// TIA Portal V17 export
// export: Created 2025-05-22T12:27:02.8614335Z, ExportSetting WithDefaults, DisplayName Totally Integrated Automation Portal, DisplayVersion V17 Update 8, DisplayName TIA Portal Openness, DisplayVersion V17 Update 8, DisplayName TIA Portal Version Control Interface, DisplayVersion V17, DisplayName SINAMICS Startdrive Advanced, DisplayVersion V17 SP2, DisplayName SINAMICS Startdrive G110M, G120, G120C, G120D, G120P, G115D, DisplayVersion V17 SP2, DisplayName SINAMICS Startdrive G130, G150, S120, S150, SINAMICS MV, S210, DisplayVersion V17 SP2, DisplayName STEP 7 Professional, DisplayVersion V17 Update 8, DisplayName SINUMERIK ONE STEP 7 Toolbox, DisplayVersion V17 Update 12, DisplayName SINUMERIK ONE PLC Basic Program Plus, DisplayVersion V17 Update 12, DisplayName SINUMERIK 840D sl STEP 7 Toolbox, DisplayVersion V17 Update 12, DisplayName STEP 7 Safety, DisplayVersion V17 Update 6, DisplayName WinCC Advanced, DisplayVersion V17 Update 8
FUNCTION "FC16701_OPC_UA_MASTER_MACHINE_DATA_UPDATE" : Void   // FC16701, LAD
{ S7_Optimized_Access := 'FALSE' }
VERSION : 0.1
// stored: AutoNumber false, IsIECCheckEnabled false, SetENOAutomatically false, UDAEnableTagReadback false
   VAR_TEMP
      RETVAL : Word;
      ZERO : Byte;   // ZERO
      STATUS_FILL : Int;   // STATUS FILL
      U01_ASPIRATION_FINAL_VALUE_AUX : Real;
      U02_ASPIRATION_FINAL_VALUE_AUX : Real;
   END_VAR
   VAR_TEMP   // added for the SCL form of the ladder/FBD networks
      _w1 : Bool;
      _w2 : Bool;
      _w3 : Bool;
      _w4 : Bool;
      _w5 : Bool;
   END_VAR
BEGIN

REGION Network 1: <<<<<<<<<<<<<<<<<<<< OPC UA MASTER MACHINE >>>>>>>>>>>>>>>>>>>>
END_REGION

REGION Network 2: GENERAL INFO - ID
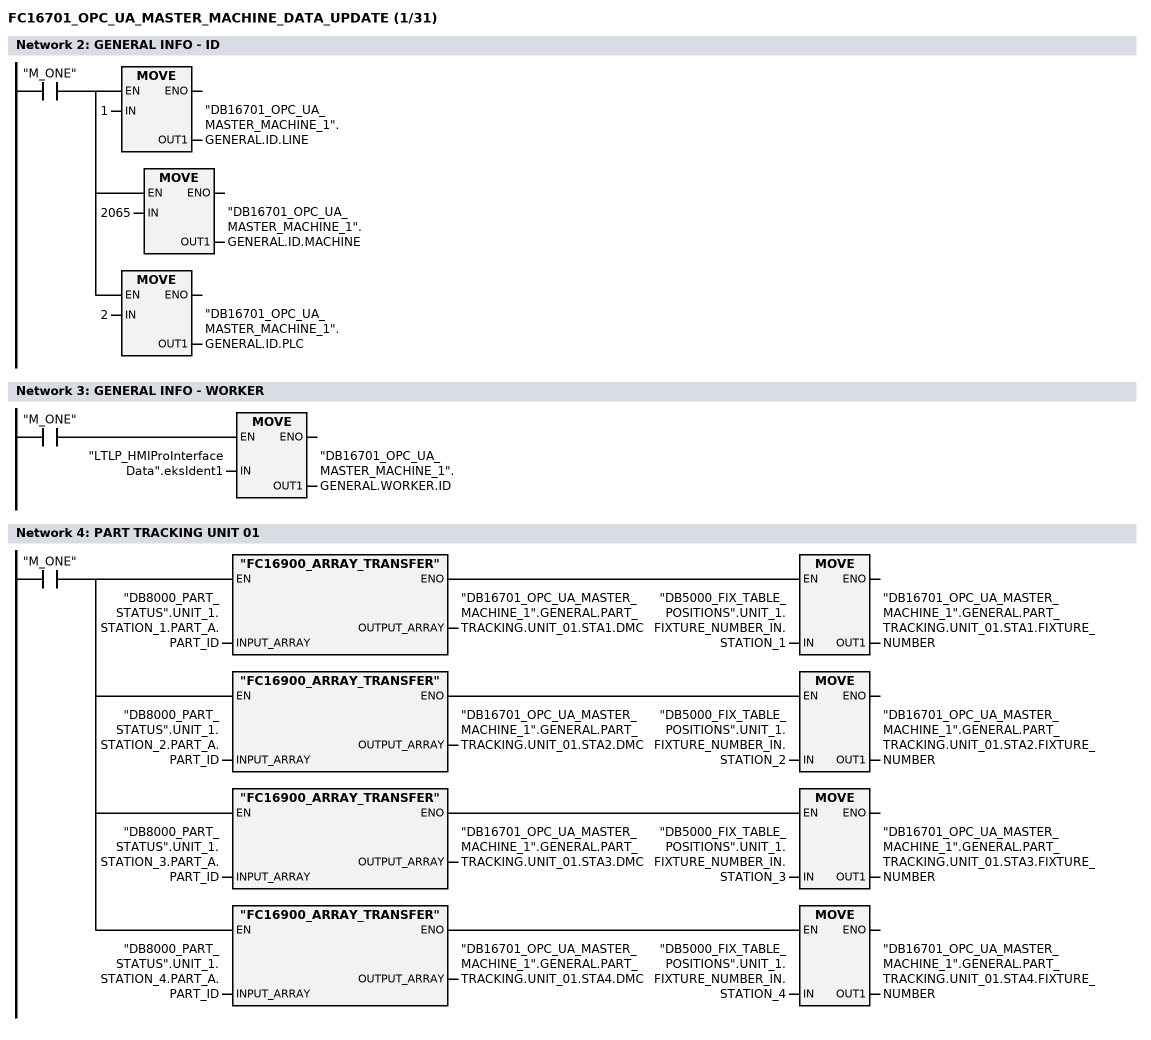
   RUNG wire#powerrail
      Contact( "M_ONE" )
      wire#w1
      Move(in := 1, out1 => "DB16701_OPC_UA_MASTER_MACHINE_1".GENERAL.ID.LINE)
   END_RUNG
   RUNG wire#w1
      Move(in := 2065, out1 => "DB16701_OPC_UA_MASTER_MACHINE_1".GENERAL.ID.MACHINE)
   END_RUNG
   RUNG wire#w1
      Move(in := 2, out1 => "DB16701_OPC_UA_MASTER_MACHINE_1".GENERAL.ID.PLC)
   END_RUNG
   // the same network as SCL:
   IF "M_ONE" THEN
       "DB16701_OPC_UA_MASTER_MACHINE_1".GENERAL.ID.LINE := 1;
       "DB16701_OPC_UA_MASTER_MACHINE_1".GENERAL.ID.MACHINE := 2065;
       "DB16701_OPC_UA_MASTER_MACHINE_1".GENERAL.ID.PLC := 2;
   END_IF;
END_REGION

REGION Network 3: GENERAL INFO - WORKER
   RUNG wire#powerrail
      Contact( "M_ONE" )
      Move(in := "LTLP_HMIProInterfaceData".eksIdent1, out1 => "DB16701_OPC_UA_MASTER_MACHINE_1".GENERAL.WORKER.ID)
   END_RUNG
   // the same network as SCL:
   IF "M_ONE" THEN
       "DB16701_OPC_UA_MASTER_MACHINE_1".GENERAL.WORKER.ID := "LTLP_HMIProInterfaceData".eksIdent1;
   END_IF;
END_REGION

REGION Network 4: PART TRACKING UNIT 01
   RUNG wire#powerrail
      Contact( "M_ONE" )
      wire#w1
      "FC16900_ARRAY_TRANSFER"(INPUT_ARRAY := "DB8000_PART_STATUS".UNIT_1.STATION_1.PART_A.PART_ID, OUTPUT_ARRAY => "DB16701_OPC_UA_MASTER_MACHINE_1".GENERAL.PART_TRACKING.UNIT_01.STA1.DMC)
      Move(in := "DB5000_FIX_TABLE_POSITIONS".UNIT_1.FIXTURE_NUMBER_IN.STATION_1, out1 => "DB16701_OPC_UA_MASTER_MACHINE_1".GENERAL.PART_TRACKING.UNIT_01.STA1.FIXTURE_NUMBER)
   END_RUNG
   RUNG wire#w1
      "FC16900_ARRAY_TRANSFER"(INPUT_ARRAY := "DB8000_PART_STATUS".UNIT_1.STATION_2.PART_A.PART_ID, OUTPUT_ARRAY => "DB16701_OPC_UA_MASTER_MACHINE_1".GENERAL.PART_TRACKING.UNIT_01.STA2.DMC)
      Move(in := "DB5000_FIX_TABLE_POSITIONS".UNIT_1.FIXTURE_NUMBER_IN.STATION_2, out1 => "DB16701_OPC_UA_MASTER_MACHINE_1".GENERAL.PART_TRACKING.UNIT_01.STA2.FIXTURE_NUMBER)
   END_RUNG
   RUNG wire#w1
      "FC16900_ARRAY_TRANSFER"(INPUT_ARRAY := "DB8000_PART_STATUS".UNIT_1.STATION_3.PART_A.PART_ID, OUTPUT_ARRAY => "DB16701_OPC_UA_MASTER_MACHINE_1".GENERAL.PART_TRACKING.UNIT_01.STA3.DMC)
      Move(in := "DB5000_FIX_TABLE_POSITIONS".UNIT_1.FIXTURE_NUMBER_IN.STATION_3, out1 => "DB16701_OPC_UA_MASTER_MACHINE_1".GENERAL.PART_TRACKING.UNIT_01.STA3.FIXTURE_NUMBER)
   END_RUNG
   RUNG wire#w1
      "FC16900_ARRAY_TRANSFER"(INPUT_ARRAY := "DB8000_PART_STATUS".UNIT_1.STATION_4.PART_A.PART_ID, OUTPUT_ARRAY => "DB16701_OPC_UA_MASTER_MACHINE_1".GENERAL.PART_TRACKING.UNIT_01.STA4.DMC)
      Move(in := "DB5000_FIX_TABLE_POSITIONS".UNIT_1.FIXTURE_NUMBER_IN.STATION_4, out1 => "DB16701_OPC_UA_MASTER_MACHINE_1".GENERAL.PART_TRACKING.UNIT_01.STA4.FIXTURE_NUMBER)
   END_RUNG
   // the same network as SCL:
   #_w2 := "M_ONE";
   "FC16900_ARRAY_TRANSFER"(EN := "M_ONE",
                           INPUT_ARRAY := "DB8000_PART_STATUS".UNIT_1.STATION_1.PART_A.PART_ID,
                           OUTPUT_ARRAY => "DB16701_OPC_UA_MASTER_MACHINE_1".GENERAL.PART_TRACKING.UNIT_01.STA1.DMC,
                           ENO => #_w1);
   IF #_w1 THEN
       "DB16701_OPC_UA_MASTER_MACHINE_1".GENERAL.PART_TRACKING.UNIT_01.STA1.FIXTURE_NUMBER := "DB5000_FIX_TABLE_POSITIONS".UNIT_1.FIXTURE_NUMBER_IN.STATION_1;
   END_IF;
   "FC16900_ARRAY_TRANSFER"(EN := #_w2,
                           INPUT_ARRAY := "DB8000_PART_STATUS".UNIT_1.STATION_2.PART_A.PART_ID,
                           OUTPUT_ARRAY => "DB16701_OPC_UA_MASTER_MACHINE_1".GENERAL.PART_TRACKING.UNIT_01.STA2.DMC,
                           ENO => #_w3);
   IF #_w3 THEN
       "DB16701_OPC_UA_MASTER_MACHINE_1".GENERAL.PART_TRACKING.UNIT_01.STA2.FIXTURE_NUMBER := "DB5000_FIX_TABLE_POSITIONS".UNIT_1.FIXTURE_NUMBER_IN.STATION_2;
   END_IF;
   "FC16900_ARRAY_TRANSFER"(EN := #_w2,
                           INPUT_ARRAY := "DB8000_PART_STATUS".UNIT_1.STATION_3.PART_A.PART_ID,
                           OUTPUT_ARRAY => "DB16701_OPC_UA_MASTER_MACHINE_1".GENERAL.PART_TRACKING.UNIT_01.STA3.DMC,
                           ENO => #_w4);
   IF #_w4 THEN
       "DB16701_OPC_UA_MASTER_MACHINE_1".GENERAL.PART_TRACKING.UNIT_01.STA3.FIXTURE_NUMBER := "DB5000_FIX_TABLE_POSITIONS".UNIT_1.FIXTURE_NUMBER_IN.STATION_3;
   END_IF;
   "FC16900_ARRAY_TRANSFER"(EN := #_w2,
                           INPUT_ARRAY := "DB8000_PART_STATUS".UNIT_1.STATION_4.PART_A.PART_ID,
                           OUTPUT_ARRAY => "DB16701_OPC_UA_MASTER_MACHINE_1".GENERAL.PART_TRACKING.UNIT_01.STA4.DMC,
                           ENO => #_w5);
   IF #_w5 THEN
       "DB16701_OPC_UA_MASTER_MACHINE_1".GENERAL.PART_TRACKING.UNIT_01.STA4.FIXTURE_NUMBER := "DB5000_FIX_TABLE_POSITIONS".UNIT_1.FIXTURE_NUMBER_IN.STATION_4;
   END_IF;
END_REGION

REGION Network 5: PART TRACKING UNIT 02
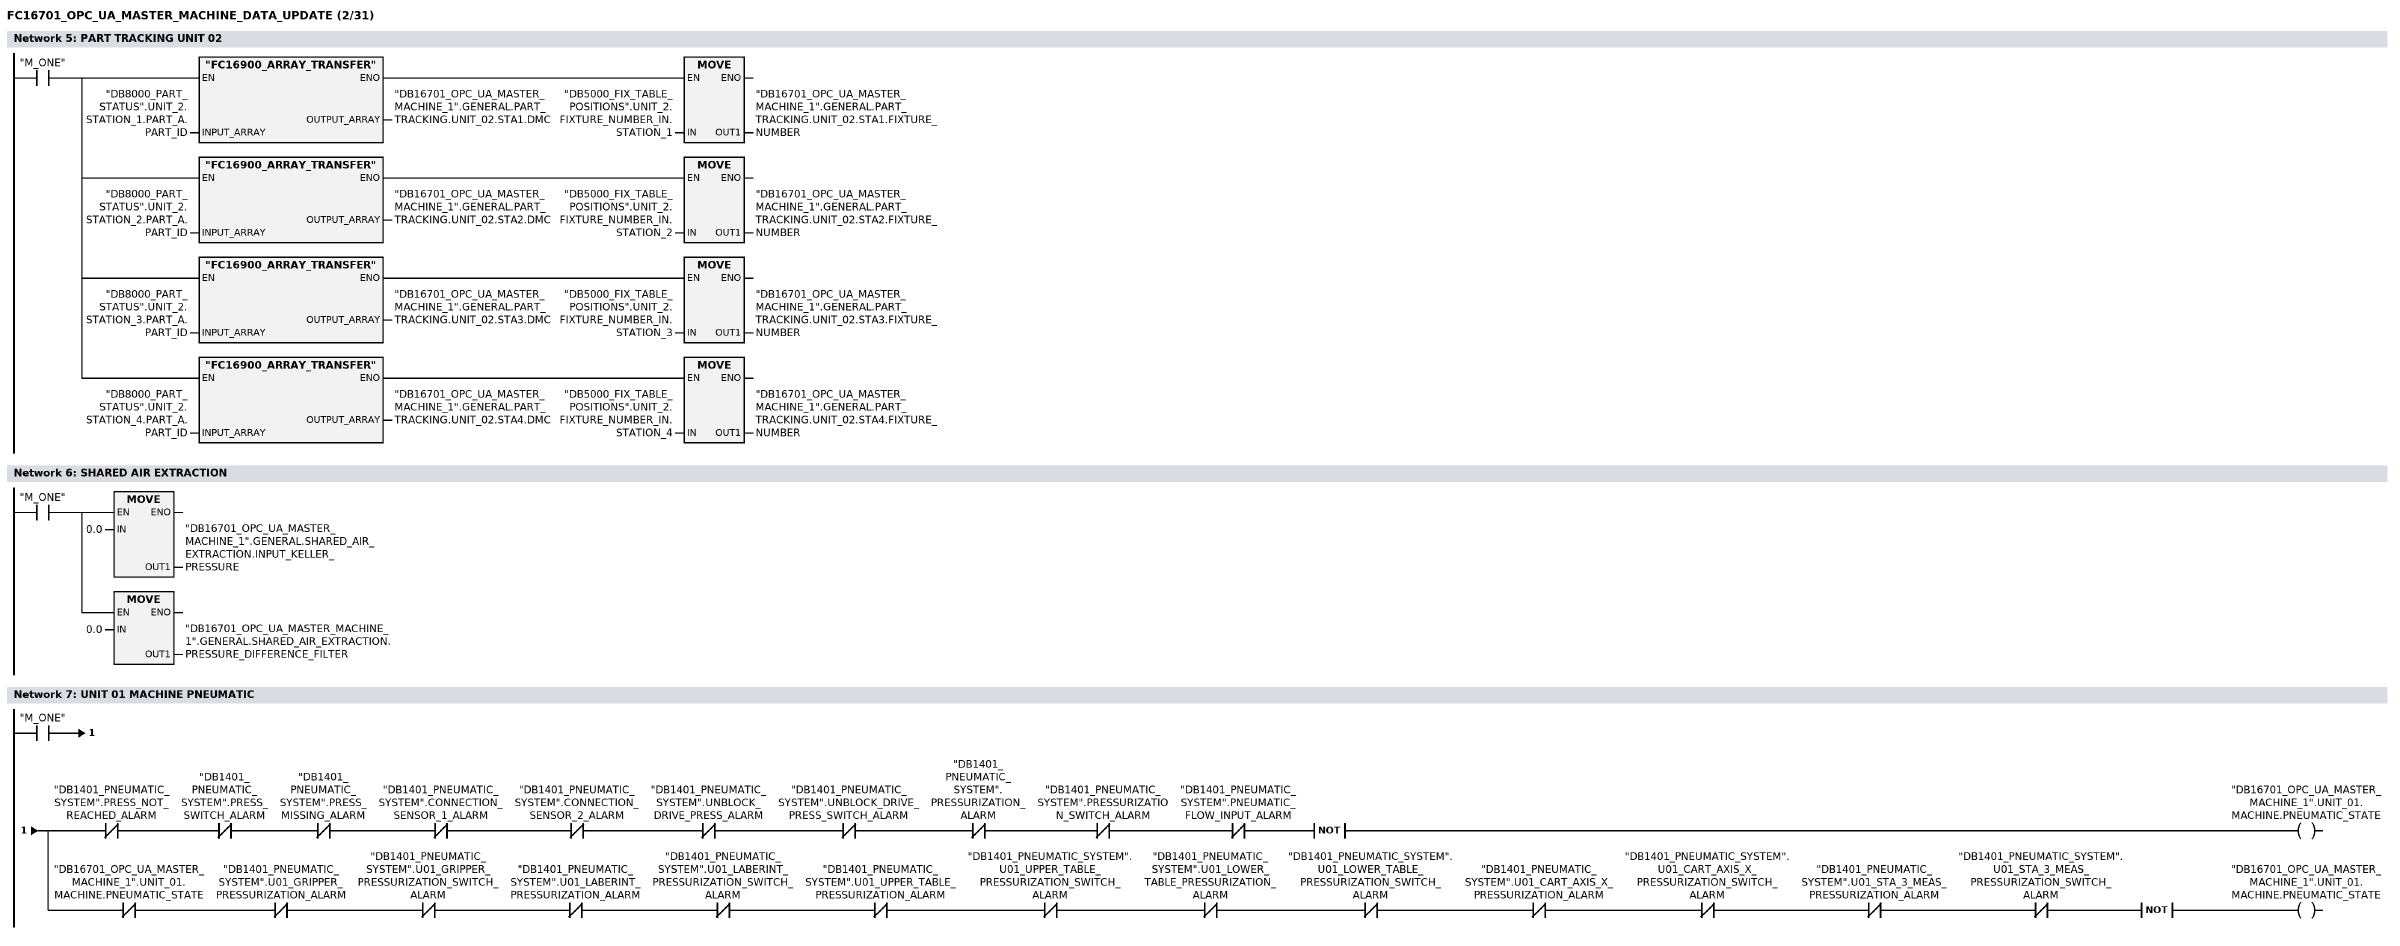
   RUNG wire#powerrail
      Contact( "M_ONE" )
      wire#w1
      "FC16900_ARRAY_TRANSFER"(INPUT_ARRAY := "DB8000_PART_STATUS".UNIT_2.STATION_1.PART_A.PART_ID, OUTPUT_ARRAY => "DB16701_OPC_UA_MASTER_MACHINE_1".GENERAL.PART_TRACKING.UNIT_02.STA1.DMC)
      Move(in := "DB5000_FIX_TABLE_POSITIONS".UNIT_2.FIXTURE_NUMBER_IN.STATION_1, out1 => "DB16701_OPC_UA_MASTER_MACHINE_1".GENERAL.PART_TRACKING.UNIT_02.STA1.FIXTURE_NUMBER)
   END_RUNG
   RUNG wire#w1
      "FC16900_ARRAY_TRANSFER"(INPUT_ARRAY := "DB8000_PART_STATUS".UNIT_2.STATION_2.PART_A.PART_ID, OUTPUT_ARRAY => "DB16701_OPC_UA_MASTER_MACHINE_1".GENERAL.PART_TRACKING.UNIT_02.STA2.DMC)
      Move(in := "DB5000_FIX_TABLE_POSITIONS".UNIT_2.FIXTURE_NUMBER_IN.STATION_2, out1 => "DB16701_OPC_UA_MASTER_MACHINE_1".GENERAL.PART_TRACKING.UNIT_02.STA2.FIXTURE_NUMBER)
   END_RUNG
   RUNG wire#w1
      "FC16900_ARRAY_TRANSFER"(INPUT_ARRAY := "DB8000_PART_STATUS".UNIT_2.STATION_3.PART_A.PART_ID, OUTPUT_ARRAY => "DB16701_OPC_UA_MASTER_MACHINE_1".GENERAL.PART_TRACKING.UNIT_02.STA3.DMC)
      Move(in := "DB5000_FIX_TABLE_POSITIONS".UNIT_2.FIXTURE_NUMBER_IN.STATION_3, out1 => "DB16701_OPC_UA_MASTER_MACHINE_1".GENERAL.PART_TRACKING.UNIT_02.STA3.FIXTURE_NUMBER)
   END_RUNG
   RUNG wire#w1
      "FC16900_ARRAY_TRANSFER"(INPUT_ARRAY := "DB8000_PART_STATUS".UNIT_2.STATION_4.PART_A.PART_ID, OUTPUT_ARRAY => "DB16701_OPC_UA_MASTER_MACHINE_1".GENERAL.PART_TRACKING.UNIT_02.STA4.DMC)
      Move(in := "DB5000_FIX_TABLE_POSITIONS".UNIT_2.FIXTURE_NUMBER_IN.STATION_4, out1 => "DB16701_OPC_UA_MASTER_MACHINE_1".GENERAL.PART_TRACKING.UNIT_02.STA4.FIXTURE_NUMBER)
   END_RUNG
   // the same network as SCL:
   #_w2 := "M_ONE";
   "FC16900_ARRAY_TRANSFER"(EN := "M_ONE",
                           INPUT_ARRAY := "DB8000_PART_STATUS".UNIT_2.STATION_1.PART_A.PART_ID,
                           OUTPUT_ARRAY => "DB16701_OPC_UA_MASTER_MACHINE_1".GENERAL.PART_TRACKING.UNIT_02.STA1.DMC,
                           ENO => #_w1);
   IF #_w1 THEN
       "DB16701_OPC_UA_MASTER_MACHINE_1".GENERAL.PART_TRACKING.UNIT_02.STA1.FIXTURE_NUMBER := "DB5000_FIX_TABLE_POSITIONS".UNIT_2.FIXTURE_NUMBER_IN.STATION_1;
   END_IF;
   "FC16900_ARRAY_TRANSFER"(EN := #_w2,
                           INPUT_ARRAY := "DB8000_PART_STATUS".UNIT_2.STATION_2.PART_A.PART_ID,
                           OUTPUT_ARRAY => "DB16701_OPC_UA_MASTER_MACHINE_1".GENERAL.PART_TRACKING.UNIT_02.STA2.DMC,
                           ENO => #_w3);
   IF #_w3 THEN
       "DB16701_OPC_UA_MASTER_MACHINE_1".GENERAL.PART_TRACKING.UNIT_02.STA2.FIXTURE_NUMBER := "DB5000_FIX_TABLE_POSITIONS".UNIT_2.FIXTURE_NUMBER_IN.STATION_2;
   END_IF;
   "FC16900_ARRAY_TRANSFER"(EN := #_w2,
                           INPUT_ARRAY := "DB8000_PART_STATUS".UNIT_2.STATION_3.PART_A.PART_ID,
                           OUTPUT_ARRAY => "DB16701_OPC_UA_MASTER_MACHINE_1".GENERAL.PART_TRACKING.UNIT_02.STA3.DMC,
                           ENO => #_w4);
   IF #_w4 THEN
       "DB16701_OPC_UA_MASTER_MACHINE_1".GENERAL.PART_TRACKING.UNIT_02.STA3.FIXTURE_NUMBER := "DB5000_FIX_TABLE_POSITIONS".UNIT_2.FIXTURE_NUMBER_IN.STATION_3;
   END_IF;
   "FC16900_ARRAY_TRANSFER"(EN := #_w2,
                           INPUT_ARRAY := "DB8000_PART_STATUS".UNIT_2.STATION_4.PART_A.PART_ID,
                           OUTPUT_ARRAY => "DB16701_OPC_UA_MASTER_MACHINE_1".GENERAL.PART_TRACKING.UNIT_02.STA4.DMC,
                           ENO => #_w5);
   IF #_w5 THEN
       "DB16701_OPC_UA_MASTER_MACHINE_1".GENERAL.PART_TRACKING.UNIT_02.STA4.FIXTURE_NUMBER := "DB5000_FIX_TABLE_POSITIONS".UNIT_2.FIXTURE_NUMBER_IN.STATION_4;
   END_IF;
END_REGION

REGION Network 6: SHARED AIR EXTRACTION
   RUNG wire#powerrail
      Contact( "M_ONE" )
      wire#w1
      Move(in := 0.0, out1 => "DB16701_OPC_UA_MASTER_MACHINE_1".GENERAL.SHARED_AIR_EXTRACTION.INPUT_KELLER_PRESSURE)
   END_RUNG
   RUNG wire#w1
      Move(in := 0.0, out1 => "DB16701_OPC_UA_MASTER_MACHINE_1".GENERAL.SHARED_AIR_EXTRACTION.PRESSURE_DIFFERENCE_FILTER)
   END_RUNG
   // the same network as SCL:
   IF "M_ONE" THEN
       "DB16701_OPC_UA_MASTER_MACHINE_1".GENERAL.SHARED_AIR_EXTRACTION.INPUT_KELLER_PRESSURE := 0.0;
       "DB16701_OPC_UA_MASTER_MACHINE_1".GENERAL.SHARED_AIR_EXTRACTION.PRESSURE_DIFFERENCE_FILTER := 0.0;
   END_IF;
END_REGION

REGION Network 7: UNIT 01 MACHINE PNEUMATIC
   RUNG wire#powerrail
      Contact( "M_ONE" )
      wire#w1
      I_Contact( "DB1401_PNEUMATIC_SYSTEM".PRESS_NOT_REACHED_ALARM )
      I_Contact( "DB1401_PNEUMATIC_SYSTEM".PRESS_SWITCH_ALARM )
      I_Contact( "DB1401_PNEUMATIC_SYSTEM".PRESS_MISSING_ALARM )
      I_Contact( "DB1401_PNEUMATIC_SYSTEM".CONNECTION_SENSOR_1_ALARM )
      I_Contact( "DB1401_PNEUMATIC_SYSTEM".CONNECTION_SENSOR_2_ALARM )
      I_Contact( "DB1401_PNEUMATIC_SYSTEM".UNBLOCK_DRIVE_PRESS_ALARM )
      I_Contact( "DB1401_PNEUMATIC_SYSTEM".UNBLOCK_DRIVE_PRESS_SWITCH_ALARM )
      I_Contact( "DB1401_PNEUMATIC_SYSTEM".PRESSURIZATION_ALARM )
      I_Contact( "DB1401_PNEUMATIC_SYSTEM".PRESSURIZATION_SWITCH_ALARM )
      I_Contact( "DB1401_PNEUMATIC_SYSTEM".PNEUMATIC_FLOW_INPUT_ALARM )
      Not()
      Coil( "DB16701_OPC_UA_MASTER_MACHINE_1".UNIT_01.MACHINE.PNEUMATIC_STATE )
   END_RUNG
   RUNG wire#w1
      I_Contact( "DB16701_OPC_UA_MASTER_MACHINE_1".UNIT_01.MACHINE.PNEUMATIC_STATE )
      I_Contact( "DB1401_PNEUMATIC_SYSTEM".U01_GRIPPER_PRESSURIZATION_ALARM )
      I_Contact( "DB1401_PNEUMATIC_SYSTEM".U01_GRIPPER_PRESSURIZATION_SWITCH_ALARM )
      I_Contact( "DB1401_PNEUMATIC_SYSTEM".U01_LABERINT_PRESSURIZATION_ALARM )
      I_Contact( "DB1401_PNEUMATIC_SYSTEM".U01_LABERINT_PRESSURIZATION_SWITCH_ALARM )
      I_Contact( "DB1401_PNEUMATIC_SYSTEM".U01_UPPER_TABLE_PRESSURIZATION_ALARM )
      I_Contact( "DB1401_PNEUMATIC_SYSTEM".U01_UPPER_TABLE_PRESSURIZATION_SWITCH_ALARM )
      I_Contact( "DB1401_PNEUMATIC_SYSTEM".U01_LOWER_TABLE_PRESSURIZATION_ALARM )
      I_Contact( "DB1401_PNEUMATIC_SYSTEM".U01_LOWER_TABLE_PRESSURIZATION_SWITCH_ALARM )
      I_Contact( "DB1401_PNEUMATIC_SYSTEM".U01_CART_AXIS_X_PRESSURIZATION_ALARM )
      I_Contact( "DB1401_PNEUMATIC_SYSTEM".U01_CART_AXIS_X_PRESSURIZATION_SWITCH_ALARM )
      I_Contact( "DB1401_PNEUMATIC_SYSTEM".U01_STA_3_MEAS_PRESSURIZATION_ALARM )
      I_Contact( "DB1401_PNEUMATIC_SYSTEM".U01_STA_3_MEAS_PRESSURIZATION_SWITCH_ALARM )
      Not()
      Coil( "DB16701_OPC_UA_MASTER_MACHINE_1".UNIT_01.MACHINE.PNEUMATIC_STATE )
   END_RUNG
   // the same network as SCL:
   "DB16701_OPC_UA_MASTER_MACHINE_1".UNIT_01.MACHINE.PNEUMATIC_STATE := NOT ("M_ONE" AND NOT "DB1401_PNEUMATIC_SYSTEM".PRESS_NOT_REACHED_ALARM AND NOT "DB1401_PNEUMATIC_SYSTEM".PRESS_SWITCH_ALARM AND NOT "DB1401_PNEUMATIC_SYSTEM".PRESS_MISSING_ALARM AND NOT "DB1401_PNEUMATIC_SYSTEM".CONNECTION_SENSOR_1_ALARM AND NOT "DB1401_PNEUMATIC_SYSTEM".CONNECTION_SENSOR_2_ALARM AND NOT "DB1401_PNEUMATIC_SYSTEM".UNBLOCK_DRIVE_PRESS_ALARM AND NOT "DB1401_PNEUMATIC_SYSTEM".UNBLOCK_DRIVE_PRESS_SWITCH_ALARM AND NOT "DB1401_PNEUMATIC_SYSTEM".PRESSURIZATION_ALARM AND NOT "DB1401_PNEUMATIC_SYSTEM".PRESSURIZATION_SWITCH_ALARM AND NOT "DB1401_PNEUMATIC_SYSTEM".PNEUMATIC_FLOW_INPUT_ALARM);
   "DB16701_OPC_UA_MASTER_MACHINE_1".UNIT_01.MACHINE.PNEUMATIC_STATE := NOT ("M_ONE" AND NOT "DB16701_OPC_UA_MASTER_MACHINE_1".UNIT_01.MACHINE.PNEUMATIC_STATE AND NOT "DB1401_PNEUMATIC_SYSTEM".U01_GRIPPER_PRESSURIZATION_ALARM AND NOT "DB1401_PNEUMATIC_SYSTEM".U01_GRIPPER_PRESSURIZATION_SWITCH_ALARM AND NOT "DB1401_PNEUMATIC_SYSTEM".U01_LABERINT_PRESSURIZATION_ALARM AND NOT "DB1401_PNEUMATIC_SYSTEM".U01_LABERINT_PRESSURIZATION_SWITCH_ALARM AND NOT "DB1401_PNEUMATIC_SYSTEM".U01_UPPER_TABLE_PRESSURIZATION_ALARM AND NOT "DB1401_PNEUMATIC_SYSTEM".U01_UPPER_TABLE_PRESSURIZATION_SWITCH_ALARM AND NOT "DB1401_PNEUMATIC_SYSTEM".U01_LOWER_TABLE_PRESSURIZATION_ALARM AND NOT "DB1401_PNEUMATIC_SYSTEM".U01_LOWER_TABLE_PRESSURIZATION_SWITCH_ALARM AND NOT "DB1401_PNEUMATIC_SYSTEM".U01_CART_AXIS_X_PRESSURIZATION_ALARM AND NOT "DB1401_PNEUMATIC_SYSTEM".U01_CART_AXIS_X_PRESSURIZATION_SWITCH_ALARM AND NOT "DB1401_PNEUMATIC_SYSTEM".U01_STA_3_MEAS_PRESSURIZATION_ALARM AND NOT "DB1401_PNEUMATIC_SYSTEM".U01_STA_3_MEAS_PRESSURIZATION_SWITCH_ALARM);
END_REGION

REGION Network 8: UNIT 01 MACHINE TEMPERATURE
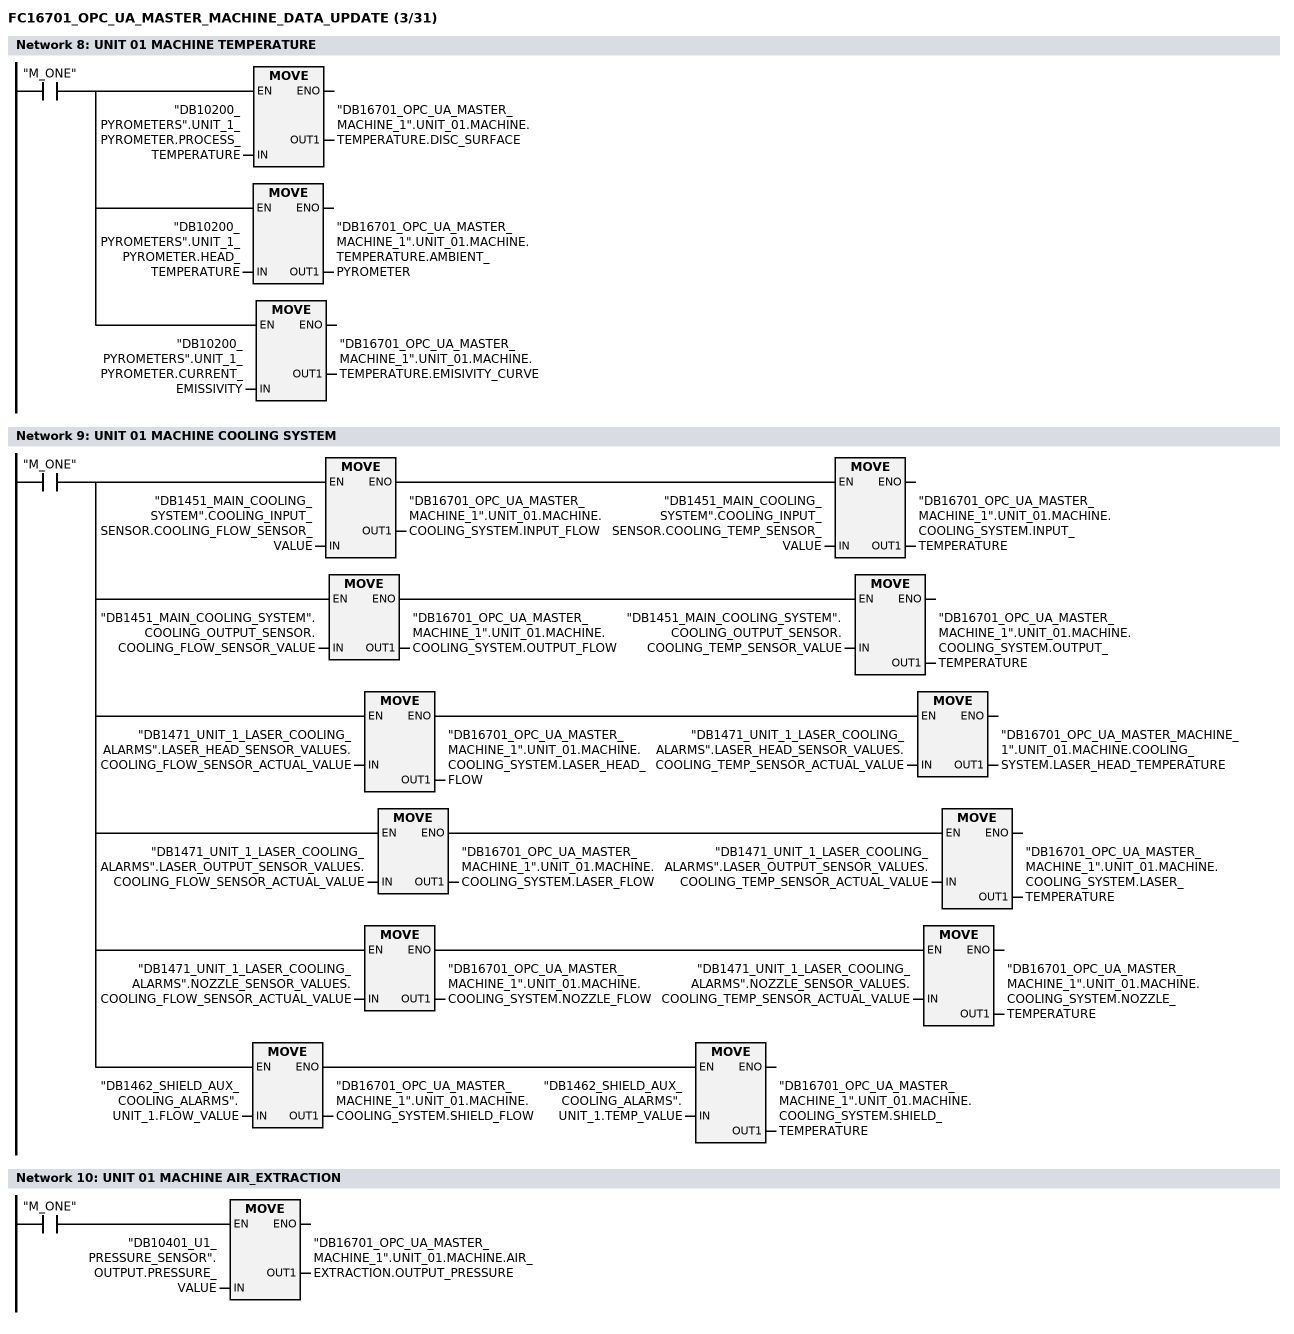
   RUNG wire#powerrail
      Contact( "M_ONE" )
      wire#w1
      Move(in := "DB10200_PYROMETERS".UNIT_1_PYROMETER.PROCESS_TEMPERATURE, out1 => "DB16701_OPC_UA_MASTER_MACHINE_1".UNIT_01.MACHINE.TEMPERATURE.DISC_SURFACE)
   END_RUNG
   RUNG wire#w1
      Move(in := "DB10200_PYROMETERS".UNIT_1_PYROMETER.HEAD_TEMPERATURE, out1 => "DB16701_OPC_UA_MASTER_MACHINE_1".UNIT_01.MACHINE.TEMPERATURE.AMBIENT_PYROMETER)
   END_RUNG
   RUNG wire#w1
      Move(in := "DB10200_PYROMETERS".UNIT_1_PYROMETER.CURRENT_EMISSIVITY, out1 => "DB16701_OPC_UA_MASTER_MACHINE_1".UNIT_01.MACHINE.TEMPERATURE.EMISIVITY_CURVE)
   END_RUNG
   // the same network as SCL:
   IF "M_ONE" THEN
       "DB16701_OPC_UA_MASTER_MACHINE_1".UNIT_01.MACHINE.TEMPERATURE.DISC_SURFACE := "DB10200_PYROMETERS".UNIT_1_PYROMETER.PROCESS_TEMPERATURE;
       "DB16701_OPC_UA_MASTER_MACHINE_1".UNIT_01.MACHINE.TEMPERATURE.AMBIENT_PYROMETER := "DB10200_PYROMETERS".UNIT_1_PYROMETER.HEAD_TEMPERATURE;
       "DB16701_OPC_UA_MASTER_MACHINE_1".UNIT_01.MACHINE.TEMPERATURE.EMISIVITY_CURVE := "DB10200_PYROMETERS".UNIT_1_PYROMETER.CURRENT_EMISSIVITY;
   END_IF;
END_REGION

REGION Network 9: UNIT 01 MACHINE COOLING SYSTEM
   RUNG wire#powerrail
      Contact( "M_ONE" )
      wire#w1
      Move(in := "DB1451_MAIN_COOLING_SYSTEM".COOLING_INPUT_SENSOR.COOLING_FLOW_SENSOR_VALUE, out1 => "DB16701_OPC_UA_MASTER_MACHINE_1".UNIT_01.MACHINE.COOLING_SYSTEM.INPUT_FLOW)
      Move(in := "DB1451_MAIN_COOLING_SYSTEM".COOLING_INPUT_SENSOR.COOLING_TEMP_SENSOR_VALUE, out1 => "DB16701_OPC_UA_MASTER_MACHINE_1".UNIT_01.MACHINE.COOLING_SYSTEM.INPUT_TEMPERATURE)
   END_RUNG
   RUNG wire#w1
      Move(in := "DB1451_MAIN_COOLING_SYSTEM".COOLING_OUTPUT_SENSOR.COOLING_FLOW_SENSOR_VALUE, out1 => "DB16701_OPC_UA_MASTER_MACHINE_1".UNIT_01.MACHINE.COOLING_SYSTEM.OUTPUT_FLOW)
      Move(in := "DB1451_MAIN_COOLING_SYSTEM".COOLING_OUTPUT_SENSOR.COOLING_TEMP_SENSOR_VALUE, out1 => "DB16701_OPC_UA_MASTER_MACHINE_1".UNIT_01.MACHINE.COOLING_SYSTEM.OUTPUT_TEMPERATURE)
   END_RUNG
   RUNG wire#w1
      Move(in := "DB1471_UNIT_1_LASER_COOLING_ALARMS".LASER_HEAD_SENSOR_VALUES.COOLING_FLOW_SENSOR_ACTUAL_VALUE, out1 => "DB16701_OPC_UA_MASTER_MACHINE_1".UNIT_01.MACHINE.COOLING_SYSTEM.LASER_HEAD_FLOW)
      Move(in := "DB1471_UNIT_1_LASER_COOLING_ALARMS".LASER_HEAD_SENSOR_VALUES.COOLING_TEMP_SENSOR_ACTUAL_VALUE, out1 => "DB16701_OPC_UA_MASTER_MACHINE_1".UNIT_01.MACHINE.COOLING_SYSTEM.LASER_HEAD_TEMPERATURE)
   END_RUNG
   RUNG wire#w1
      Move(in := "DB1471_UNIT_1_LASER_COOLING_ALARMS".LASER_OUTPUT_SENSOR_VALUES.COOLING_FLOW_SENSOR_ACTUAL_VALUE, out1 => "DB16701_OPC_UA_MASTER_MACHINE_1".UNIT_01.MACHINE.COOLING_SYSTEM.LASER_FLOW)
      Move(in := "DB1471_UNIT_1_LASER_COOLING_ALARMS".LASER_OUTPUT_SENSOR_VALUES.COOLING_TEMP_SENSOR_ACTUAL_VALUE, out1 => "DB16701_OPC_UA_MASTER_MACHINE_1".UNIT_01.MACHINE.COOLING_SYSTEM.LASER_TEMPERATURE)
   END_RUNG
   RUNG wire#w1
      Move(in := "DB1471_UNIT_1_LASER_COOLING_ALARMS".NOZZLE_SENSOR_VALUES.COOLING_FLOW_SENSOR_ACTUAL_VALUE, out1 => "DB16701_OPC_UA_MASTER_MACHINE_1".UNIT_01.MACHINE.COOLING_SYSTEM.NOZZLE_FLOW)
      Move(in := "DB1471_UNIT_1_LASER_COOLING_ALARMS".NOZZLE_SENSOR_VALUES.COOLING_TEMP_SENSOR_ACTUAL_VALUE, out1 => "DB16701_OPC_UA_MASTER_MACHINE_1".UNIT_01.MACHINE.COOLING_SYSTEM.NOZZLE_TEMPERATURE)
   END_RUNG
   RUNG wire#w1
      Move(in := "DB1462_SHIELD_AUX_COOLING_ALARMS".UNIT_1.FLOW_VALUE, out1 => "DB16701_OPC_UA_MASTER_MACHINE_1".UNIT_01.MACHINE.COOLING_SYSTEM.SHIELD_FLOW)
      Move(in := "DB1462_SHIELD_AUX_COOLING_ALARMS".UNIT_1.TEMP_VALUE, out1 => "DB16701_OPC_UA_MASTER_MACHINE_1".UNIT_01.MACHINE.COOLING_SYSTEM.SHIELD_TEMPERATURE)
   END_RUNG
   // the same network as SCL:
   IF "M_ONE" THEN
       "DB16701_OPC_UA_MASTER_MACHINE_1".UNIT_01.MACHINE.COOLING_SYSTEM.INPUT_FLOW := "DB1451_MAIN_COOLING_SYSTEM".COOLING_INPUT_SENSOR.COOLING_FLOW_SENSOR_VALUE;
       "DB16701_OPC_UA_MASTER_MACHINE_1".UNIT_01.MACHINE.COOLING_SYSTEM.INPUT_TEMPERATURE := "DB1451_MAIN_COOLING_SYSTEM".COOLING_INPUT_SENSOR.COOLING_TEMP_SENSOR_VALUE;
       "DB16701_OPC_UA_MASTER_MACHINE_1".UNIT_01.MACHINE.COOLING_SYSTEM.OUTPUT_FLOW := "DB1451_MAIN_COOLING_SYSTEM".COOLING_OUTPUT_SENSOR.COOLING_FLOW_SENSOR_VALUE;
       "DB16701_OPC_UA_MASTER_MACHINE_1".UNIT_01.MACHINE.COOLING_SYSTEM.OUTPUT_TEMPERATURE := "DB1451_MAIN_COOLING_SYSTEM".COOLING_OUTPUT_SENSOR.COOLING_TEMP_SENSOR_VALUE;
       "DB16701_OPC_UA_MASTER_MACHINE_1".UNIT_01.MACHINE.COOLING_SYSTEM.LASER_HEAD_FLOW := "DB1471_UNIT_1_LASER_COOLING_ALARMS".LASER_HEAD_SENSOR_VALUES.COOLING_FLOW_SENSOR_ACTUAL_VALUE;
       "DB16701_OPC_UA_MASTER_MACHINE_1".UNIT_01.MACHINE.COOLING_SYSTEM.LASER_HEAD_TEMPERATURE := "DB1471_UNIT_1_LASER_COOLING_ALARMS".LASER_HEAD_SENSOR_VALUES.COOLING_TEMP_SENSOR_ACTUAL_VALUE;
       "DB16701_OPC_UA_MASTER_MACHINE_1".UNIT_01.MACHINE.COOLING_SYSTEM.LASER_FLOW := "DB1471_UNIT_1_LASER_COOLING_ALARMS".LASER_OUTPUT_SENSOR_VALUES.COOLING_FLOW_SENSOR_ACTUAL_VALUE;
       "DB16701_OPC_UA_MASTER_MACHINE_1".UNIT_01.MACHINE.COOLING_SYSTEM.LASER_TEMPERATURE := "DB1471_UNIT_1_LASER_COOLING_ALARMS".LASER_OUTPUT_SENSOR_VALUES.COOLING_TEMP_SENSOR_ACTUAL_VALUE;
       "DB16701_OPC_UA_MASTER_MACHINE_1".UNIT_01.MACHINE.COOLING_SYSTEM.NOZZLE_FLOW := "DB1471_UNIT_1_LASER_COOLING_ALARMS".NOZZLE_SENSOR_VALUES.COOLING_FLOW_SENSOR_ACTUAL_VALUE;
       "DB16701_OPC_UA_MASTER_MACHINE_1".UNIT_01.MACHINE.COOLING_SYSTEM.NOZZLE_TEMPERATURE := "DB1471_UNIT_1_LASER_COOLING_ALARMS".NOZZLE_SENSOR_VALUES.COOLING_TEMP_SENSOR_ACTUAL_VALUE;
       "DB16701_OPC_UA_MASTER_MACHINE_1".UNIT_01.MACHINE.COOLING_SYSTEM.SHIELD_FLOW := "DB1462_SHIELD_AUX_COOLING_ALARMS".UNIT_1.FLOW_VALUE;
       "DB16701_OPC_UA_MASTER_MACHINE_1".UNIT_01.MACHINE.COOLING_SYSTEM.SHIELD_TEMPERATURE := "DB1462_SHIELD_AUX_COOLING_ALARMS".UNIT_1.TEMP_VALUE;
   END_IF;
END_REGION

REGION Network 10: UNIT 01 MACHINE AIR_EXTRACTION
   RUNG wire#powerrail
      Contact( "M_ONE" )
      Move(in := "DB10401_U1_PRESSURE_SENSOR".OUTPUT.PRESSURE_VALUE, out1 => "DB16701_OPC_UA_MASTER_MACHINE_1".UNIT_01.MACHINE.AIR_EXTRACTION.OUTPUT_PRESSURE)
   END_RUNG
   // the same network as SCL:
   IF "M_ONE" THEN
       "DB16701_OPC_UA_MASTER_MACHINE_1".UNIT_01.MACHINE.AIR_EXTRACTION.OUTPUT_PRESSURE := "DB10401_U1_PRESSURE_SENSOR".OUTPUT.PRESSURE_VALUE;
   END_IF;
END_REGION

REGION Network 11: UNIT 01 MACHINE ST3 PRESSURE CONTROL
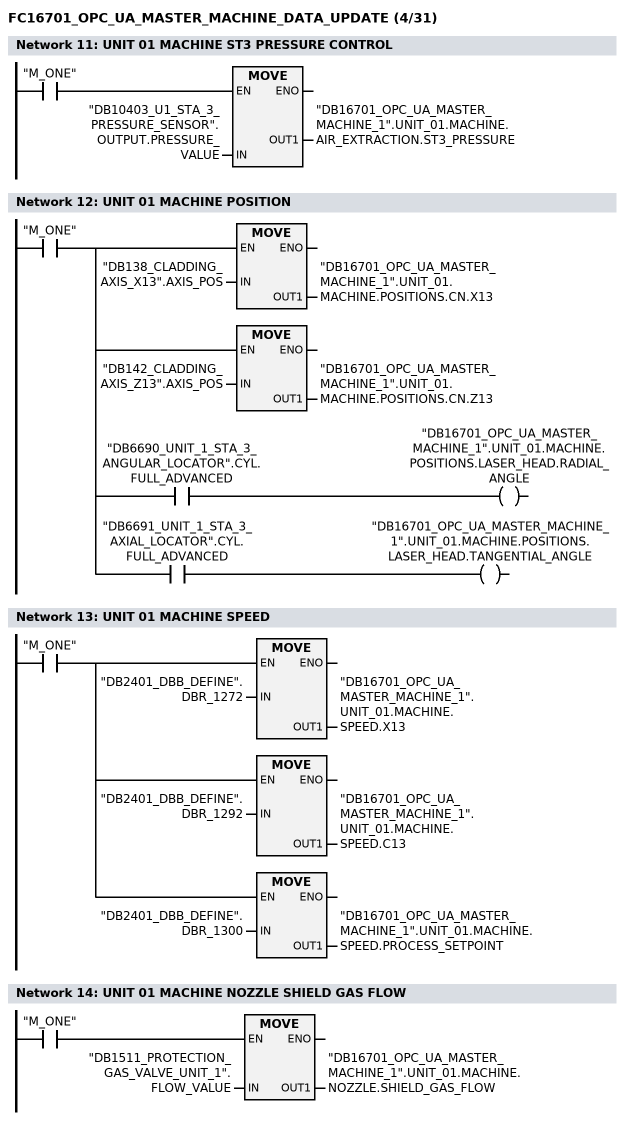
   RUNG wire#powerrail
      Contact( "M_ONE" )
      Move(in := "DB10403_U1_STA_3_PRESSURE_SENSOR".OUTPUT.PRESSURE_VALUE, out1 => "DB16701_OPC_UA_MASTER_MACHINE_1".UNIT_01.MACHINE.AIR_EXTRACTION.ST3_PRESSURE)
   END_RUNG
   // the same network as SCL:
   IF "M_ONE" THEN
       "DB16701_OPC_UA_MASTER_MACHINE_1".UNIT_01.MACHINE.AIR_EXTRACTION.ST3_PRESSURE := "DB10403_U1_STA_3_PRESSURE_SENSOR".OUTPUT.PRESSURE_VALUE;
   END_IF;
END_REGION

REGION Network 12: UNIT 01 MACHINE POSITION
   RUNG wire#powerrail
      Contact( "M_ONE" )
      wire#w1
      Move(in := "DB138_CLADDING_AXIS_X13".AXIS_POS, out1 => "DB16701_OPC_UA_MASTER_MACHINE_1".UNIT_01.MACHINE.POSITIONS.CN.X13)
   END_RUNG
   RUNG wire#w1
      Move(in := "DB142_CLADDING_AXIS_Z13".AXIS_POS, out1 => "DB16701_OPC_UA_MASTER_MACHINE_1".UNIT_01.MACHINE.POSITIONS.CN.Z13)
   END_RUNG
   RUNG wire#w1
      Contact( "DB6690_UNIT_1_STA_3_ANGULAR_LOCATOR".CYL.FULL_ADVANCED )
      Coil( "DB16701_OPC_UA_MASTER_MACHINE_1".UNIT_01.MACHINE.POSITIONS.LASER_HEAD.RADIAL_ANGLE )
   END_RUNG
   RUNG wire#w1
      Contact( "DB6691_UNIT_1_STA_3_AXIAL_LOCATOR".CYL.FULL_ADVANCED )
      Coil( "DB16701_OPC_UA_MASTER_MACHINE_1".UNIT_01.MACHINE.POSITIONS.LASER_HEAD.TANGENTIAL_ANGLE )
   END_RUNG
   // the same network as SCL:
   IF "M_ONE" THEN
       "DB16701_OPC_UA_MASTER_MACHINE_1".UNIT_01.MACHINE.POSITIONS.CN.X13 := "DB138_CLADDING_AXIS_X13".AXIS_POS;
       "DB16701_OPC_UA_MASTER_MACHINE_1".UNIT_01.MACHINE.POSITIONS.CN.Z13 := "DB142_CLADDING_AXIS_Z13".AXIS_POS;
   END_IF;
   "DB16701_OPC_UA_MASTER_MACHINE_1".UNIT_01.MACHINE.POSITIONS.LASER_HEAD.RADIAL_ANGLE := "M_ONE" AND "DB6690_UNIT_1_STA_3_ANGULAR_LOCATOR".CYL.FULL_ADVANCED;
   "DB16701_OPC_UA_MASTER_MACHINE_1".UNIT_01.MACHINE.POSITIONS.LASER_HEAD.TANGENTIAL_ANGLE := "M_ONE" AND "DB6691_UNIT_1_STA_3_AXIAL_LOCATOR".CYL.FULL_ADVANCED;
END_REGION

REGION Network 13: UNIT 01 MACHINE SPEED
   RUNG wire#powerrail
      Contact( "M_ONE" )
      wire#w1
      Move(in := "DB2401_DBB_DEFINE".DBR_1272, out1 => "DB16701_OPC_UA_MASTER_MACHINE_1".UNIT_01.MACHINE.SPEED.X13)
   END_RUNG
   RUNG wire#w1
      Move(in := "DB2401_DBB_DEFINE".DBR_1292, out1 => "DB16701_OPC_UA_MASTER_MACHINE_1".UNIT_01.MACHINE.SPEED.C13)
   END_RUNG
   RUNG wire#w1
      Move(in := "DB2401_DBB_DEFINE".DBR_1300, out1 => "DB16701_OPC_UA_MASTER_MACHINE_1".UNIT_01.MACHINE.SPEED.PROCESS_SETPOINT)
   END_RUNG
   // the same network as SCL:
   IF "M_ONE" THEN
       "DB16701_OPC_UA_MASTER_MACHINE_1".UNIT_01.MACHINE.SPEED.X13 := "DB2401_DBB_DEFINE".DBR_1272;
       "DB16701_OPC_UA_MASTER_MACHINE_1".UNIT_01.MACHINE.SPEED.C13 := "DB2401_DBB_DEFINE".DBR_1292;
       "DB16701_OPC_UA_MASTER_MACHINE_1".UNIT_01.MACHINE.SPEED.PROCESS_SETPOINT := "DB2401_DBB_DEFINE".DBR_1300;
   END_IF;
END_REGION

REGION Network 14: UNIT 01 MACHINE NOZZLE SHIELD GAS FLOW
   RUNG wire#powerrail
      Contact( "M_ONE" )
      Move(in := "DB1511_PROTECTION_GAS_VALVE_UNIT_1".FLOW_VALUE, out1 => "DB16701_OPC_UA_MASTER_MACHINE_1".UNIT_01.MACHINE.NOZZLE.SHIELD_GAS_FLOW)
   END_RUNG
   // the same network as SCL:
   IF "M_ONE" THEN
       "DB16701_OPC_UA_MASTER_MACHINE_1".UNIT_01.MACHINE.NOZZLE.SHIELD_GAS_FLOW := "DB1511_PROTECTION_GAS_VALVE_UNIT_1".FLOW_VALUE;
   END_IF;
END_REGION

REGION Network 15: UNIT 01 PROCCESS
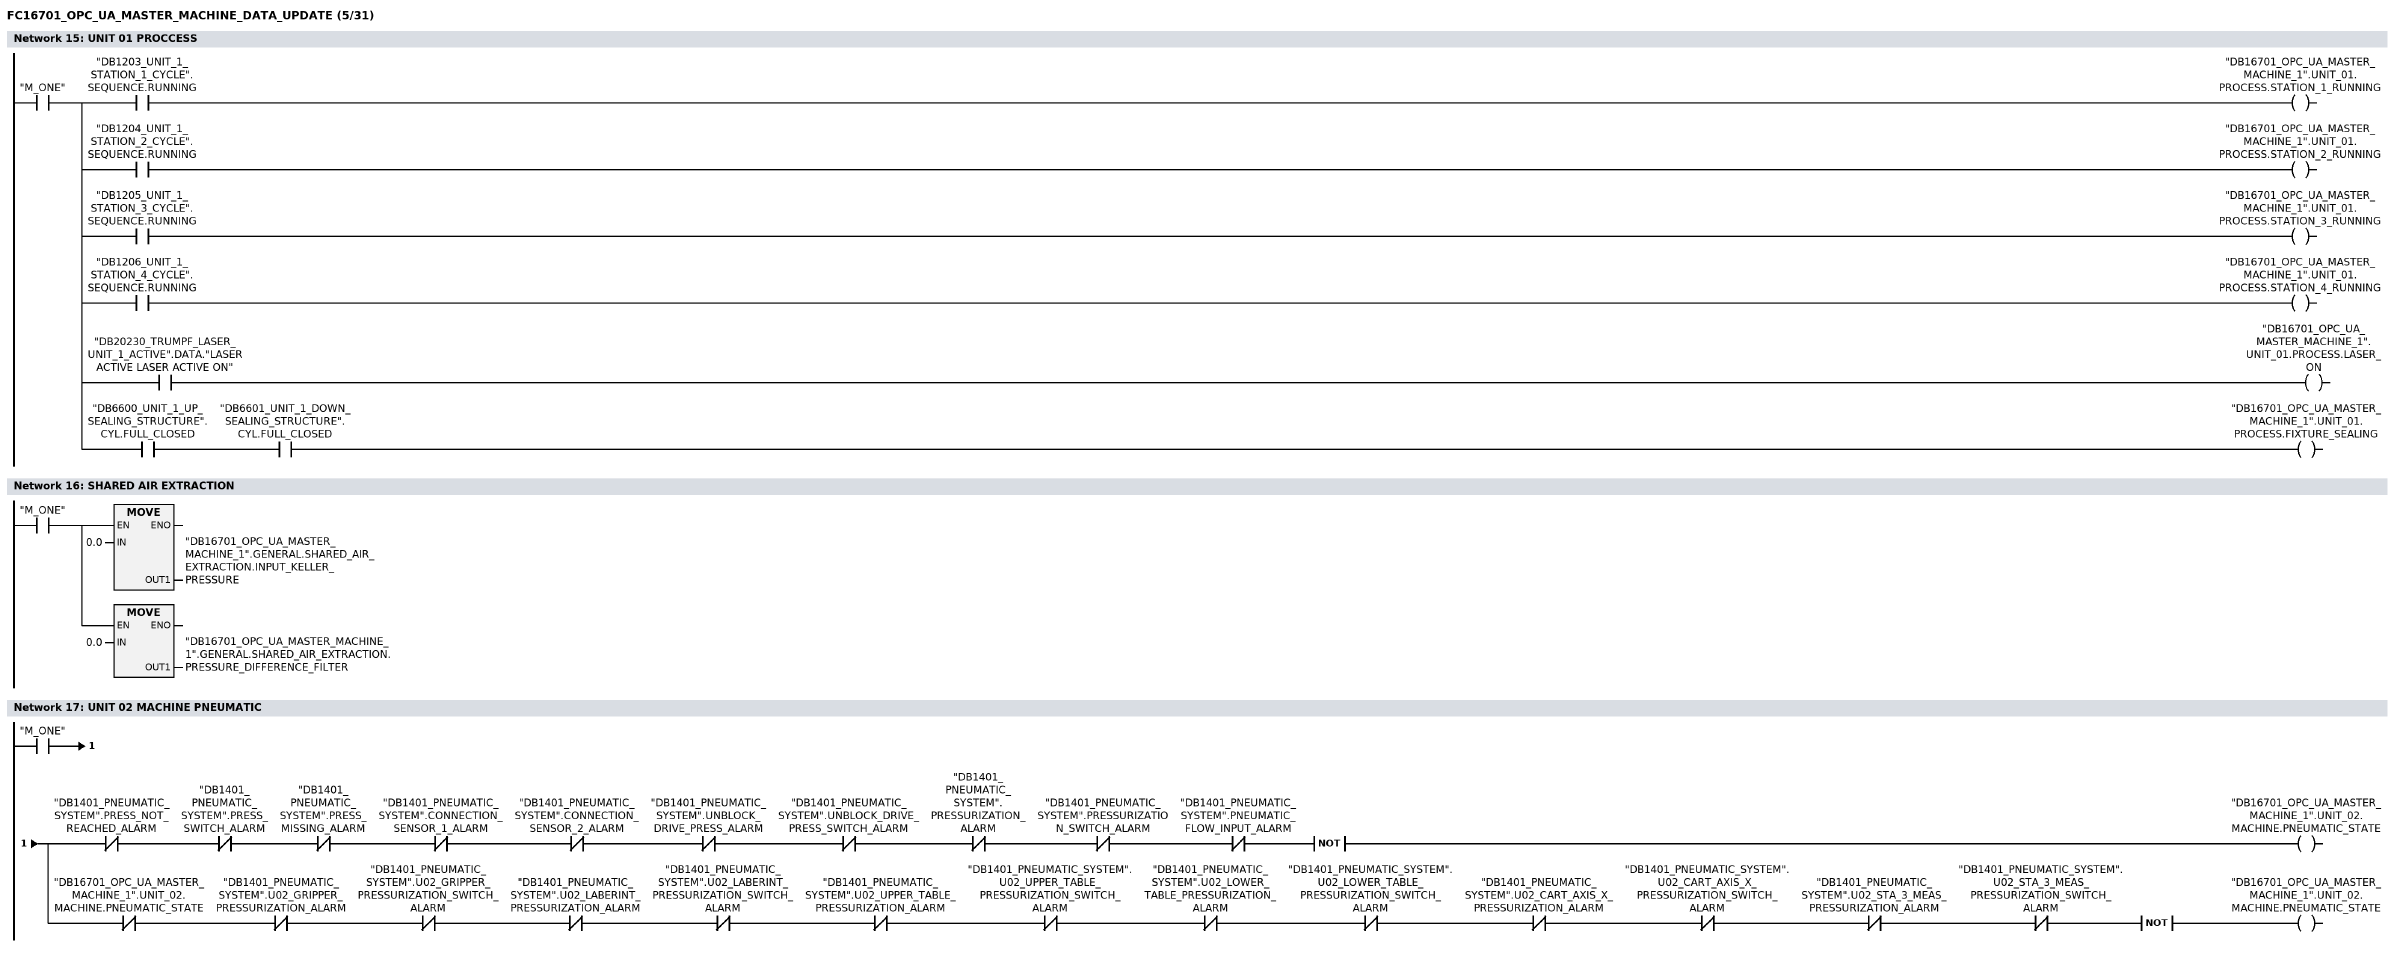
   RUNG wire#powerrail
      Contact( "M_ONE" )
      wire#w1
      Contact( "DB1203_UNIT_1_STATION_1_CYCLE".SEQUENCE.RUNNING )
      Coil( "DB16701_OPC_UA_MASTER_MACHINE_1".UNIT_01.PROCESS.STATION_1_RUNNING )
   END_RUNG
   RUNG wire#w1
      Contact( "DB1204_UNIT_1_STATION_2_CYCLE".SEQUENCE.RUNNING )
      Coil( "DB16701_OPC_UA_MASTER_MACHINE_1".UNIT_01.PROCESS.STATION_2_RUNNING )
   END_RUNG
   RUNG wire#w1
      Contact( "DB1205_UNIT_1_STATION_3_CYCLE".SEQUENCE.RUNNING )
      Coil( "DB16701_OPC_UA_MASTER_MACHINE_1".UNIT_01.PROCESS.STATION_3_RUNNING )
   END_RUNG
   RUNG wire#w1
      Contact( "DB1206_UNIT_1_STATION_4_CYCLE".SEQUENCE.RUNNING )
      Coil( "DB16701_OPC_UA_MASTER_MACHINE_1".UNIT_01.PROCESS.STATION_4_RUNNING )
   END_RUNG
   RUNG wire#w1
      Contact( "DB20230_TRUMPF_LASER_UNIT_1_ACTIVE".DATA."LASER ACTIVE LASER ACTIVE ON" )
      Coil( "DB16701_OPC_UA_MASTER_MACHINE_1".UNIT_01.PROCESS.LASER_ON )
   END_RUNG
   RUNG wire#w1
      Contact( "DB6600_UNIT_1_UP_SEALING_STRUCTURE".CYL.FULL_CLOSED )
      Contact( "DB6601_UNIT_1_DOWN_SEALING_STRUCTURE".CYL.FULL_CLOSED )
      Coil( "DB16701_OPC_UA_MASTER_MACHINE_1".UNIT_01.PROCESS.FIXTURE_SEALING )
   END_RUNG
   // the same network as SCL:
   "DB16701_OPC_UA_MASTER_MACHINE_1".UNIT_01.PROCESS.STATION_1_RUNNING := "M_ONE" AND "DB1203_UNIT_1_STATION_1_CYCLE".SEQUENCE.RUNNING;
   "DB16701_OPC_UA_MASTER_MACHINE_1".UNIT_01.PROCESS.STATION_2_RUNNING := "M_ONE" AND "DB1204_UNIT_1_STATION_2_CYCLE".SEQUENCE.RUNNING;
   "DB16701_OPC_UA_MASTER_MACHINE_1".UNIT_01.PROCESS.STATION_3_RUNNING := "M_ONE" AND "DB1205_UNIT_1_STATION_3_CYCLE".SEQUENCE.RUNNING;
   "DB16701_OPC_UA_MASTER_MACHINE_1".UNIT_01.PROCESS.STATION_4_RUNNING := "M_ONE" AND "DB1206_UNIT_1_STATION_4_CYCLE".SEQUENCE.RUNNING;
   "DB16701_OPC_UA_MASTER_MACHINE_1".UNIT_01.PROCESS.LASER_ON := "M_ONE" AND "DB20230_TRUMPF_LASER_UNIT_1_ACTIVE".DATA."LASER ACTIVE LASER ACTIVE ON";
   "DB16701_OPC_UA_MASTER_MACHINE_1".UNIT_01.PROCESS.FIXTURE_SEALING := "M_ONE" AND "DB6600_UNIT_1_UP_SEALING_STRUCTURE".CYL.FULL_CLOSED AND "DB6601_UNIT_1_DOWN_SEALING_STRUCTURE".CYL.FULL_CLOSED;
END_REGION

REGION Network 16: SHARED AIR EXTRACTION
   RUNG wire#powerrail
      Contact( "M_ONE" )
      wire#w1
      Move(in := 0.0, out1 => "DB16701_OPC_UA_MASTER_MACHINE_1".GENERAL.SHARED_AIR_EXTRACTION.INPUT_KELLER_PRESSURE)
   END_RUNG
   RUNG wire#w1
      Move(in := 0.0, out1 => "DB16701_OPC_UA_MASTER_MACHINE_1".GENERAL.SHARED_AIR_EXTRACTION.PRESSURE_DIFFERENCE_FILTER)
   END_RUNG
   // the same network as SCL:
   IF "M_ONE" THEN
       "DB16701_OPC_UA_MASTER_MACHINE_1".GENERAL.SHARED_AIR_EXTRACTION.INPUT_KELLER_PRESSURE := 0.0;
       "DB16701_OPC_UA_MASTER_MACHINE_1".GENERAL.SHARED_AIR_EXTRACTION.PRESSURE_DIFFERENCE_FILTER := 0.0;
   END_IF;
END_REGION

REGION Network 17: UNIT 02 MACHINE PNEUMATIC
   RUNG wire#powerrail
      Contact( "M_ONE" )
      wire#w1
      I_Contact( "DB1401_PNEUMATIC_SYSTEM".PRESS_NOT_REACHED_ALARM )
      I_Contact( "DB1401_PNEUMATIC_SYSTEM".PRESS_SWITCH_ALARM )
      I_Contact( "DB1401_PNEUMATIC_SYSTEM".PRESS_MISSING_ALARM )
      I_Contact( "DB1401_PNEUMATIC_SYSTEM".CONNECTION_SENSOR_1_ALARM )
      I_Contact( "DB1401_PNEUMATIC_SYSTEM".CONNECTION_SENSOR_2_ALARM )
      I_Contact( "DB1401_PNEUMATIC_SYSTEM".UNBLOCK_DRIVE_PRESS_ALARM )
      I_Contact( "DB1401_PNEUMATIC_SYSTEM".UNBLOCK_DRIVE_PRESS_SWITCH_ALARM )
      I_Contact( "DB1401_PNEUMATIC_SYSTEM".PRESSURIZATION_ALARM )
      I_Contact( "DB1401_PNEUMATIC_SYSTEM".PRESSURIZATION_SWITCH_ALARM )
      I_Contact( "DB1401_PNEUMATIC_SYSTEM".PNEUMATIC_FLOW_INPUT_ALARM )
      Not()
      Coil( "DB16701_OPC_UA_MASTER_MACHINE_1".UNIT_02.MACHINE.PNEUMATIC_STATE )
   END_RUNG
   RUNG wire#w1
      I_Contact( "DB16701_OPC_UA_MASTER_MACHINE_1".UNIT_02.MACHINE.PNEUMATIC_STATE )
      I_Contact( "DB1401_PNEUMATIC_SYSTEM".U02_GRIPPER_PRESSURIZATION_ALARM )
      I_Contact( "DB1401_PNEUMATIC_SYSTEM".U02_GRIPPER_PRESSURIZATION_SWITCH_ALARM )
      I_Contact( "DB1401_PNEUMATIC_SYSTEM".U02_LABERINT_PRESSURIZATION_ALARM )
      I_Contact( "DB1401_PNEUMATIC_SYSTEM".U02_LABERINT_PRESSURIZATION_SWITCH_ALARM )
      I_Contact( "DB1401_PNEUMATIC_SYSTEM".U02_UPPER_TABLE_PRESSURIZATION_ALARM )
      I_Contact( "DB1401_PNEUMATIC_SYSTEM".U02_UPPER_TABLE_PRESSURIZATION_SWITCH_ALARM )
      I_Contact( "DB1401_PNEUMATIC_SYSTEM".U02_LOWER_TABLE_PRESSURIZATION_ALARM )
      I_Contact( "DB1401_PNEUMATIC_SYSTEM".U02_LOWER_TABLE_PRESSURIZATION_SWITCH_ALARM )
      I_Contact( "DB1401_PNEUMATIC_SYSTEM".U02_CART_AXIS_X_PRESSURIZATION_ALARM )
      I_Contact( "DB1401_PNEUMATIC_SYSTEM".U02_CART_AXIS_X_PRESSURIZATION_SWITCH_ALARM )
      I_Contact( "DB1401_PNEUMATIC_SYSTEM".U02_STA_3_MEAS_PRESSURIZATION_ALARM )
      I_Contact( "DB1401_PNEUMATIC_SYSTEM".U02_STA_3_MEAS_PRESSURIZATION_SWITCH_ALARM )
      Not()
      Coil( "DB16701_OPC_UA_MASTER_MACHINE_1".UNIT_02.MACHINE.PNEUMATIC_STATE )
   END_RUNG
   // the same network as SCL:
   "DB16701_OPC_UA_MASTER_MACHINE_1".UNIT_02.MACHINE.PNEUMATIC_STATE := NOT ("M_ONE" AND NOT "DB1401_PNEUMATIC_SYSTEM".PRESS_NOT_REACHED_ALARM AND NOT "DB1401_PNEUMATIC_SYSTEM".PRESS_SWITCH_ALARM AND NOT "DB1401_PNEUMATIC_SYSTEM".PRESS_MISSING_ALARM AND NOT "DB1401_PNEUMATIC_SYSTEM".CONNECTION_SENSOR_1_ALARM AND NOT "DB1401_PNEUMATIC_SYSTEM".CONNECTION_SENSOR_2_ALARM AND NOT "DB1401_PNEUMATIC_SYSTEM".UNBLOCK_DRIVE_PRESS_ALARM AND NOT "DB1401_PNEUMATIC_SYSTEM".UNBLOCK_DRIVE_PRESS_SWITCH_ALARM AND NOT "DB1401_PNEUMATIC_SYSTEM".PRESSURIZATION_ALARM AND NOT "DB1401_PNEUMATIC_SYSTEM".PRESSURIZATION_SWITCH_ALARM AND NOT "DB1401_PNEUMATIC_SYSTEM".PNEUMATIC_FLOW_INPUT_ALARM);
   "DB16701_OPC_UA_MASTER_MACHINE_1".UNIT_02.MACHINE.PNEUMATIC_STATE := NOT ("M_ONE" AND NOT "DB16701_OPC_UA_MASTER_MACHINE_1".UNIT_02.MACHINE.PNEUMATIC_STATE AND NOT "DB1401_PNEUMATIC_SYSTEM".U02_GRIPPER_PRESSURIZATION_ALARM AND NOT "DB1401_PNEUMATIC_SYSTEM".U02_GRIPPER_PRESSURIZATION_SWITCH_ALARM AND NOT "DB1401_PNEUMATIC_SYSTEM".U02_LABERINT_PRESSURIZATION_ALARM AND NOT "DB1401_PNEUMATIC_SYSTEM".U02_LABERINT_PRESSURIZATION_SWITCH_ALARM AND NOT "DB1401_PNEUMATIC_SYSTEM".U02_UPPER_TABLE_PRESSURIZATION_ALARM AND NOT "DB1401_PNEUMATIC_SYSTEM".U02_UPPER_TABLE_PRESSURIZATION_SWITCH_ALARM AND NOT "DB1401_PNEUMATIC_SYSTEM".U02_LOWER_TABLE_PRESSURIZATION_ALARM AND NOT "DB1401_PNEUMATIC_SYSTEM".U02_LOWER_TABLE_PRESSURIZATION_SWITCH_ALARM AND NOT "DB1401_PNEUMATIC_SYSTEM".U02_CART_AXIS_X_PRESSURIZATION_ALARM AND NOT "DB1401_PNEUMATIC_SYSTEM".U02_CART_AXIS_X_PRESSURIZATION_SWITCH_ALARM AND NOT "DB1401_PNEUMATIC_SYSTEM".U02_STA_3_MEAS_PRESSURIZATION_ALARM AND NOT "DB1401_PNEUMATIC_SYSTEM".U02_STA_3_MEAS_PRESSURIZATION_SWITCH_ALARM);
END_REGION

REGION Network 18: UNIT 02 MACHINE TEMPERATURE
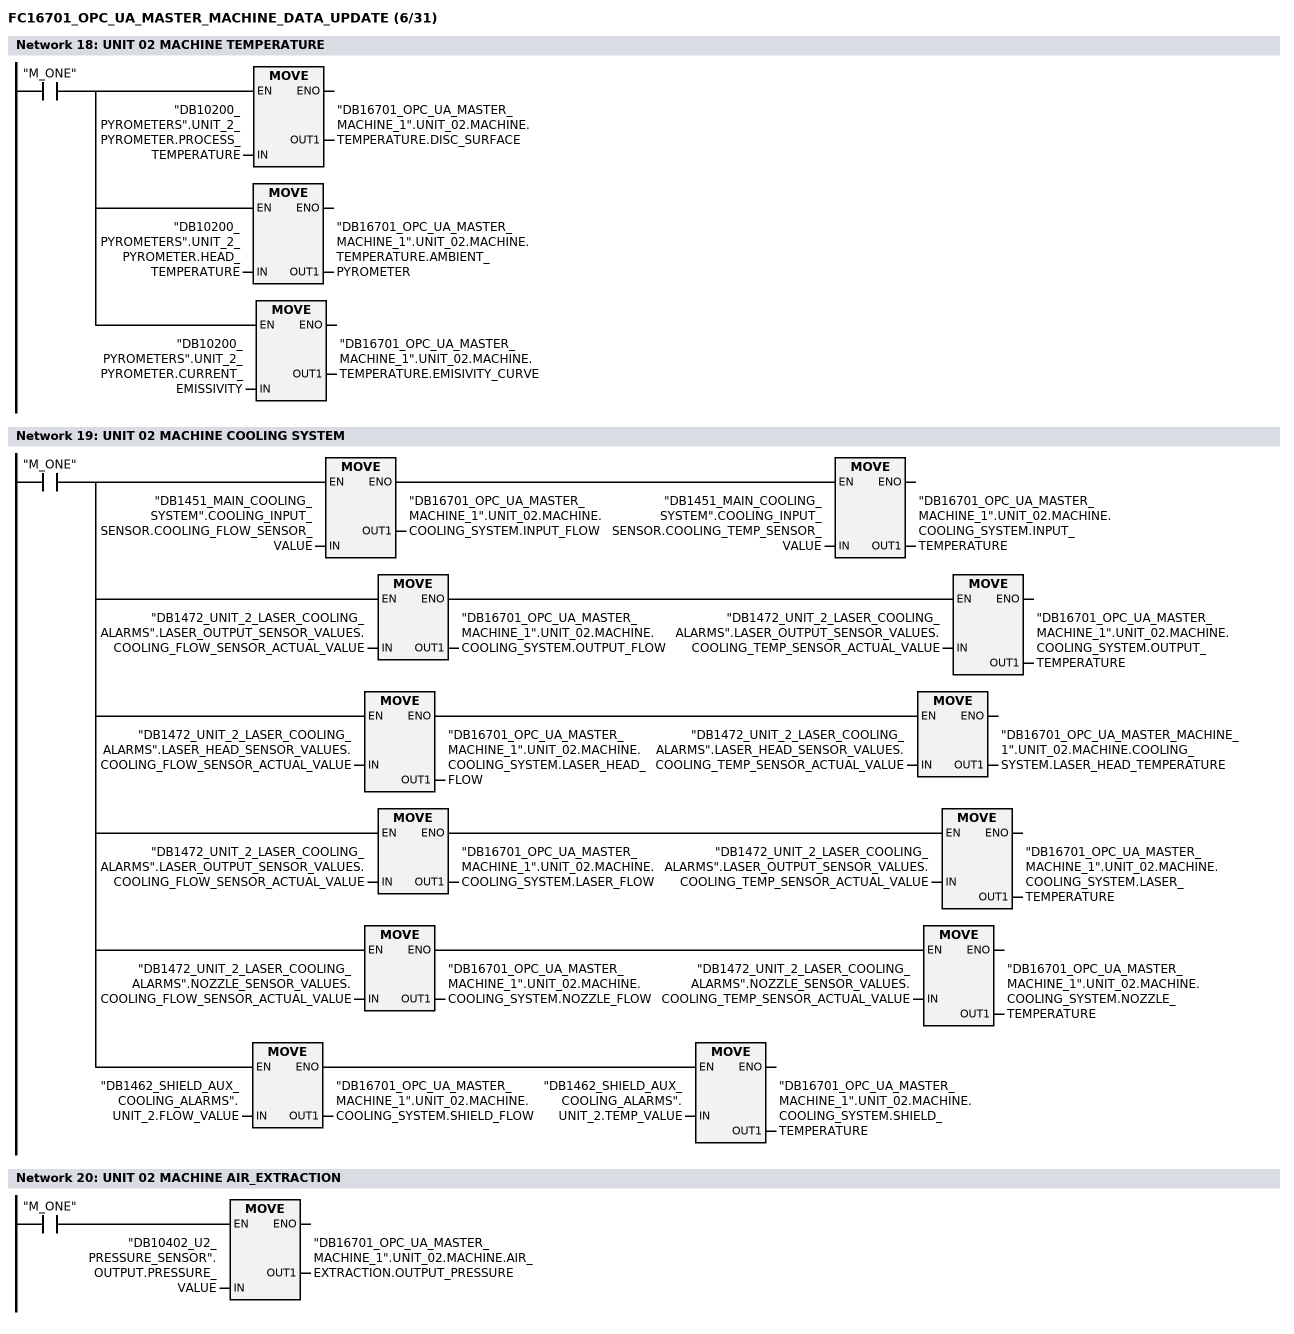
   RUNG wire#powerrail
      Contact( "M_ONE" )
      wire#w1
      Move(in := "DB10200_PYROMETERS".UNIT_2_PYROMETER.PROCESS_TEMPERATURE, out1 => "DB16701_OPC_UA_MASTER_MACHINE_1".UNIT_02.MACHINE.TEMPERATURE.DISC_SURFACE)
   END_RUNG
   RUNG wire#w1
      Move(in := "DB10200_PYROMETERS".UNIT_2_PYROMETER.HEAD_TEMPERATURE, out1 => "DB16701_OPC_UA_MASTER_MACHINE_1".UNIT_02.MACHINE.TEMPERATURE.AMBIENT_PYROMETER)
   END_RUNG
   RUNG wire#w1
      Move(in := "DB10200_PYROMETERS".UNIT_2_PYROMETER.CURRENT_EMISSIVITY, out1 => "DB16701_OPC_UA_MASTER_MACHINE_1".UNIT_02.MACHINE.TEMPERATURE.EMISIVITY_CURVE)
   END_RUNG
   // the same network as SCL:
   IF "M_ONE" THEN
       "DB16701_OPC_UA_MASTER_MACHINE_1".UNIT_02.MACHINE.TEMPERATURE.DISC_SURFACE := "DB10200_PYROMETERS".UNIT_2_PYROMETER.PROCESS_TEMPERATURE;
       "DB16701_OPC_UA_MASTER_MACHINE_1".UNIT_02.MACHINE.TEMPERATURE.AMBIENT_PYROMETER := "DB10200_PYROMETERS".UNIT_2_PYROMETER.HEAD_TEMPERATURE;
       "DB16701_OPC_UA_MASTER_MACHINE_1".UNIT_02.MACHINE.TEMPERATURE.EMISIVITY_CURVE := "DB10200_PYROMETERS".UNIT_2_PYROMETER.CURRENT_EMISSIVITY;
   END_IF;
END_REGION

REGION Network 19: UNIT 02 MACHINE COOLING SYSTEM
   RUNG wire#powerrail
      Contact( "M_ONE" )
      wire#w1
      Move(in := "DB1451_MAIN_COOLING_SYSTEM".COOLING_INPUT_SENSOR.COOLING_FLOW_SENSOR_VALUE, out1 => "DB16701_OPC_UA_MASTER_MACHINE_1".UNIT_02.MACHINE.COOLING_SYSTEM.INPUT_FLOW)
      Move(in := "DB1451_MAIN_COOLING_SYSTEM".COOLING_INPUT_SENSOR.COOLING_TEMP_SENSOR_VALUE, out1 => "DB16701_OPC_UA_MASTER_MACHINE_1".UNIT_02.MACHINE.COOLING_SYSTEM.INPUT_TEMPERATURE)
   END_RUNG
   RUNG wire#w1
      Move(in := "DB1472_UNIT_2_LASER_COOLING_ALARMS".LASER_OUTPUT_SENSOR_VALUES.COOLING_FLOW_SENSOR_ACTUAL_VALUE, out1 => "DB16701_OPC_UA_MASTER_MACHINE_1".UNIT_02.MACHINE.COOLING_SYSTEM.OUTPUT_FLOW)
      Move(in := "DB1472_UNIT_2_LASER_COOLING_ALARMS".LASER_OUTPUT_SENSOR_VALUES.COOLING_TEMP_SENSOR_ACTUAL_VALUE, out1 => "DB16701_OPC_UA_MASTER_MACHINE_1".UNIT_02.MACHINE.COOLING_SYSTEM.OUTPUT_TEMPERATURE)
   END_RUNG
   RUNG wire#w1
      Move(in := "DB1472_UNIT_2_LASER_COOLING_ALARMS".LASER_HEAD_SENSOR_VALUES.COOLING_FLOW_SENSOR_ACTUAL_VALUE, out1 => "DB16701_OPC_UA_MASTER_MACHINE_1".UNIT_02.MACHINE.COOLING_SYSTEM.LASER_HEAD_FLOW)
      Move(in := "DB1472_UNIT_2_LASER_COOLING_ALARMS".LASER_HEAD_SENSOR_VALUES.COOLING_TEMP_SENSOR_ACTUAL_VALUE, out1 => "DB16701_OPC_UA_MASTER_MACHINE_1".UNIT_02.MACHINE.COOLING_SYSTEM.LASER_HEAD_TEMPERATURE)
   END_RUNG
   RUNG wire#w1
      Move(in := "DB1472_UNIT_2_LASER_COOLING_ALARMS".LASER_OUTPUT_SENSOR_VALUES.COOLING_FLOW_SENSOR_ACTUAL_VALUE, out1 => "DB16701_OPC_UA_MASTER_MACHINE_1".UNIT_02.MACHINE.COOLING_SYSTEM.LASER_FLOW)
      Move(in := "DB1472_UNIT_2_LASER_COOLING_ALARMS".LASER_OUTPUT_SENSOR_VALUES.COOLING_TEMP_SENSOR_ACTUAL_VALUE, out1 => "DB16701_OPC_UA_MASTER_MACHINE_1".UNIT_02.MACHINE.COOLING_SYSTEM.LASER_TEMPERATURE)
   END_RUNG
   RUNG wire#w1
      Move(in := "DB1472_UNIT_2_LASER_COOLING_ALARMS".NOZZLE_SENSOR_VALUES.COOLING_FLOW_SENSOR_ACTUAL_VALUE, out1 => "DB16701_OPC_UA_MASTER_MACHINE_1".UNIT_02.MACHINE.COOLING_SYSTEM.NOZZLE_FLOW)
      Move(in := "DB1472_UNIT_2_LASER_COOLING_ALARMS".NOZZLE_SENSOR_VALUES.COOLING_TEMP_SENSOR_ACTUAL_VALUE, out1 => "DB16701_OPC_UA_MASTER_MACHINE_1".UNIT_02.MACHINE.COOLING_SYSTEM.NOZZLE_TEMPERATURE)
   END_RUNG
   RUNG wire#w1
      Move(in := "DB1462_SHIELD_AUX_COOLING_ALARMS".UNIT_2.FLOW_VALUE, out1 => "DB16701_OPC_UA_MASTER_MACHINE_1".UNIT_02.MACHINE.COOLING_SYSTEM.SHIELD_FLOW)
      Move(in := "DB1462_SHIELD_AUX_COOLING_ALARMS".UNIT_2.TEMP_VALUE, out1 => "DB16701_OPC_UA_MASTER_MACHINE_1".UNIT_02.MACHINE.COOLING_SYSTEM.SHIELD_TEMPERATURE)
   END_RUNG
   // the same network as SCL:
   IF "M_ONE" THEN
       "DB16701_OPC_UA_MASTER_MACHINE_1".UNIT_02.MACHINE.COOLING_SYSTEM.INPUT_FLOW := "DB1451_MAIN_COOLING_SYSTEM".COOLING_INPUT_SENSOR.COOLING_FLOW_SENSOR_VALUE;
       "DB16701_OPC_UA_MASTER_MACHINE_1".UNIT_02.MACHINE.COOLING_SYSTEM.INPUT_TEMPERATURE := "DB1451_MAIN_COOLING_SYSTEM".COOLING_INPUT_SENSOR.COOLING_TEMP_SENSOR_VALUE;
       "DB16701_OPC_UA_MASTER_MACHINE_1".UNIT_02.MACHINE.COOLING_SYSTEM.OUTPUT_FLOW := "DB1472_UNIT_2_LASER_COOLING_ALARMS".LASER_OUTPUT_SENSOR_VALUES.COOLING_FLOW_SENSOR_ACTUAL_VALUE;
       "DB16701_OPC_UA_MASTER_MACHINE_1".UNIT_02.MACHINE.COOLING_SYSTEM.OUTPUT_TEMPERATURE := "DB1472_UNIT_2_LASER_COOLING_ALARMS".LASER_OUTPUT_SENSOR_VALUES.COOLING_TEMP_SENSOR_ACTUAL_VALUE;
       "DB16701_OPC_UA_MASTER_MACHINE_1".UNIT_02.MACHINE.COOLING_SYSTEM.LASER_HEAD_FLOW := "DB1472_UNIT_2_LASER_COOLING_ALARMS".LASER_HEAD_SENSOR_VALUES.COOLING_FLOW_SENSOR_ACTUAL_VALUE;
       "DB16701_OPC_UA_MASTER_MACHINE_1".UNIT_02.MACHINE.COOLING_SYSTEM.LASER_HEAD_TEMPERATURE := "DB1472_UNIT_2_LASER_COOLING_ALARMS".LASER_HEAD_SENSOR_VALUES.COOLING_TEMP_SENSOR_ACTUAL_VALUE;
       "DB16701_OPC_UA_MASTER_MACHINE_1".UNIT_02.MACHINE.COOLING_SYSTEM.LASER_FLOW := "DB1472_UNIT_2_LASER_COOLING_ALARMS".LASER_OUTPUT_SENSOR_VALUES.COOLING_FLOW_SENSOR_ACTUAL_VALUE;
       "DB16701_OPC_UA_MASTER_MACHINE_1".UNIT_02.MACHINE.COOLING_SYSTEM.LASER_TEMPERATURE := "DB1472_UNIT_2_LASER_COOLING_ALARMS".LASER_OUTPUT_SENSOR_VALUES.COOLING_TEMP_SENSOR_ACTUAL_VALUE;
       "DB16701_OPC_UA_MASTER_MACHINE_1".UNIT_02.MACHINE.COOLING_SYSTEM.NOZZLE_FLOW := "DB1472_UNIT_2_LASER_COOLING_ALARMS".NOZZLE_SENSOR_VALUES.COOLING_FLOW_SENSOR_ACTUAL_VALUE;
       "DB16701_OPC_UA_MASTER_MACHINE_1".UNIT_02.MACHINE.COOLING_SYSTEM.NOZZLE_TEMPERATURE := "DB1472_UNIT_2_LASER_COOLING_ALARMS".NOZZLE_SENSOR_VALUES.COOLING_TEMP_SENSOR_ACTUAL_VALUE;
       "DB16701_OPC_UA_MASTER_MACHINE_1".UNIT_02.MACHINE.COOLING_SYSTEM.SHIELD_FLOW := "DB1462_SHIELD_AUX_COOLING_ALARMS".UNIT_2.FLOW_VALUE;
       "DB16701_OPC_UA_MASTER_MACHINE_1".UNIT_02.MACHINE.COOLING_SYSTEM.SHIELD_TEMPERATURE := "DB1462_SHIELD_AUX_COOLING_ALARMS".UNIT_2.TEMP_VALUE;
   END_IF;
END_REGION

REGION Network 20: UNIT 02 MACHINE AIR_EXTRACTION
   RUNG wire#powerrail
      Contact( "M_ONE" )
      Move(in := "DB10402_U2_PRESSURE_SENSOR".OUTPUT.PRESSURE_VALUE, out1 => "DB16701_OPC_UA_MASTER_MACHINE_1".UNIT_02.MACHINE.AIR_EXTRACTION.OUTPUT_PRESSURE)
   END_RUNG
   // the same network as SCL:
   IF "M_ONE" THEN
       "DB16701_OPC_UA_MASTER_MACHINE_1".UNIT_02.MACHINE.AIR_EXTRACTION.OUTPUT_PRESSURE := "DB10402_U2_PRESSURE_SENSOR".OUTPUT.PRESSURE_VALUE;
   END_IF;
END_REGION

REGION Network 21: UNIT 02 MACHINE ST3 PRESSURE CONTROL
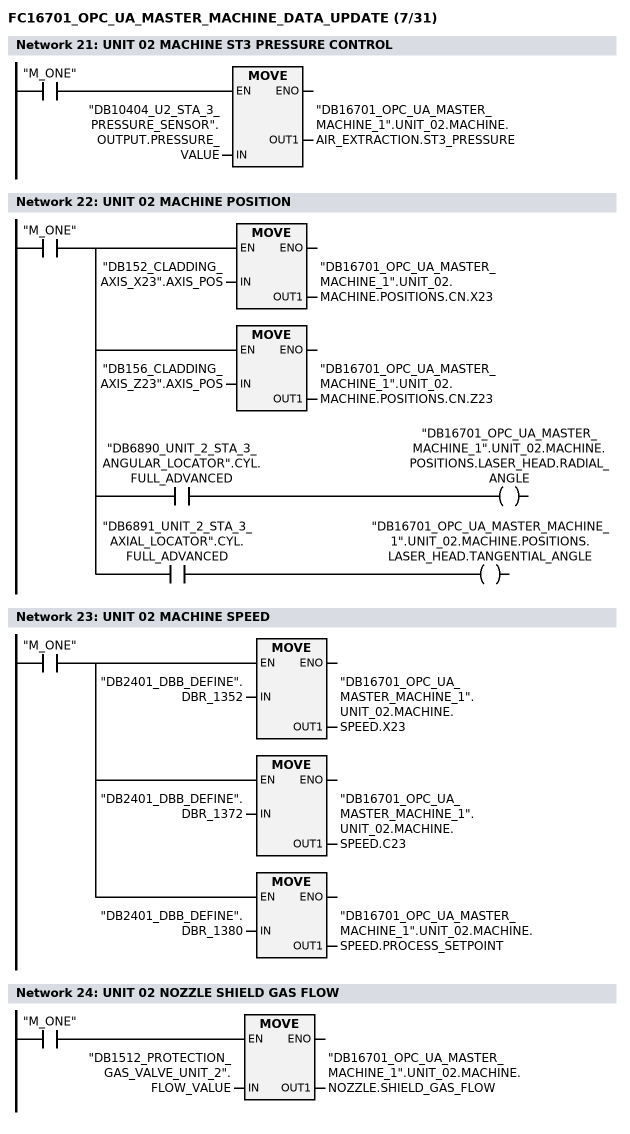
   RUNG wire#powerrail
      Contact( "M_ONE" )
      Move(in := "DB10404_U2_STA_3_PRESSURE_SENSOR".OUTPUT.PRESSURE_VALUE, out1 => "DB16701_OPC_UA_MASTER_MACHINE_1".UNIT_02.MACHINE.AIR_EXTRACTION.ST3_PRESSURE)
   END_RUNG
   // the same network as SCL:
   IF "M_ONE" THEN
       "DB16701_OPC_UA_MASTER_MACHINE_1".UNIT_02.MACHINE.AIR_EXTRACTION.ST3_PRESSURE := "DB10404_U2_STA_3_PRESSURE_SENSOR".OUTPUT.PRESSURE_VALUE;
   END_IF;
END_REGION

REGION Network 22: UNIT 02 MACHINE POSITION
   RUNG wire#powerrail
      Contact( "M_ONE" )
      wire#w1
      Move(in := "DB152_CLADDING_AXIS_X23".AXIS_POS, out1 => "DB16701_OPC_UA_MASTER_MACHINE_1".UNIT_02.MACHINE.POSITIONS.CN.X23)
   END_RUNG
   RUNG wire#w1
      Move(in := "DB156_CLADDING_AXIS_Z23".AXIS_POS, out1 => "DB16701_OPC_UA_MASTER_MACHINE_1".UNIT_02.MACHINE.POSITIONS.CN.Z23)
   END_RUNG
   RUNG wire#w1
      Contact( "DB6890_UNIT_2_STA_3_ANGULAR_LOCATOR".CYL.FULL_ADVANCED )
      Coil( "DB16701_OPC_UA_MASTER_MACHINE_1".UNIT_02.MACHINE.POSITIONS.LASER_HEAD.RADIAL_ANGLE )
   END_RUNG
   RUNG wire#w1
      Contact( "DB6891_UNIT_2_STA_3_AXIAL_LOCATOR".CYL.FULL_ADVANCED )
      Coil( "DB16701_OPC_UA_MASTER_MACHINE_1".UNIT_02.MACHINE.POSITIONS.LASER_HEAD.TANGENTIAL_ANGLE )
   END_RUNG
   // the same network as SCL:
   IF "M_ONE" THEN
       "DB16701_OPC_UA_MASTER_MACHINE_1".UNIT_02.MACHINE.POSITIONS.CN.X23 := "DB152_CLADDING_AXIS_X23".AXIS_POS;
       "DB16701_OPC_UA_MASTER_MACHINE_1".UNIT_02.MACHINE.POSITIONS.CN.Z23 := "DB156_CLADDING_AXIS_Z23".AXIS_POS;
   END_IF;
   "DB16701_OPC_UA_MASTER_MACHINE_1".UNIT_02.MACHINE.POSITIONS.LASER_HEAD.RADIAL_ANGLE := "M_ONE" AND "DB6890_UNIT_2_STA_3_ANGULAR_LOCATOR".CYL.FULL_ADVANCED;
   "DB16701_OPC_UA_MASTER_MACHINE_1".UNIT_02.MACHINE.POSITIONS.LASER_HEAD.TANGENTIAL_ANGLE := "M_ONE" AND "DB6891_UNIT_2_STA_3_AXIAL_LOCATOR".CYL.FULL_ADVANCED;
END_REGION

REGION Network 23: UNIT 02 MACHINE SPEED
   RUNG wire#powerrail
      Contact( "M_ONE" )
      wire#w1
      Move(in := "DB2401_DBB_DEFINE".DBR_1352, out1 => "DB16701_OPC_UA_MASTER_MACHINE_1".UNIT_02.MACHINE.SPEED.X23)
   END_RUNG
   RUNG wire#w1
      Move(in := "DB2401_DBB_DEFINE".DBR_1372, out1 => "DB16701_OPC_UA_MASTER_MACHINE_1".UNIT_02.MACHINE.SPEED.C23)
   END_RUNG
   RUNG wire#w1
      Move(in := "DB2401_DBB_DEFINE".DBR_1380, out1 => "DB16701_OPC_UA_MASTER_MACHINE_1".UNIT_02.MACHINE.SPEED.PROCESS_SETPOINT)
   END_RUNG
   // the same network as SCL:
   IF "M_ONE" THEN
       "DB16701_OPC_UA_MASTER_MACHINE_1".UNIT_02.MACHINE.SPEED.X23 := "DB2401_DBB_DEFINE".DBR_1352;
       "DB16701_OPC_UA_MASTER_MACHINE_1".UNIT_02.MACHINE.SPEED.C23 := "DB2401_DBB_DEFINE".DBR_1372;
       "DB16701_OPC_UA_MASTER_MACHINE_1".UNIT_02.MACHINE.SPEED.PROCESS_SETPOINT := "DB2401_DBB_DEFINE".DBR_1380;
   END_IF;
END_REGION

REGION Network 24: UNIT 02 NOZZLE SHIELD GAS FLOW
   RUNG wire#powerrail
      Contact( "M_ONE" )
      Move(in := "DB1512_PROTECTION_GAS_VALVE_UNIT_2".FLOW_VALUE, out1 => "DB16701_OPC_UA_MASTER_MACHINE_1".UNIT_02.MACHINE.NOZZLE.SHIELD_GAS_FLOW)
   END_RUNG
   // the same network as SCL:
   IF "M_ONE" THEN
       "DB16701_OPC_UA_MASTER_MACHINE_1".UNIT_02.MACHINE.NOZZLE.SHIELD_GAS_FLOW := "DB1512_PROTECTION_GAS_VALVE_UNIT_2".FLOW_VALUE;
   END_IF;
END_REGION

REGION Network 25: UNIT 02 PROCCESS
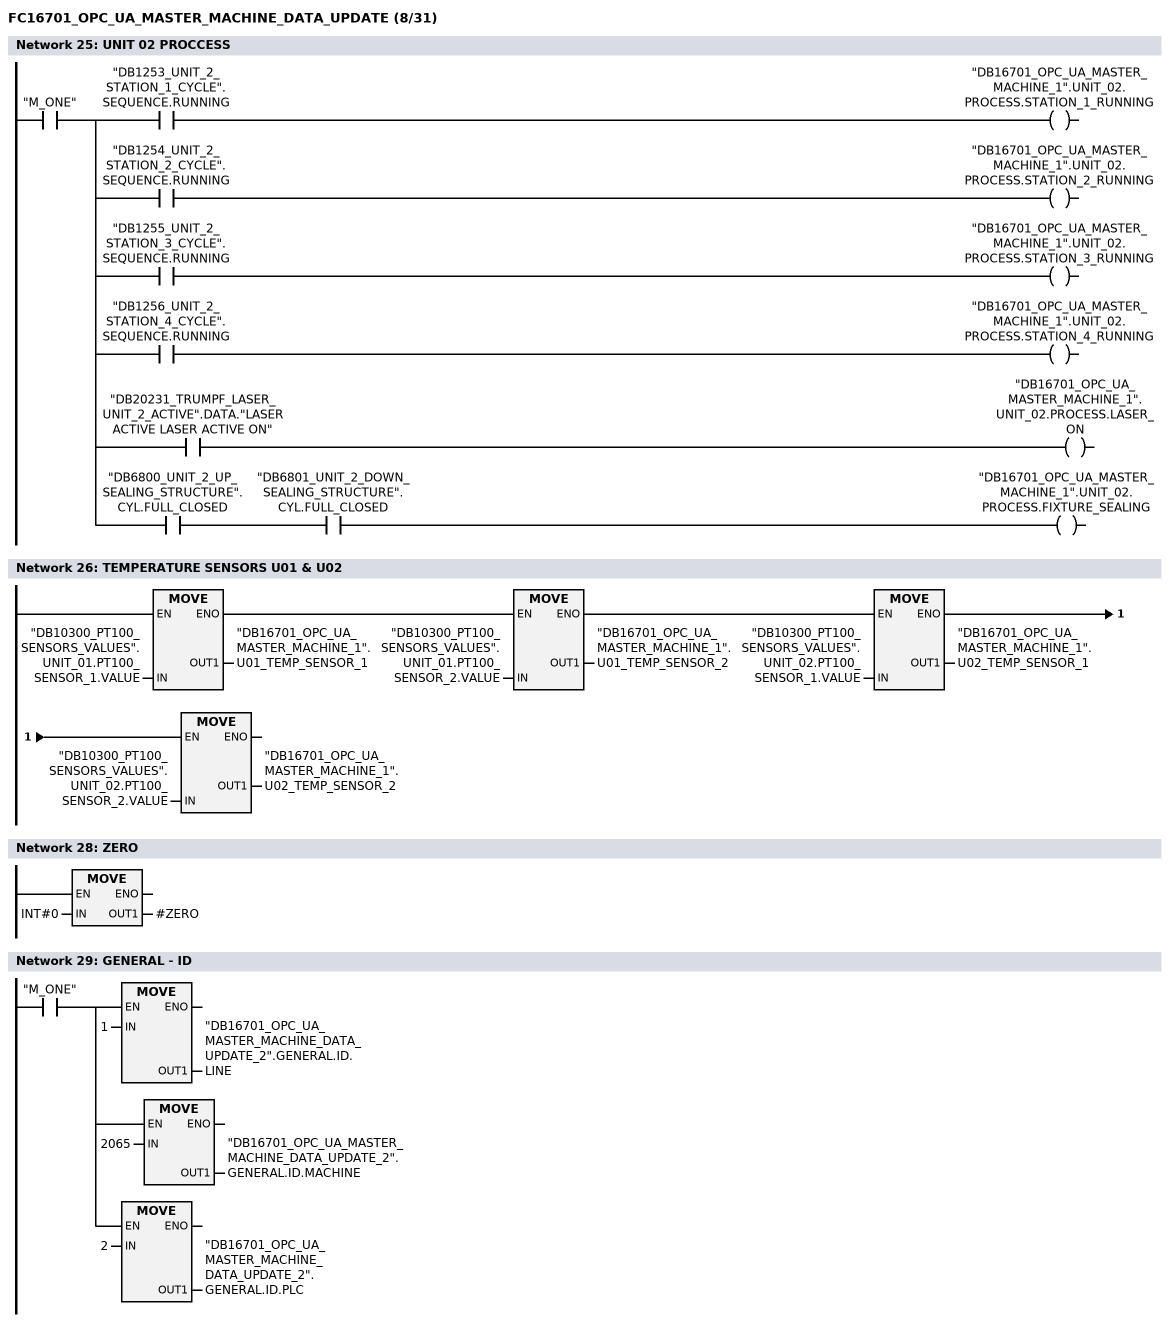
   RUNG wire#powerrail
      Contact( "M_ONE" )
      wire#w1
      Contact( "DB1253_UNIT_2_STATION_1_CYCLE".SEQUENCE.RUNNING )
      Coil( "DB16701_OPC_UA_MASTER_MACHINE_1".UNIT_02.PROCESS.STATION_1_RUNNING )
   END_RUNG
   RUNG wire#w1
      Contact( "DB1254_UNIT_2_STATION_2_CYCLE".SEQUENCE.RUNNING )
      Coil( "DB16701_OPC_UA_MASTER_MACHINE_1".UNIT_02.PROCESS.STATION_2_RUNNING )
   END_RUNG
   RUNG wire#w1
      Contact( "DB1255_UNIT_2_STATION_3_CYCLE".SEQUENCE.RUNNING )
      Coil( "DB16701_OPC_UA_MASTER_MACHINE_1".UNIT_02.PROCESS.STATION_3_RUNNING )
   END_RUNG
   RUNG wire#w1
      Contact( "DB1256_UNIT_2_STATION_4_CYCLE".SEQUENCE.RUNNING )
      Coil( "DB16701_OPC_UA_MASTER_MACHINE_1".UNIT_02.PROCESS.STATION_4_RUNNING )
   END_RUNG
   RUNG wire#w1
      Contact( "DB20231_TRUMPF_LASER_UNIT_2_ACTIVE".DATA."LASER ACTIVE LASER ACTIVE ON" )
      Coil( "DB16701_OPC_UA_MASTER_MACHINE_1".UNIT_02.PROCESS.LASER_ON )
   END_RUNG
   RUNG wire#w1
      Contact( "DB6800_UNIT_2_UP_SEALING_STRUCTURE".CYL.FULL_CLOSED )
      Contact( "DB6801_UNIT_2_DOWN_SEALING_STRUCTURE".CYL.FULL_CLOSED )
      Coil( "DB16701_OPC_UA_MASTER_MACHINE_1".UNIT_02.PROCESS.FIXTURE_SEALING )
   END_RUNG
   // the same network as SCL:
   "DB16701_OPC_UA_MASTER_MACHINE_1".UNIT_02.PROCESS.STATION_1_RUNNING := "M_ONE" AND "DB1253_UNIT_2_STATION_1_CYCLE".SEQUENCE.RUNNING;
   "DB16701_OPC_UA_MASTER_MACHINE_1".UNIT_02.PROCESS.STATION_2_RUNNING := "M_ONE" AND "DB1254_UNIT_2_STATION_2_CYCLE".SEQUENCE.RUNNING;
   "DB16701_OPC_UA_MASTER_MACHINE_1".UNIT_02.PROCESS.STATION_3_RUNNING := "M_ONE" AND "DB1255_UNIT_2_STATION_3_CYCLE".SEQUENCE.RUNNING;
   "DB16701_OPC_UA_MASTER_MACHINE_1".UNIT_02.PROCESS.STATION_4_RUNNING := "M_ONE" AND "DB1256_UNIT_2_STATION_4_CYCLE".SEQUENCE.RUNNING;
   "DB16701_OPC_UA_MASTER_MACHINE_1".UNIT_02.PROCESS.LASER_ON := "M_ONE" AND "DB20231_TRUMPF_LASER_UNIT_2_ACTIVE".DATA."LASER ACTIVE LASER ACTIVE ON";
   "DB16701_OPC_UA_MASTER_MACHINE_1".UNIT_02.PROCESS.FIXTURE_SEALING := "M_ONE" AND "DB6800_UNIT_2_UP_SEALING_STRUCTURE".CYL.FULL_CLOSED AND "DB6801_UNIT_2_DOWN_SEALING_STRUCTURE".CYL.FULL_CLOSED;
END_REGION

REGION Network 26: TEMPERATURE SENSORS U01 & U02
   RUNG wire#powerrail
      Move(in := "DB10300_PT100_SENSORS_VALUES".UNIT_01.PT100_SENSOR_1.VALUE, out1 => "DB16701_OPC_UA_MASTER_MACHINE_1".U01_TEMP_SENSOR_1)
      Move(in := "DB10300_PT100_SENSORS_VALUES".UNIT_01.PT100_SENSOR_2.VALUE, out1 => "DB16701_OPC_UA_MASTER_MACHINE_1".U01_TEMP_SENSOR_2)
      Move(in := "DB10300_PT100_SENSORS_VALUES".UNIT_02.PT100_SENSOR_1.VALUE, out1 => "DB16701_OPC_UA_MASTER_MACHINE_1".U02_TEMP_SENSOR_1)
      Move(in := "DB10300_PT100_SENSORS_VALUES".UNIT_02.PT100_SENSOR_2.VALUE, out1 => "DB16701_OPC_UA_MASTER_MACHINE_1".U02_TEMP_SENSOR_2)
   END_RUNG
   // the same network as SCL:
   "DB16701_OPC_UA_MASTER_MACHINE_1".U01_TEMP_SENSOR_1 := "DB10300_PT100_SENSORS_VALUES".UNIT_01.PT100_SENSOR_1.VALUE;
   "DB16701_OPC_UA_MASTER_MACHINE_1".U01_TEMP_SENSOR_2 := "DB10300_PT100_SENSORS_VALUES".UNIT_01.PT100_SENSOR_2.VALUE;
   "DB16701_OPC_UA_MASTER_MACHINE_1".U02_TEMP_SENSOR_1 := "DB10300_PT100_SENSORS_VALUES".UNIT_02.PT100_SENSOR_1.VALUE;
   "DB16701_OPC_UA_MASTER_MACHINE_1".U02_TEMP_SENSOR_2 := "DB10300_PT100_SENSORS_VALUES".UNIT_02.PT100_SENSOR_2.VALUE;
END_REGION

REGION Network 27: <<<<<<<<<<<<<<<<<<<< OPC UA MASTER MACHINE NEW DB >>>>>>>>>>>>>>>>>>>>
END_REGION

REGION Network 28: ZERO
   RUNG wire#powerrail
      { S7_GenerateENO := "TRUE" } Move(in := INT#0, out1 => #ZERO)
   END_RUNG
   // the same network as SCL:
   #ZERO := INT#0;
END_REGION

REGION Network 29: GENERAL - ID
   RUNG wire#powerrail
      Contact( "M_ONE" )
      wire#w1
      Move(in := 1, out1 => "DB16701_OPC_UA_MASTER_MACHINE_DATA_UPDATE_2".GENERAL.ID.LINE)
   END_RUNG
   RUNG wire#w1
      Move(in := 2065, out1 => "DB16701_OPC_UA_MASTER_MACHINE_DATA_UPDATE_2".GENERAL.ID.MACHINE)
   END_RUNG
   RUNG wire#w1
      Move(in := 2, out1 => "DB16701_OPC_UA_MASTER_MACHINE_DATA_UPDATE_2".GENERAL.ID.PLC)
   END_RUNG
   // the same network as SCL:
   IF "M_ONE" THEN
       "DB16701_OPC_UA_MASTER_MACHINE_DATA_UPDATE_2".GENERAL.ID.LINE := 1;
       "DB16701_OPC_UA_MASTER_MACHINE_DATA_UPDATE_2".GENERAL.ID.MACHINE := 2065;
       "DB16701_OPC_UA_MASTER_MACHINE_DATA_UPDATE_2".GENERAL.ID.PLC := 2;
   END_IF;
END_REGION

REGION Network 30: PARAMETERS - PART TYPE
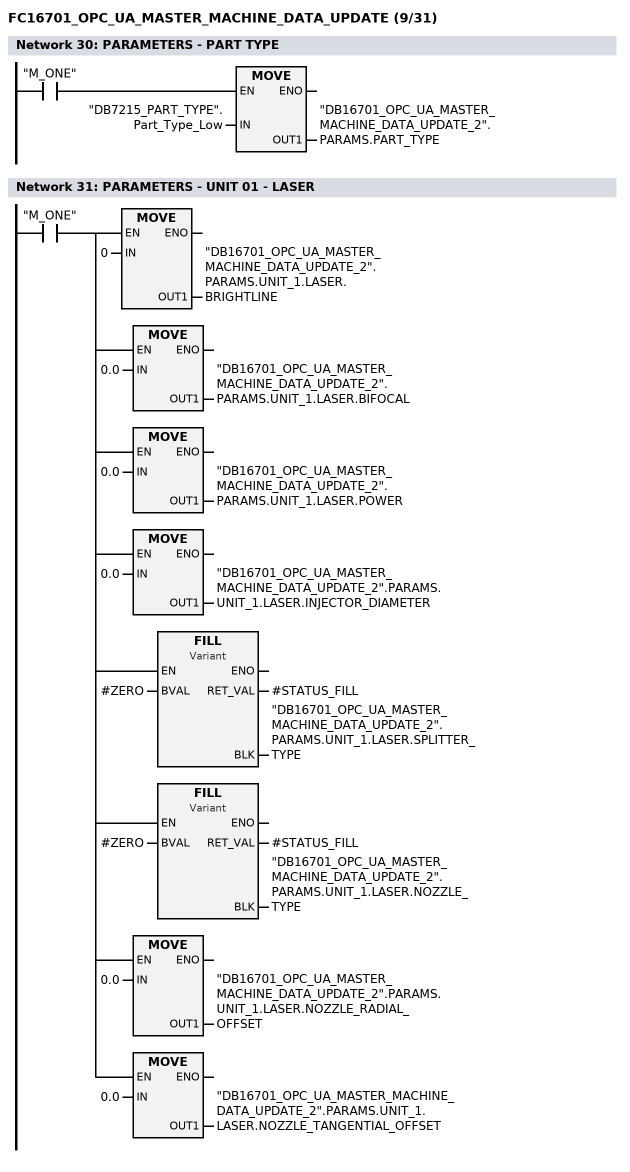
   RUNG wire#powerrail
      Contact( "M_ONE" )
      Move(in := "DB7215_PART_TYPE".Part_Type_Low, out1 => "DB16701_OPC_UA_MASTER_MACHINE_DATA_UPDATE_2".PARAMS.PART_TYPE)
   END_RUNG
   // the same network as SCL:
   IF "M_ONE" THEN
       "DB16701_OPC_UA_MASTER_MACHINE_DATA_UPDATE_2".PARAMS.PART_TYPE := "DB7215_PART_TYPE".Part_Type_Low;
   END_IF;
END_REGION

REGION Network 31: PARAMETERS - UNIT 01 - LASER
   RUNG wire#powerrail
      Contact( "M_ONE" )
      wire#w1
      Move(in := 0, out1 => "DB16701_OPC_UA_MASTER_MACHINE_DATA_UPDATE_2".PARAMS.UNIT_1.LASER.BRIGHTLINE)
   END_RUNG
   RUNG wire#w1
      Move(in := 0.0, out1 => "DB16701_OPC_UA_MASTER_MACHINE_DATA_UPDATE_2".PARAMS.UNIT_1.LASER.BIFOCAL)
   END_RUNG
   RUNG wire#w1
      Move(in := 0.0, out1 => "DB16701_OPC_UA_MASTER_MACHINE_DATA_UPDATE_2".PARAMS.UNIT_1.LASER.POWER)
   END_RUNG
   RUNG wire#w1
      Move(in := 0.0, out1 => "DB16701_OPC_UA_MASTER_MACHINE_DATA_UPDATE_2".PARAMS.UNIT_1.LASER.INJECTOR_DIAMETER)
   END_RUNG
   RUNG wire#w1
      { S7_Templates := "ptr_type := Variant" } FILL(BVAL := #ZERO, RET_VAL => #STATUS_FILL, BLK => "DB16701_OPC_UA_MASTER_MACHINE_DATA_UPDATE_2".PARAMS.UNIT_1.LASER.SPLITTER_TYPE)
   END_RUNG
   RUNG wire#w1
      { S7_Templates := "ptr_type := Variant" } FILL(BVAL := #ZERO, RET_VAL => #STATUS_FILL, BLK => "DB16701_OPC_UA_MASTER_MACHINE_DATA_UPDATE_2".PARAMS.UNIT_1.LASER.NOZZLE_TYPE)
   END_RUNG
   RUNG wire#w1
      Move(in := 0.0, out1 => "DB16701_OPC_UA_MASTER_MACHINE_DATA_UPDATE_2".PARAMS.UNIT_1.LASER.NOZZLE_RADIAL_OFFSET)
   END_RUNG
   RUNG wire#w1
      Move(in := 0.0, out1 => "DB16701_OPC_UA_MASTER_MACHINE_DATA_UPDATE_2".PARAMS.UNIT_1.LASER.NOZZLE_TANGENTIAL_OFFSET)
   END_RUNG
   // the same network as SCL:
   IF "M_ONE" THEN
       "DB16701_OPC_UA_MASTER_MACHINE_DATA_UPDATE_2".PARAMS.UNIT_1.LASER.BRIGHTLINE := 0;
       "DB16701_OPC_UA_MASTER_MACHINE_DATA_UPDATE_2".PARAMS.UNIT_1.LASER.BIFOCAL := 0.0;
       "DB16701_OPC_UA_MASTER_MACHINE_DATA_UPDATE_2".PARAMS.UNIT_1.LASER.POWER := 0.0;
       "DB16701_OPC_UA_MASTER_MACHINE_DATA_UPDATE_2".PARAMS.UNIT_1.LASER.INJECTOR_DIAMETER := 0.0;
   END_IF;
   #_w1 := "M_ONE";
   IF #_w1 THEN
       #STATUS_FILL := FILL(BVAL := #ZERO,
                            BLK => "DB16701_OPC_UA_MASTER_MACHINE_DATA_UPDATE_2".PARAMS.UNIT_1.LASER.SPLITTER_TYPE);
       #STATUS_FILL := FILL(BVAL := #ZERO,
                            BLK => "DB16701_OPC_UA_MASTER_MACHINE_DATA_UPDATE_2".PARAMS.UNIT_1.LASER.NOZZLE_TYPE);
       "DB16701_OPC_UA_MASTER_MACHINE_DATA_UPDATE_2".PARAMS.UNIT_1.LASER.NOZZLE_RADIAL_OFFSET := 0.0;
       "DB16701_OPC_UA_MASTER_MACHINE_DATA_UPDATE_2".PARAMS.UNIT_1.LASER.NOZZLE_TANGENTIAL_OFFSET := 0.0;
   END_IF;
END_REGION

REGION Network 32: PARAMETERS - UNIT 01 - MACHINE
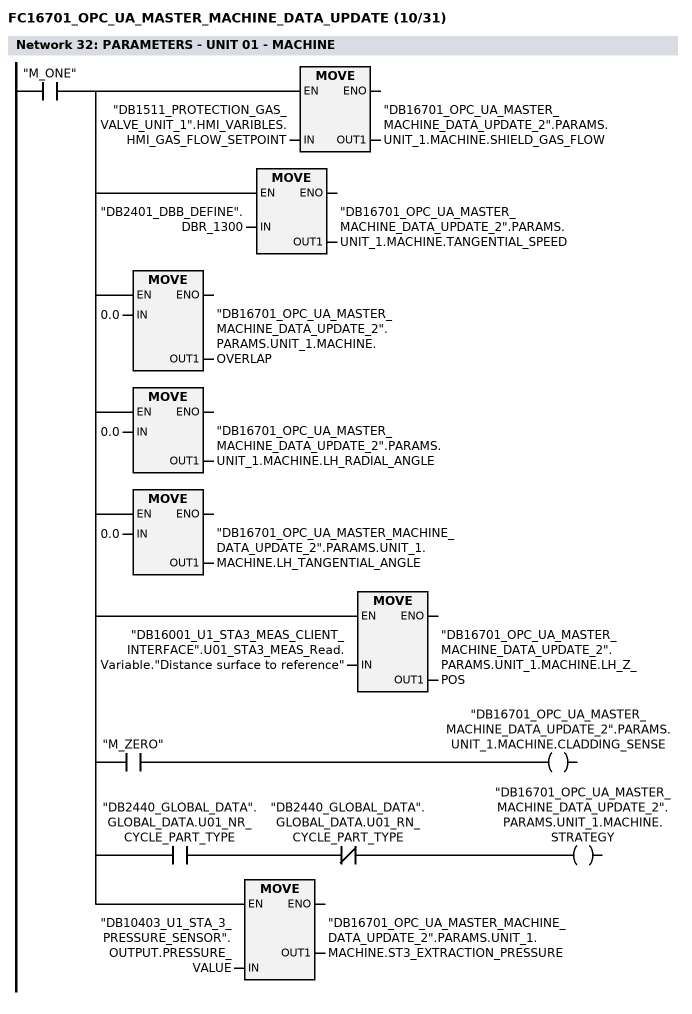
   RUNG wire#powerrail
      Contact( "M_ONE" )
      wire#w1
      Move(in := "DB1511_PROTECTION_GAS_VALVE_UNIT_1".HMI_VARIBLES.HMI_GAS_FLOW_SETPOINT, out1 => "DB16701_OPC_UA_MASTER_MACHINE_DATA_UPDATE_2".PARAMS.UNIT_1.MACHINE.SHIELD_GAS_FLOW)
   END_RUNG
   RUNG wire#w1
      Move(in := "DB2401_DBB_DEFINE".DBR_1300, out1 => "DB16701_OPC_UA_MASTER_MACHINE_DATA_UPDATE_2".PARAMS.UNIT_1.MACHINE.TANGENTIAL_SPEED)
   END_RUNG
   RUNG wire#w1
      Move(in := 0.0, out1 => "DB16701_OPC_UA_MASTER_MACHINE_DATA_UPDATE_2".PARAMS.UNIT_1.MACHINE.OVERLAP)
   END_RUNG
   RUNG wire#w1
      Move(in := 0.0, out1 => "DB16701_OPC_UA_MASTER_MACHINE_DATA_UPDATE_2".PARAMS.UNIT_1.MACHINE.LH_RADIAL_ANGLE)
   END_RUNG
   RUNG wire#w1
      Move(in := 0.0, out1 => "DB16701_OPC_UA_MASTER_MACHINE_DATA_UPDATE_2".PARAMS.UNIT_1.MACHINE.LH_TANGENTIAL_ANGLE)
   END_RUNG
   RUNG wire#w1
      Move(in := "DB16001_U1_STA3_MEAS_CLIENT_INTERFACE".U01_STA3_MEAS_Read.Variable."Distance surface to reference", out1 => "DB16701_OPC_UA_MASTER_MACHINE_DATA_UPDATE_2".PARAMS.UNIT_1.MACHINE.LH_Z_POS)
   END_RUNG
   RUNG wire#w1
      Contact( "M_ZERO" )
      Coil( "DB16701_OPC_UA_MASTER_MACHINE_DATA_UPDATE_2".PARAMS.UNIT_1.MACHINE.CLADDING_SENSE )
   END_RUNG
   RUNG wire#w1
      Contact( "DB2440_GLOBAL_DATA".GLOBAL_DATA.U01_NR_CYCLE_PART_TYPE )
      I_Contact( "DB2440_GLOBAL_DATA".GLOBAL_DATA.U01_RN_CYCLE_PART_TYPE )
      Coil( "DB16701_OPC_UA_MASTER_MACHINE_DATA_UPDATE_2".PARAMS.UNIT_1.MACHINE.STRATEGY )
   END_RUNG
   RUNG wire#w1
      Move(in := "DB10403_U1_STA_3_PRESSURE_SENSOR".OUTPUT.PRESSURE_VALUE, out1 => "DB16701_OPC_UA_MASTER_MACHINE_DATA_UPDATE_2".PARAMS.UNIT_1.MACHINE.ST3_EXTRACTION_PRESSURE)
   END_RUNG
   // the same network as SCL:
   IF "M_ONE" THEN
       "DB16701_OPC_UA_MASTER_MACHINE_DATA_UPDATE_2".PARAMS.UNIT_1.MACHINE.SHIELD_GAS_FLOW := "DB1511_PROTECTION_GAS_VALVE_UNIT_1".HMI_VARIBLES.HMI_GAS_FLOW_SETPOINT;
       "DB16701_OPC_UA_MASTER_MACHINE_DATA_UPDATE_2".PARAMS.UNIT_1.MACHINE.TANGENTIAL_SPEED := "DB2401_DBB_DEFINE".DBR_1300;
       "DB16701_OPC_UA_MASTER_MACHINE_DATA_UPDATE_2".PARAMS.UNIT_1.MACHINE.OVERLAP := 0.0;
       "DB16701_OPC_UA_MASTER_MACHINE_DATA_UPDATE_2".PARAMS.UNIT_1.MACHINE.LH_RADIAL_ANGLE := 0.0;
       "DB16701_OPC_UA_MASTER_MACHINE_DATA_UPDATE_2".PARAMS.UNIT_1.MACHINE.LH_TANGENTIAL_ANGLE := 0.0;
       "DB16701_OPC_UA_MASTER_MACHINE_DATA_UPDATE_2".PARAMS.UNIT_1.MACHINE.LH_Z_POS := "DB16001_U1_STA3_MEAS_CLIENT_INTERFACE".U01_STA3_MEAS_Read.Variable."Distance surface to reference";
   END_IF;
   "DB16701_OPC_UA_MASTER_MACHINE_DATA_UPDATE_2".PARAMS.UNIT_1.MACHINE.CLADDING_SENSE := "M_ONE" AND "M_ZERO";
   "DB16701_OPC_UA_MASTER_MACHINE_DATA_UPDATE_2".PARAMS.UNIT_1.MACHINE.STRATEGY := "M_ONE" AND "DB2440_GLOBAL_DATA".GLOBAL_DATA.U01_NR_CYCLE_PART_TYPE AND NOT "DB2440_GLOBAL_DATA".GLOBAL_DATA.U01_RN_CYCLE_PART_TYPE;
   IF "M_ONE" THEN
       "DB16701_OPC_UA_MASTER_MACHINE_DATA_UPDATE_2".PARAMS.UNIT_1.MACHINE.ST3_EXTRACTION_PRESSURE := "DB10403_U1_STA_3_PRESSURE_SENSOR".OUTPUT.PRESSURE_VALUE;
   END_IF;
END_REGION

REGION Network 33: PARAMETERS - UNIT 02 - LASER
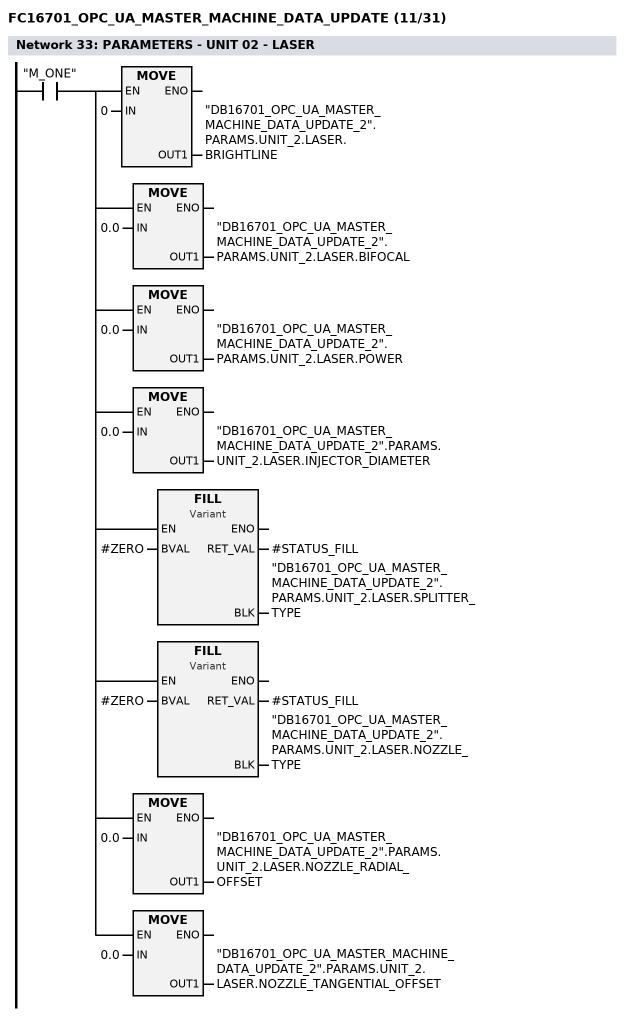
   RUNG wire#powerrail
      Contact( "M_ONE" )
      wire#w1
      Move(in := 0, out1 => "DB16701_OPC_UA_MASTER_MACHINE_DATA_UPDATE_2".PARAMS.UNIT_2.LASER.BRIGHTLINE)
   END_RUNG
   RUNG wire#w1
      Move(in := 0.0, out1 => "DB16701_OPC_UA_MASTER_MACHINE_DATA_UPDATE_2".PARAMS.UNIT_2.LASER.BIFOCAL)
   END_RUNG
   RUNG wire#w1
      Move(in := 0.0, out1 => "DB16701_OPC_UA_MASTER_MACHINE_DATA_UPDATE_2".PARAMS.UNIT_2.LASER.POWER)
   END_RUNG
   RUNG wire#w1
      Move(in := 0.0, out1 => "DB16701_OPC_UA_MASTER_MACHINE_DATA_UPDATE_2".PARAMS.UNIT_2.LASER.INJECTOR_DIAMETER)
   END_RUNG
   RUNG wire#w1
      { S7_Templates := "ptr_type := Variant" } FILL(BVAL := #ZERO, RET_VAL => #STATUS_FILL, BLK => "DB16701_OPC_UA_MASTER_MACHINE_DATA_UPDATE_2".PARAMS.UNIT_2.LASER.SPLITTER_TYPE)
   END_RUNG
   RUNG wire#w1
      { S7_Templates := "ptr_type := Variant" } FILL(BVAL := #ZERO, RET_VAL => #STATUS_FILL, BLK => "DB16701_OPC_UA_MASTER_MACHINE_DATA_UPDATE_2".PARAMS.UNIT_2.LASER.NOZZLE_TYPE)
   END_RUNG
   RUNG wire#w1
      Move(in := 0.0, out1 => "DB16701_OPC_UA_MASTER_MACHINE_DATA_UPDATE_2".PARAMS.UNIT_2.LASER.NOZZLE_RADIAL_OFFSET)
   END_RUNG
   RUNG wire#w1
      Move(in := 0.0, out1 => "DB16701_OPC_UA_MASTER_MACHINE_DATA_UPDATE_2".PARAMS.UNIT_2.LASER.NOZZLE_TANGENTIAL_OFFSET)
   END_RUNG
   // the same network as SCL:
   IF "M_ONE" THEN
       "DB16701_OPC_UA_MASTER_MACHINE_DATA_UPDATE_2".PARAMS.UNIT_2.LASER.BRIGHTLINE := 0;
       "DB16701_OPC_UA_MASTER_MACHINE_DATA_UPDATE_2".PARAMS.UNIT_2.LASER.BIFOCAL := 0.0;
       "DB16701_OPC_UA_MASTER_MACHINE_DATA_UPDATE_2".PARAMS.UNIT_2.LASER.POWER := 0.0;
       "DB16701_OPC_UA_MASTER_MACHINE_DATA_UPDATE_2".PARAMS.UNIT_2.LASER.INJECTOR_DIAMETER := 0.0;
   END_IF;
   #_w1 := "M_ONE";
   IF #_w1 THEN
       #STATUS_FILL := FILL(BVAL := #ZERO,
                            BLK => "DB16701_OPC_UA_MASTER_MACHINE_DATA_UPDATE_2".PARAMS.UNIT_2.LASER.SPLITTER_TYPE);
       #STATUS_FILL := FILL(BVAL := #ZERO,
                            BLK => "DB16701_OPC_UA_MASTER_MACHINE_DATA_UPDATE_2".PARAMS.UNIT_2.LASER.NOZZLE_TYPE);
       "DB16701_OPC_UA_MASTER_MACHINE_DATA_UPDATE_2".PARAMS.UNIT_2.LASER.NOZZLE_RADIAL_OFFSET := 0.0;
       "DB16701_OPC_UA_MASTER_MACHINE_DATA_UPDATE_2".PARAMS.UNIT_2.LASER.NOZZLE_TANGENTIAL_OFFSET := 0.0;
   END_IF;
END_REGION

REGION Network 34: PARAMETERS - UNIT 02 - MACHINE
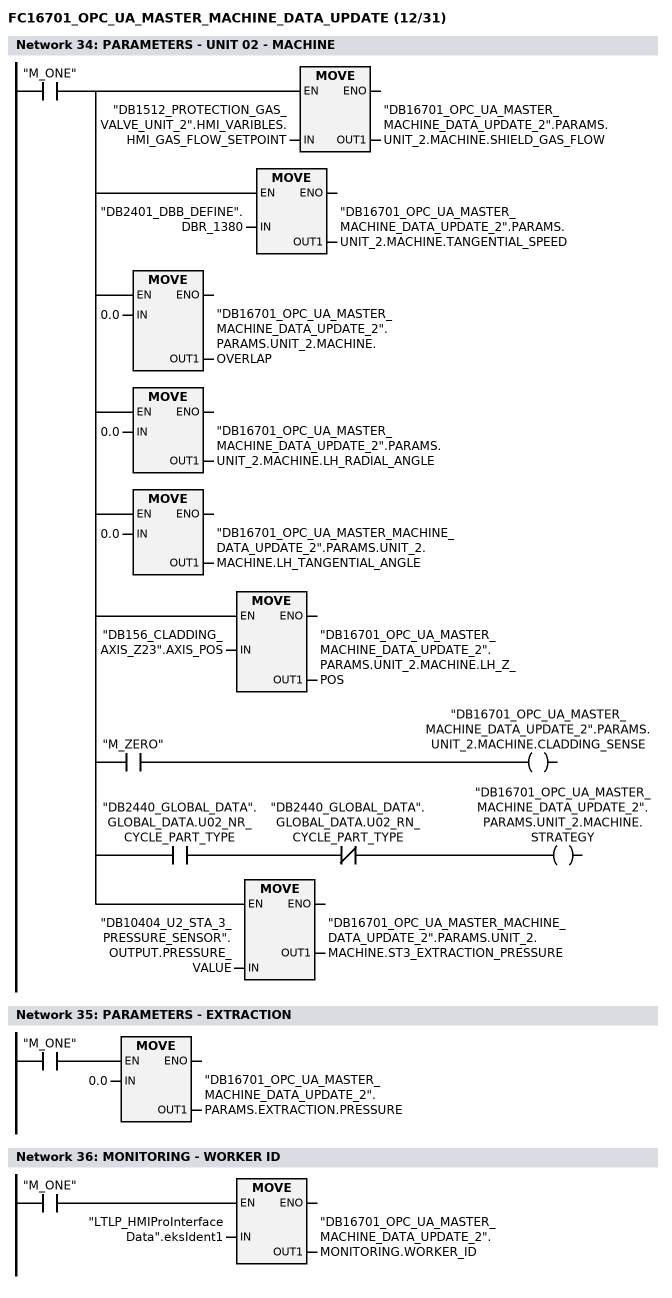
   RUNG wire#powerrail
      Contact( "M_ONE" )
      wire#w1
      Move(in := "DB1512_PROTECTION_GAS_VALVE_UNIT_2".HMI_VARIBLES.HMI_GAS_FLOW_SETPOINT, out1 => "DB16701_OPC_UA_MASTER_MACHINE_DATA_UPDATE_2".PARAMS.UNIT_2.MACHINE.SHIELD_GAS_FLOW)
   END_RUNG
   RUNG wire#w1
      Move(in := "DB2401_DBB_DEFINE".DBR_1380, out1 => "DB16701_OPC_UA_MASTER_MACHINE_DATA_UPDATE_2".PARAMS.UNIT_2.MACHINE.TANGENTIAL_SPEED)
   END_RUNG
   RUNG wire#w1
      Move(in := 0.0, out1 => "DB16701_OPC_UA_MASTER_MACHINE_DATA_UPDATE_2".PARAMS.UNIT_2.MACHINE.OVERLAP)
   END_RUNG
   RUNG wire#w1
      Move(in := 0.0, out1 => "DB16701_OPC_UA_MASTER_MACHINE_DATA_UPDATE_2".PARAMS.UNIT_2.MACHINE.LH_RADIAL_ANGLE)
   END_RUNG
   RUNG wire#w1
      Move(in := 0.0, out1 => "DB16701_OPC_UA_MASTER_MACHINE_DATA_UPDATE_2".PARAMS.UNIT_2.MACHINE.LH_TANGENTIAL_ANGLE)
   END_RUNG
   RUNG wire#w1
      Move(in := "DB156_CLADDING_AXIS_Z23".AXIS_POS, out1 => "DB16701_OPC_UA_MASTER_MACHINE_DATA_UPDATE_2".PARAMS.UNIT_2.MACHINE.LH_Z_POS)
   END_RUNG
   RUNG wire#w1
      Contact( "M_ZERO" )
      Coil( "DB16701_OPC_UA_MASTER_MACHINE_DATA_UPDATE_2".PARAMS.UNIT_2.MACHINE.CLADDING_SENSE )
   END_RUNG
   RUNG wire#w1
      Contact( "DB2440_GLOBAL_DATA".GLOBAL_DATA.U02_NR_CYCLE_PART_TYPE )
      I_Contact( "DB2440_GLOBAL_DATA".GLOBAL_DATA.U02_RN_CYCLE_PART_TYPE )
      Coil( "DB16701_OPC_UA_MASTER_MACHINE_DATA_UPDATE_2".PARAMS.UNIT_2.MACHINE.STRATEGY )
   END_RUNG
   RUNG wire#w1
      Move(in := "DB10404_U2_STA_3_PRESSURE_SENSOR".OUTPUT.PRESSURE_VALUE, out1 => "DB16701_OPC_UA_MASTER_MACHINE_DATA_UPDATE_2".PARAMS.UNIT_2.MACHINE.ST3_EXTRACTION_PRESSURE)
   END_RUNG
   // the same network as SCL:
   IF "M_ONE" THEN
       "DB16701_OPC_UA_MASTER_MACHINE_DATA_UPDATE_2".PARAMS.UNIT_2.MACHINE.SHIELD_GAS_FLOW := "DB1512_PROTECTION_GAS_VALVE_UNIT_2".HMI_VARIBLES.HMI_GAS_FLOW_SETPOINT;
       "DB16701_OPC_UA_MASTER_MACHINE_DATA_UPDATE_2".PARAMS.UNIT_2.MACHINE.TANGENTIAL_SPEED := "DB2401_DBB_DEFINE".DBR_1380;
       "DB16701_OPC_UA_MASTER_MACHINE_DATA_UPDATE_2".PARAMS.UNIT_2.MACHINE.OVERLAP := 0.0;
       "DB16701_OPC_UA_MASTER_MACHINE_DATA_UPDATE_2".PARAMS.UNIT_2.MACHINE.LH_RADIAL_ANGLE := 0.0;
       "DB16701_OPC_UA_MASTER_MACHINE_DATA_UPDATE_2".PARAMS.UNIT_2.MACHINE.LH_TANGENTIAL_ANGLE := 0.0;
       "DB16701_OPC_UA_MASTER_MACHINE_DATA_UPDATE_2".PARAMS.UNIT_2.MACHINE.LH_Z_POS := "DB156_CLADDING_AXIS_Z23".AXIS_POS;
   END_IF;
   "DB16701_OPC_UA_MASTER_MACHINE_DATA_UPDATE_2".PARAMS.UNIT_2.MACHINE.CLADDING_SENSE := "M_ONE" AND "M_ZERO";
   "DB16701_OPC_UA_MASTER_MACHINE_DATA_UPDATE_2".PARAMS.UNIT_2.MACHINE.STRATEGY := "M_ONE" AND "DB2440_GLOBAL_DATA".GLOBAL_DATA.U02_NR_CYCLE_PART_TYPE AND NOT "DB2440_GLOBAL_DATA".GLOBAL_DATA.U02_RN_CYCLE_PART_TYPE;
   IF "M_ONE" THEN
       "DB16701_OPC_UA_MASTER_MACHINE_DATA_UPDATE_2".PARAMS.UNIT_2.MACHINE.ST3_EXTRACTION_PRESSURE := "DB10404_U2_STA_3_PRESSURE_SENSOR".OUTPUT.PRESSURE_VALUE;
   END_IF;
END_REGION

REGION Network 35: PARAMETERS - EXTRACTION
   RUNG wire#powerrail
      Contact( "M_ONE" )
      Move(in := 0.0, out1 => "DB16701_OPC_UA_MASTER_MACHINE_DATA_UPDATE_2".PARAMS.EXTRACTION.PRESSURE)
   END_RUNG
   // the same network as SCL:
   IF "M_ONE" THEN "DB16701_OPC_UA_MASTER_MACHINE_DATA_UPDATE_2".PARAMS.EXTRACTION.PRESSURE := 0.0; END_IF;
END_REGION

REGION Network 36: MONITORING - WORKER ID
   RUNG wire#powerrail
      Contact( "M_ONE" )
      Move(in := "LTLP_HMIProInterfaceData".eksIdent1, out1 => "DB16701_OPC_UA_MASTER_MACHINE_DATA_UPDATE_2".MONITORING.WORKER_ID)
   END_RUNG
   // the same network as SCL:
   IF "M_ONE" THEN
       "DB16701_OPC_UA_MASTER_MACHINE_DATA_UPDATE_2".MONITORING.WORKER_ID := "LTLP_HMIProInterfaceData".eksIdent1;
   END_IF;
END_REGION

REGION Network 37: MONITORING - EXTRACTION
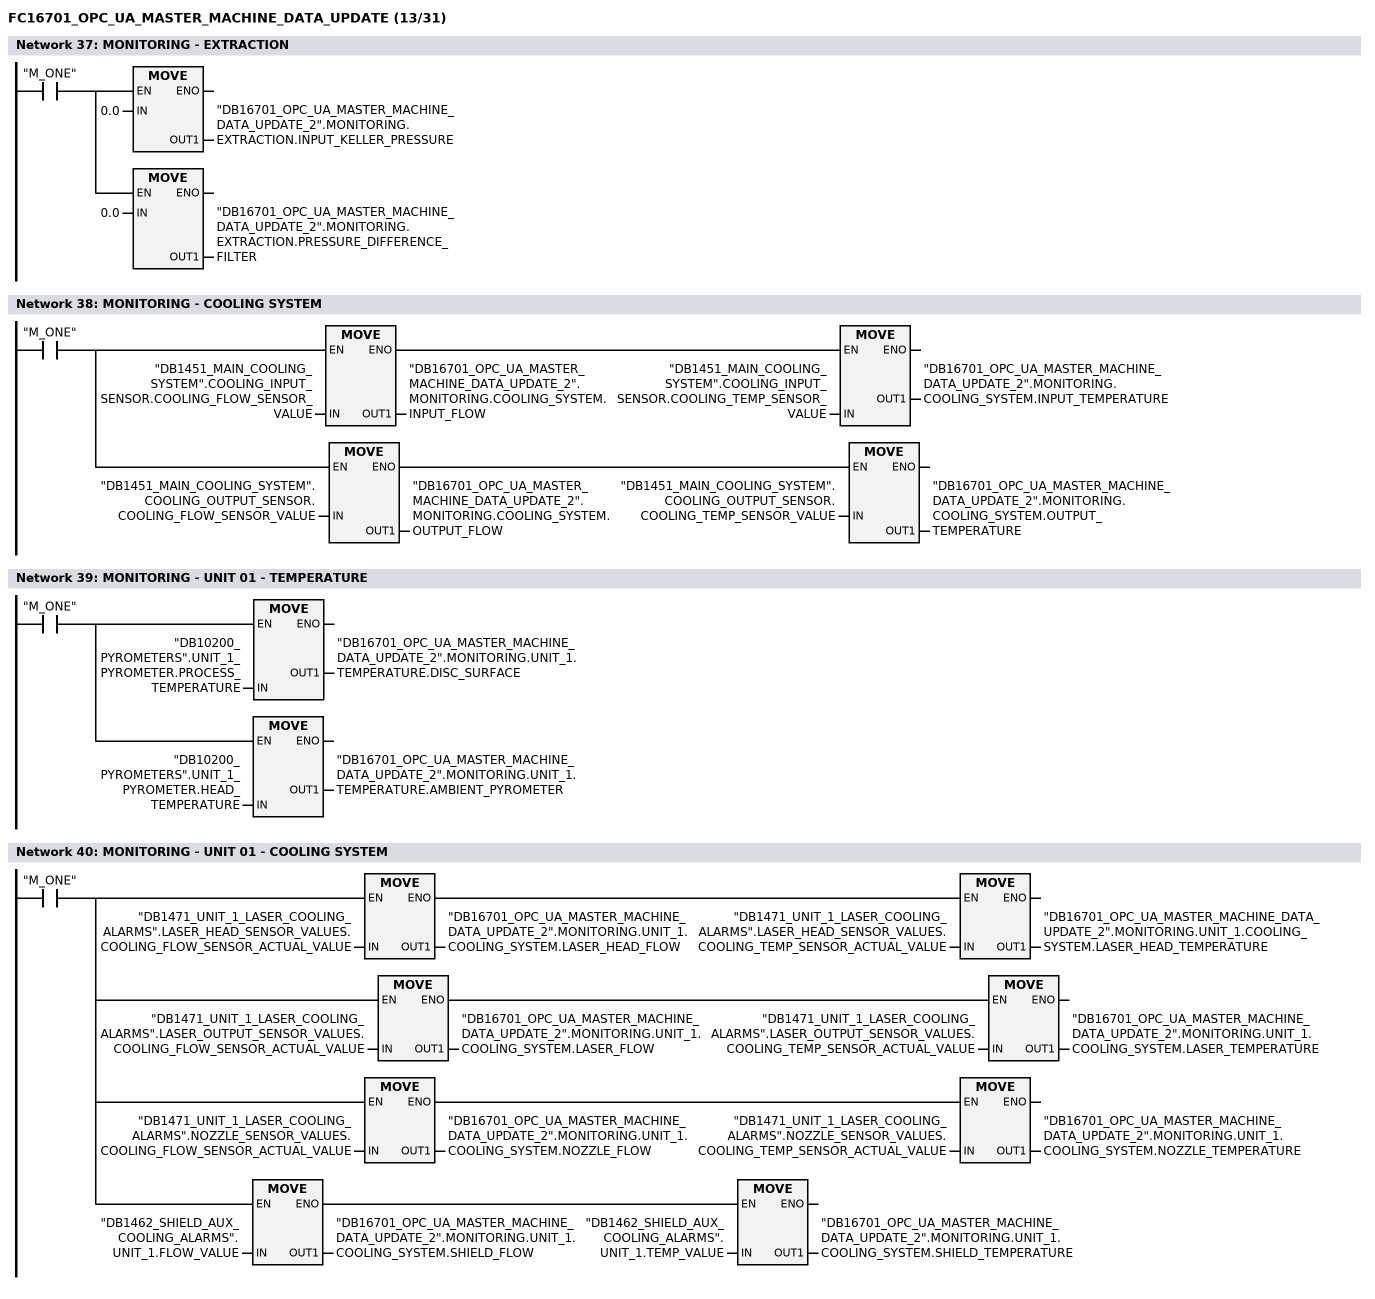
   RUNG wire#powerrail
      Contact( "M_ONE" )
      wire#w1
      Move(in := 0.0, out1 => "DB16701_OPC_UA_MASTER_MACHINE_DATA_UPDATE_2".MONITORING.EXTRACTION.INPUT_KELLER_PRESSURE)
   END_RUNG
   RUNG wire#w1
      Move(in := 0.0, out1 => "DB16701_OPC_UA_MASTER_MACHINE_DATA_UPDATE_2".MONITORING.EXTRACTION.PRESSURE_DIFFERENCE_FILTER)
   END_RUNG
   // the same network as SCL:
   IF "M_ONE" THEN
       "DB16701_OPC_UA_MASTER_MACHINE_DATA_UPDATE_2".MONITORING.EXTRACTION.INPUT_KELLER_PRESSURE := 0.0;
       "DB16701_OPC_UA_MASTER_MACHINE_DATA_UPDATE_2".MONITORING.EXTRACTION.PRESSURE_DIFFERENCE_FILTER := 0.0;
   END_IF;
END_REGION

REGION Network 38: MONITORING - COOLING SYSTEM
   RUNG wire#powerrail
      Contact( "M_ONE" )
      wire#w1
      Move(in := "DB1451_MAIN_COOLING_SYSTEM".COOLING_INPUT_SENSOR.COOLING_FLOW_SENSOR_VALUE, out1 => "DB16701_OPC_UA_MASTER_MACHINE_DATA_UPDATE_2".MONITORING.COOLING_SYSTEM.INPUT_FLOW)
      Move(in := "DB1451_MAIN_COOLING_SYSTEM".COOLING_INPUT_SENSOR.COOLING_TEMP_SENSOR_VALUE, out1 => "DB16701_OPC_UA_MASTER_MACHINE_DATA_UPDATE_2".MONITORING.COOLING_SYSTEM.INPUT_TEMPERATURE)
   END_RUNG
   RUNG wire#w1
      Move(in := "DB1451_MAIN_COOLING_SYSTEM".COOLING_OUTPUT_SENSOR.COOLING_FLOW_SENSOR_VALUE, out1 => "DB16701_OPC_UA_MASTER_MACHINE_DATA_UPDATE_2".MONITORING.COOLING_SYSTEM.OUTPUT_FLOW)
      Move(in := "DB1451_MAIN_COOLING_SYSTEM".COOLING_OUTPUT_SENSOR.COOLING_TEMP_SENSOR_VALUE, out1 => "DB16701_OPC_UA_MASTER_MACHINE_DATA_UPDATE_2".MONITORING.COOLING_SYSTEM.OUTPUT_TEMPERATURE)
   END_RUNG
   // the same network as SCL:
   IF "M_ONE" THEN
       "DB16701_OPC_UA_MASTER_MACHINE_DATA_UPDATE_2".MONITORING.COOLING_SYSTEM.INPUT_FLOW := "DB1451_MAIN_COOLING_SYSTEM".COOLING_INPUT_SENSOR.COOLING_FLOW_SENSOR_VALUE;
       "DB16701_OPC_UA_MASTER_MACHINE_DATA_UPDATE_2".MONITORING.COOLING_SYSTEM.INPUT_TEMPERATURE := "DB1451_MAIN_COOLING_SYSTEM".COOLING_INPUT_SENSOR.COOLING_TEMP_SENSOR_VALUE;
       "DB16701_OPC_UA_MASTER_MACHINE_DATA_UPDATE_2".MONITORING.COOLING_SYSTEM.OUTPUT_FLOW := "DB1451_MAIN_COOLING_SYSTEM".COOLING_OUTPUT_SENSOR.COOLING_FLOW_SENSOR_VALUE;
       "DB16701_OPC_UA_MASTER_MACHINE_DATA_UPDATE_2".MONITORING.COOLING_SYSTEM.OUTPUT_TEMPERATURE := "DB1451_MAIN_COOLING_SYSTEM".COOLING_OUTPUT_SENSOR.COOLING_TEMP_SENSOR_VALUE;
   END_IF;
END_REGION

REGION Network 39: MONITORING - UNIT 01 - TEMPERATURE
   RUNG wire#powerrail
      Contact( "M_ONE" )
      wire#w1
      Move(in := "DB10200_PYROMETERS".UNIT_1_PYROMETER.PROCESS_TEMPERATURE, out1 => "DB16701_OPC_UA_MASTER_MACHINE_DATA_UPDATE_2".MONITORING.UNIT_1.TEMPERATURE.DISC_SURFACE)
   END_RUNG
   RUNG wire#w1
      Move(in := "DB10200_PYROMETERS".UNIT_1_PYROMETER.HEAD_TEMPERATURE, out1 => "DB16701_OPC_UA_MASTER_MACHINE_DATA_UPDATE_2".MONITORING.UNIT_1.TEMPERATURE.AMBIENT_PYROMETER)
   END_RUNG
   // the same network as SCL:
   IF "M_ONE" THEN
       "DB16701_OPC_UA_MASTER_MACHINE_DATA_UPDATE_2".MONITORING.UNIT_1.TEMPERATURE.DISC_SURFACE := "DB10200_PYROMETERS".UNIT_1_PYROMETER.PROCESS_TEMPERATURE;
       "DB16701_OPC_UA_MASTER_MACHINE_DATA_UPDATE_2".MONITORING.UNIT_1.TEMPERATURE.AMBIENT_PYROMETER := "DB10200_PYROMETERS".UNIT_1_PYROMETER.HEAD_TEMPERATURE;
   END_IF;
END_REGION

REGION Network 40: MONITORING - UNIT 01 - COOLING SYSTEM
   RUNG wire#powerrail
      Contact( "M_ONE" )
      wire#w1
      Move(in := "DB1471_UNIT_1_LASER_COOLING_ALARMS".LASER_HEAD_SENSOR_VALUES.COOLING_FLOW_SENSOR_ACTUAL_VALUE, out1 => "DB16701_OPC_UA_MASTER_MACHINE_DATA_UPDATE_2".MONITORING.UNIT_1.COOLING_SYSTEM.LASER_HEAD_FLOW)
      Move(in := "DB1471_UNIT_1_LASER_COOLING_ALARMS".LASER_HEAD_SENSOR_VALUES.COOLING_TEMP_SENSOR_ACTUAL_VALUE, out1 => "DB16701_OPC_UA_MASTER_MACHINE_DATA_UPDATE_2".MONITORING.UNIT_1.COOLING_SYSTEM.LASER_HEAD_TEMPERATURE)
   END_RUNG
   RUNG wire#w1
      Move(in := "DB1471_UNIT_1_LASER_COOLING_ALARMS".LASER_OUTPUT_SENSOR_VALUES.COOLING_FLOW_SENSOR_ACTUAL_VALUE, out1 => "DB16701_OPC_UA_MASTER_MACHINE_DATA_UPDATE_2".MONITORING.UNIT_1.COOLING_SYSTEM.LASER_FLOW)
      Move(in := "DB1471_UNIT_1_LASER_COOLING_ALARMS".LASER_OUTPUT_SENSOR_VALUES.COOLING_TEMP_SENSOR_ACTUAL_VALUE, out1 => "DB16701_OPC_UA_MASTER_MACHINE_DATA_UPDATE_2".MONITORING.UNIT_1.COOLING_SYSTEM.LASER_TEMPERATURE)
   END_RUNG
   RUNG wire#w1
      Move(in := "DB1471_UNIT_1_LASER_COOLING_ALARMS".NOZZLE_SENSOR_VALUES.COOLING_FLOW_SENSOR_ACTUAL_VALUE, out1 => "DB16701_OPC_UA_MASTER_MACHINE_DATA_UPDATE_2".MONITORING.UNIT_1.COOLING_SYSTEM.NOZZLE_FLOW)
      Move(in := "DB1471_UNIT_1_LASER_COOLING_ALARMS".NOZZLE_SENSOR_VALUES.COOLING_TEMP_SENSOR_ACTUAL_VALUE, out1 => "DB16701_OPC_UA_MASTER_MACHINE_DATA_UPDATE_2".MONITORING.UNIT_1.COOLING_SYSTEM.NOZZLE_TEMPERATURE)
   END_RUNG
   RUNG wire#w1
      Move(in := "DB1462_SHIELD_AUX_COOLING_ALARMS".UNIT_1.FLOW_VALUE, out1 => "DB16701_OPC_UA_MASTER_MACHINE_DATA_UPDATE_2".MONITORING.UNIT_1.COOLING_SYSTEM.SHIELD_FLOW)
      Move(in := "DB1462_SHIELD_AUX_COOLING_ALARMS".UNIT_1.TEMP_VALUE, out1 => "DB16701_OPC_UA_MASTER_MACHINE_DATA_UPDATE_2".MONITORING.UNIT_1.COOLING_SYSTEM.SHIELD_TEMPERATURE)
   END_RUNG
   // the same network as SCL:
   IF "M_ONE" THEN
       "DB16701_OPC_UA_MASTER_MACHINE_DATA_UPDATE_2".MONITORING.UNIT_1.COOLING_SYSTEM.LASER_HEAD_FLOW := "DB1471_UNIT_1_LASER_COOLING_ALARMS".LASER_HEAD_SENSOR_VALUES.COOLING_FLOW_SENSOR_ACTUAL_VALUE;
       "DB16701_OPC_UA_MASTER_MACHINE_DATA_UPDATE_2".MONITORING.UNIT_1.COOLING_SYSTEM.LASER_HEAD_TEMPERATURE := "DB1471_UNIT_1_LASER_COOLING_ALARMS".LASER_HEAD_SENSOR_VALUES.COOLING_TEMP_SENSOR_ACTUAL_VALUE;
       "DB16701_OPC_UA_MASTER_MACHINE_DATA_UPDATE_2".MONITORING.UNIT_1.COOLING_SYSTEM.LASER_FLOW := "DB1471_UNIT_1_LASER_COOLING_ALARMS".LASER_OUTPUT_SENSOR_VALUES.COOLING_FLOW_SENSOR_ACTUAL_VALUE;
       "DB16701_OPC_UA_MASTER_MACHINE_DATA_UPDATE_2".MONITORING.UNIT_1.COOLING_SYSTEM.LASER_TEMPERATURE := "DB1471_UNIT_1_LASER_COOLING_ALARMS".LASER_OUTPUT_SENSOR_VALUES.COOLING_TEMP_SENSOR_ACTUAL_VALUE;
       "DB16701_OPC_UA_MASTER_MACHINE_DATA_UPDATE_2".MONITORING.UNIT_1.COOLING_SYSTEM.NOZZLE_FLOW := "DB1471_UNIT_1_LASER_COOLING_ALARMS".NOZZLE_SENSOR_VALUES.COOLING_FLOW_SENSOR_ACTUAL_VALUE;
       "DB16701_OPC_UA_MASTER_MACHINE_DATA_UPDATE_2".MONITORING.UNIT_1.COOLING_SYSTEM.NOZZLE_TEMPERATURE := "DB1471_UNIT_1_LASER_COOLING_ALARMS".NOZZLE_SENSOR_VALUES.COOLING_TEMP_SENSOR_ACTUAL_VALUE;
       "DB16701_OPC_UA_MASTER_MACHINE_DATA_UPDATE_2".MONITORING.UNIT_1.COOLING_SYSTEM.SHIELD_FLOW := "DB1462_SHIELD_AUX_COOLING_ALARMS".UNIT_1.FLOW_VALUE;
       "DB16701_OPC_UA_MASTER_MACHINE_DATA_UPDATE_2".MONITORING.UNIT_1.COOLING_SYSTEM.SHIELD_TEMPERATURE := "DB1462_SHIELD_AUX_COOLING_ALARMS".UNIT_1.TEMP_VALUE;
   END_IF;
END_REGION

REGION Network 41: MONITORING - UNIT 01 - AIR EXTRACTION
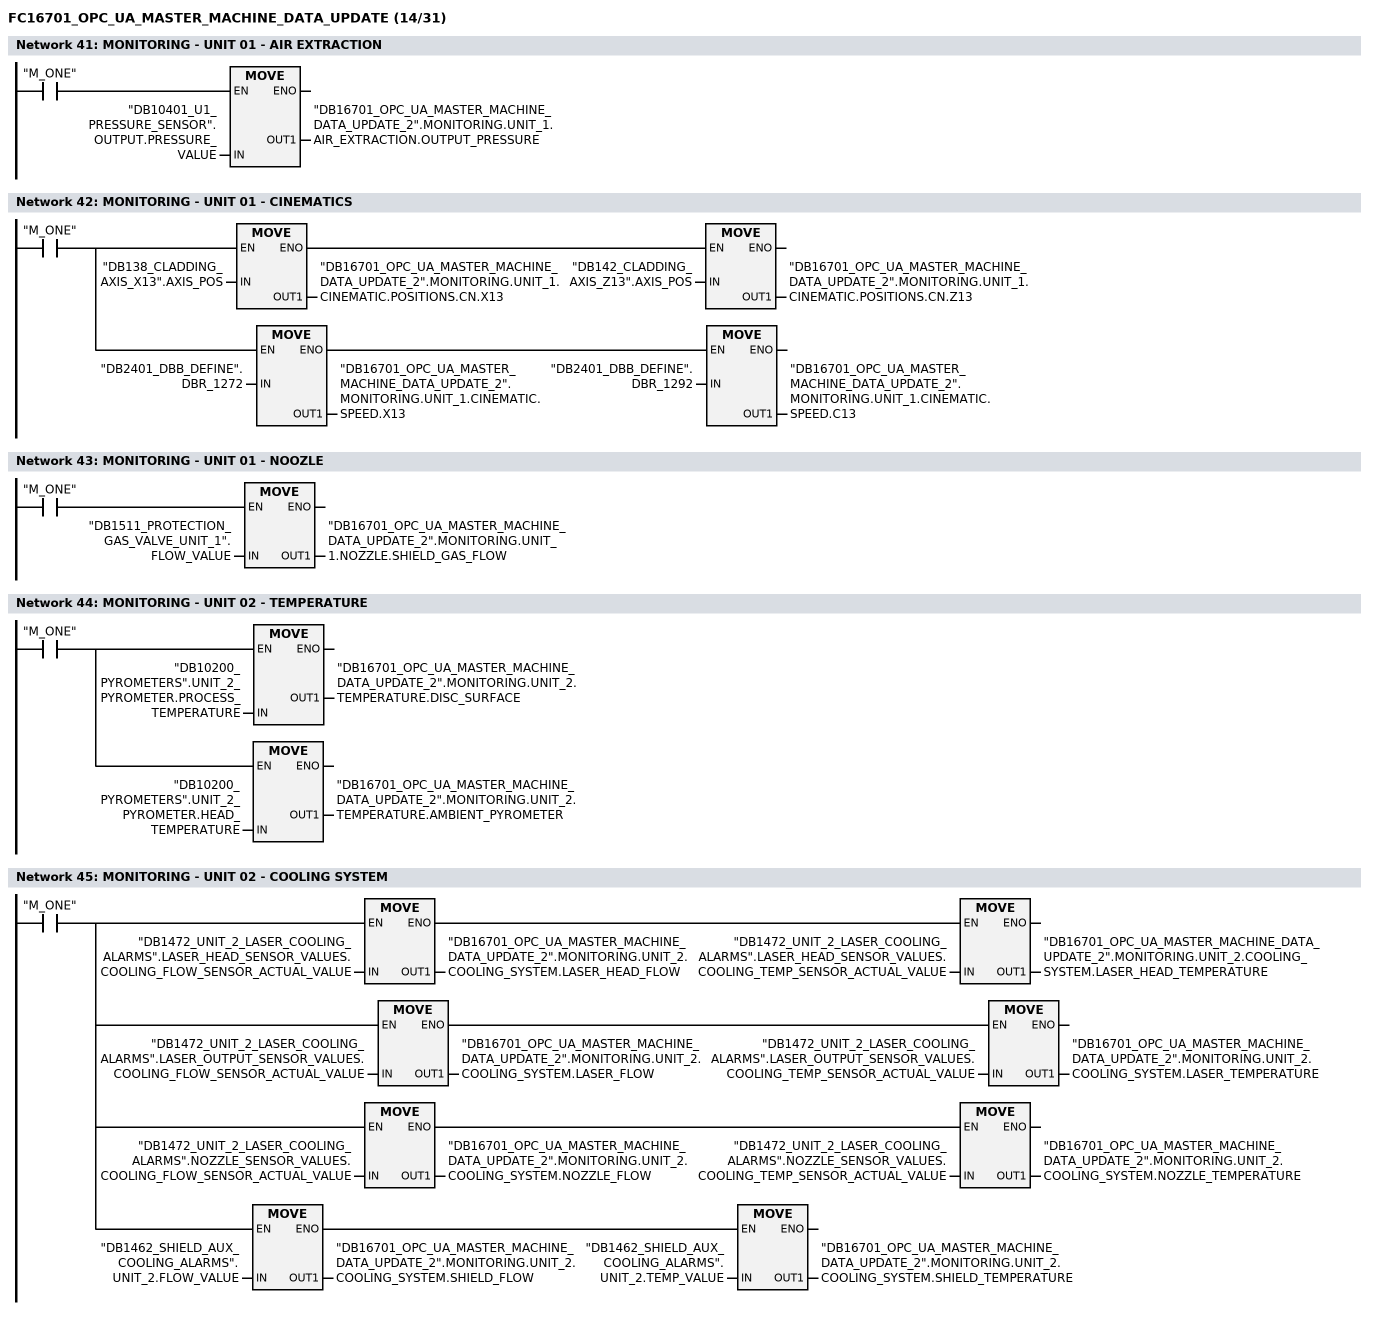
   RUNG wire#powerrail
      Contact( "M_ONE" )
      Move(in := "DB10401_U1_PRESSURE_SENSOR".OUTPUT.PRESSURE_VALUE, out1 => "DB16701_OPC_UA_MASTER_MACHINE_DATA_UPDATE_2".MONITORING.UNIT_1.AIR_EXTRACTION.OUTPUT_PRESSURE)
   END_RUNG
   // the same network as SCL:
   IF "M_ONE" THEN
       "DB16701_OPC_UA_MASTER_MACHINE_DATA_UPDATE_2".MONITORING.UNIT_1.AIR_EXTRACTION.OUTPUT_PRESSURE := "DB10401_U1_PRESSURE_SENSOR".OUTPUT.PRESSURE_VALUE;
   END_IF;
END_REGION

REGION Network 42: MONITORING - UNIT 01 - CINEMATICS
   RUNG wire#powerrail
      Contact( "M_ONE" )
      wire#w1
      Move(in := "DB138_CLADDING_AXIS_X13".AXIS_POS, out1 => "DB16701_OPC_UA_MASTER_MACHINE_DATA_UPDATE_2".MONITORING.UNIT_1.CINEMATIC.POSITIONS.CN.X13)
      Move(in := "DB142_CLADDING_AXIS_Z13".AXIS_POS, out1 => "DB16701_OPC_UA_MASTER_MACHINE_DATA_UPDATE_2".MONITORING.UNIT_1.CINEMATIC.POSITIONS.CN.Z13)
   END_RUNG
   RUNG wire#w1
      Move(in := "DB2401_DBB_DEFINE".DBR_1272, out1 => "DB16701_OPC_UA_MASTER_MACHINE_DATA_UPDATE_2".MONITORING.UNIT_1.CINEMATIC.SPEED.X13)
      Move(in := "DB2401_DBB_DEFINE".DBR_1292, out1 => "DB16701_OPC_UA_MASTER_MACHINE_DATA_UPDATE_2".MONITORING.UNIT_1.CINEMATIC.SPEED.C13)
   END_RUNG
   // the same network as SCL:
   IF "M_ONE" THEN
       "DB16701_OPC_UA_MASTER_MACHINE_DATA_UPDATE_2".MONITORING.UNIT_1.CINEMATIC.POSITIONS.CN.X13 := "DB138_CLADDING_AXIS_X13".AXIS_POS;
       "DB16701_OPC_UA_MASTER_MACHINE_DATA_UPDATE_2".MONITORING.UNIT_1.CINEMATIC.POSITIONS.CN.Z13 := "DB142_CLADDING_AXIS_Z13".AXIS_POS;
       "DB16701_OPC_UA_MASTER_MACHINE_DATA_UPDATE_2".MONITORING.UNIT_1.CINEMATIC.SPEED.X13 := "DB2401_DBB_DEFINE".DBR_1272;
       "DB16701_OPC_UA_MASTER_MACHINE_DATA_UPDATE_2".MONITORING.UNIT_1.CINEMATIC.SPEED.C13 := "DB2401_DBB_DEFINE".DBR_1292;
   END_IF;
END_REGION

REGION Network 43: MONITORING - UNIT 01 - NOOZLE
   RUNG wire#powerrail
      Contact( "M_ONE" )
      Move(in := "DB1511_PROTECTION_GAS_VALVE_UNIT_1".FLOW_VALUE, out1 => "DB16701_OPC_UA_MASTER_MACHINE_DATA_UPDATE_2".MONITORING.UNIT_1.NOZZLE.SHIELD_GAS_FLOW)
   END_RUNG
   // the same network as SCL:
   IF "M_ONE" THEN
       "DB16701_OPC_UA_MASTER_MACHINE_DATA_UPDATE_2".MONITORING.UNIT_1.NOZZLE.SHIELD_GAS_FLOW := "DB1511_PROTECTION_GAS_VALVE_UNIT_1".FLOW_VALUE;
   END_IF;
END_REGION

REGION Network 44: MONITORING - UNIT 02 - TEMPERATURE
   RUNG wire#powerrail
      Contact( "M_ONE" )
      wire#w1
      Move(in := "DB10200_PYROMETERS".UNIT_2_PYROMETER.PROCESS_TEMPERATURE, out1 => "DB16701_OPC_UA_MASTER_MACHINE_DATA_UPDATE_2".MONITORING.UNIT_2.TEMPERATURE.DISC_SURFACE)
   END_RUNG
   RUNG wire#w1
      Move(in := "DB10200_PYROMETERS".UNIT_2_PYROMETER.HEAD_TEMPERATURE, out1 => "DB16701_OPC_UA_MASTER_MACHINE_DATA_UPDATE_2".MONITORING.UNIT_2.TEMPERATURE.AMBIENT_PYROMETER)
   END_RUNG
   // the same network as SCL:
   IF "M_ONE" THEN
       "DB16701_OPC_UA_MASTER_MACHINE_DATA_UPDATE_2".MONITORING.UNIT_2.TEMPERATURE.DISC_SURFACE := "DB10200_PYROMETERS".UNIT_2_PYROMETER.PROCESS_TEMPERATURE;
       "DB16701_OPC_UA_MASTER_MACHINE_DATA_UPDATE_2".MONITORING.UNIT_2.TEMPERATURE.AMBIENT_PYROMETER := "DB10200_PYROMETERS".UNIT_2_PYROMETER.HEAD_TEMPERATURE;
   END_IF;
END_REGION

REGION Network 45: MONITORING - UNIT 02 - COOLING SYSTEM
   RUNG wire#powerrail
      Contact( "M_ONE" )
      wire#w1
      Move(in := "DB1472_UNIT_2_LASER_COOLING_ALARMS".LASER_HEAD_SENSOR_VALUES.COOLING_FLOW_SENSOR_ACTUAL_VALUE, out1 => "DB16701_OPC_UA_MASTER_MACHINE_DATA_UPDATE_2".MONITORING.UNIT_2.COOLING_SYSTEM.LASER_HEAD_FLOW)
      Move(in := "DB1472_UNIT_2_LASER_COOLING_ALARMS".LASER_HEAD_SENSOR_VALUES.COOLING_TEMP_SENSOR_ACTUAL_VALUE, out1 => "DB16701_OPC_UA_MASTER_MACHINE_DATA_UPDATE_2".MONITORING.UNIT_2.COOLING_SYSTEM.LASER_HEAD_TEMPERATURE)
   END_RUNG
   RUNG wire#w1
      Move(in := "DB1472_UNIT_2_LASER_COOLING_ALARMS".LASER_OUTPUT_SENSOR_VALUES.COOLING_FLOW_SENSOR_ACTUAL_VALUE, out1 => "DB16701_OPC_UA_MASTER_MACHINE_DATA_UPDATE_2".MONITORING.UNIT_2.COOLING_SYSTEM.LASER_FLOW)
      Move(in := "DB1472_UNIT_2_LASER_COOLING_ALARMS".LASER_OUTPUT_SENSOR_VALUES.COOLING_TEMP_SENSOR_ACTUAL_VALUE, out1 => "DB16701_OPC_UA_MASTER_MACHINE_DATA_UPDATE_2".MONITORING.UNIT_2.COOLING_SYSTEM.LASER_TEMPERATURE)
   END_RUNG
   RUNG wire#w1
      Move(in := "DB1472_UNIT_2_LASER_COOLING_ALARMS".NOZZLE_SENSOR_VALUES.COOLING_FLOW_SENSOR_ACTUAL_VALUE, out1 => "DB16701_OPC_UA_MASTER_MACHINE_DATA_UPDATE_2".MONITORING.UNIT_2.COOLING_SYSTEM.NOZZLE_FLOW)
      Move(in := "DB1472_UNIT_2_LASER_COOLING_ALARMS".NOZZLE_SENSOR_VALUES.COOLING_TEMP_SENSOR_ACTUAL_VALUE, out1 => "DB16701_OPC_UA_MASTER_MACHINE_DATA_UPDATE_2".MONITORING.UNIT_2.COOLING_SYSTEM.NOZZLE_TEMPERATURE)
   END_RUNG
   RUNG wire#w1
      Move(in := "DB1462_SHIELD_AUX_COOLING_ALARMS".UNIT_2.FLOW_VALUE, out1 => "DB16701_OPC_UA_MASTER_MACHINE_DATA_UPDATE_2".MONITORING.UNIT_2.COOLING_SYSTEM.SHIELD_FLOW)
      Move(in := "DB1462_SHIELD_AUX_COOLING_ALARMS".UNIT_2.TEMP_VALUE, out1 => "DB16701_OPC_UA_MASTER_MACHINE_DATA_UPDATE_2".MONITORING.UNIT_2.COOLING_SYSTEM.SHIELD_TEMPERATURE)
   END_RUNG
   // the same network as SCL:
   IF "M_ONE" THEN
       "DB16701_OPC_UA_MASTER_MACHINE_DATA_UPDATE_2".MONITORING.UNIT_2.COOLING_SYSTEM.LASER_HEAD_FLOW := "DB1472_UNIT_2_LASER_COOLING_ALARMS".LASER_HEAD_SENSOR_VALUES.COOLING_FLOW_SENSOR_ACTUAL_VALUE;
       "DB16701_OPC_UA_MASTER_MACHINE_DATA_UPDATE_2".MONITORING.UNIT_2.COOLING_SYSTEM.LASER_HEAD_TEMPERATURE := "DB1472_UNIT_2_LASER_COOLING_ALARMS".LASER_HEAD_SENSOR_VALUES.COOLING_TEMP_SENSOR_ACTUAL_VALUE;
       "DB16701_OPC_UA_MASTER_MACHINE_DATA_UPDATE_2".MONITORING.UNIT_2.COOLING_SYSTEM.LASER_FLOW := "DB1472_UNIT_2_LASER_COOLING_ALARMS".LASER_OUTPUT_SENSOR_VALUES.COOLING_FLOW_SENSOR_ACTUAL_VALUE;
       "DB16701_OPC_UA_MASTER_MACHINE_DATA_UPDATE_2".MONITORING.UNIT_2.COOLING_SYSTEM.LASER_TEMPERATURE := "DB1472_UNIT_2_LASER_COOLING_ALARMS".LASER_OUTPUT_SENSOR_VALUES.COOLING_TEMP_SENSOR_ACTUAL_VALUE;
       "DB16701_OPC_UA_MASTER_MACHINE_DATA_UPDATE_2".MONITORING.UNIT_2.COOLING_SYSTEM.NOZZLE_FLOW := "DB1472_UNIT_2_LASER_COOLING_ALARMS".NOZZLE_SENSOR_VALUES.COOLING_FLOW_SENSOR_ACTUAL_VALUE;
       "DB16701_OPC_UA_MASTER_MACHINE_DATA_UPDATE_2".MONITORING.UNIT_2.COOLING_SYSTEM.NOZZLE_TEMPERATURE := "DB1472_UNIT_2_LASER_COOLING_ALARMS".NOZZLE_SENSOR_VALUES.COOLING_TEMP_SENSOR_ACTUAL_VALUE;
       "DB16701_OPC_UA_MASTER_MACHINE_DATA_UPDATE_2".MONITORING.UNIT_2.COOLING_SYSTEM.SHIELD_FLOW := "DB1462_SHIELD_AUX_COOLING_ALARMS".UNIT_2.FLOW_VALUE;
       "DB16701_OPC_UA_MASTER_MACHINE_DATA_UPDATE_2".MONITORING.UNIT_2.COOLING_SYSTEM.SHIELD_TEMPERATURE := "DB1462_SHIELD_AUX_COOLING_ALARMS".UNIT_2.TEMP_VALUE;
   END_IF;
END_REGION

REGION Network 46: MONITORING - UNIT 02 - AIR EXTRACTION
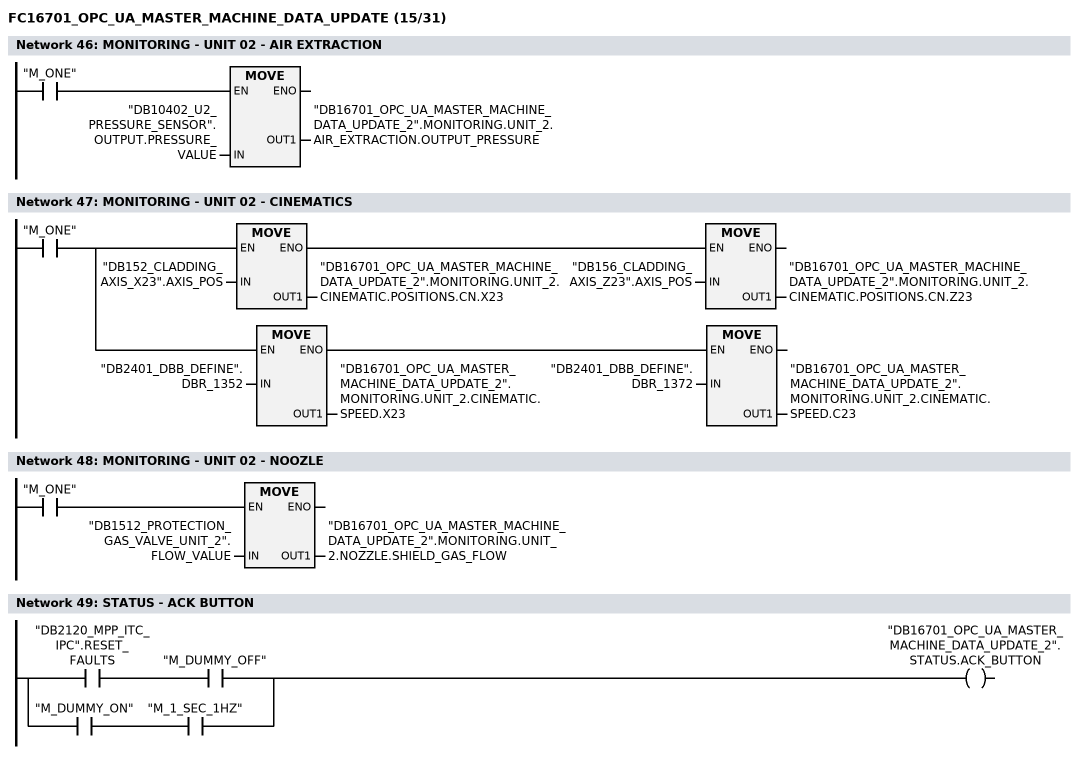
   RUNG wire#powerrail
      Contact( "M_ONE" )
      Move(in := "DB10402_U2_PRESSURE_SENSOR".OUTPUT.PRESSURE_VALUE, out1 => "DB16701_OPC_UA_MASTER_MACHINE_DATA_UPDATE_2".MONITORING.UNIT_2.AIR_EXTRACTION.OUTPUT_PRESSURE)
   END_RUNG
   // the same network as SCL:
   IF "M_ONE" THEN
       "DB16701_OPC_UA_MASTER_MACHINE_DATA_UPDATE_2".MONITORING.UNIT_2.AIR_EXTRACTION.OUTPUT_PRESSURE := "DB10402_U2_PRESSURE_SENSOR".OUTPUT.PRESSURE_VALUE;
   END_IF;
END_REGION

REGION Network 47: MONITORING - UNIT 02 - CINEMATICS
   RUNG wire#powerrail
      Contact( "M_ONE" )
      wire#w1
      Move(in := "DB152_CLADDING_AXIS_X23".AXIS_POS, out1 => "DB16701_OPC_UA_MASTER_MACHINE_DATA_UPDATE_2".MONITORING.UNIT_2.CINEMATIC.POSITIONS.CN.X23)
      Move(in := "DB156_CLADDING_AXIS_Z23".AXIS_POS, out1 => "DB16701_OPC_UA_MASTER_MACHINE_DATA_UPDATE_2".MONITORING.UNIT_2.CINEMATIC.POSITIONS.CN.Z23)
   END_RUNG
   RUNG wire#w1
      Move(in := "DB2401_DBB_DEFINE".DBR_1352, out1 => "DB16701_OPC_UA_MASTER_MACHINE_DATA_UPDATE_2".MONITORING.UNIT_2.CINEMATIC.SPEED.X23)
      Move(in := "DB2401_DBB_DEFINE".DBR_1372, out1 => "DB16701_OPC_UA_MASTER_MACHINE_DATA_UPDATE_2".MONITORING.UNIT_2.CINEMATIC.SPEED.C23)
   END_RUNG
   // the same network as SCL:
   IF "M_ONE" THEN
       "DB16701_OPC_UA_MASTER_MACHINE_DATA_UPDATE_2".MONITORING.UNIT_2.CINEMATIC.POSITIONS.CN.X23 := "DB152_CLADDING_AXIS_X23".AXIS_POS;
       "DB16701_OPC_UA_MASTER_MACHINE_DATA_UPDATE_2".MONITORING.UNIT_2.CINEMATIC.POSITIONS.CN.Z23 := "DB156_CLADDING_AXIS_Z23".AXIS_POS;
       "DB16701_OPC_UA_MASTER_MACHINE_DATA_UPDATE_2".MONITORING.UNIT_2.CINEMATIC.SPEED.X23 := "DB2401_DBB_DEFINE".DBR_1352;
       "DB16701_OPC_UA_MASTER_MACHINE_DATA_UPDATE_2".MONITORING.UNIT_2.CINEMATIC.SPEED.C23 := "DB2401_DBB_DEFINE".DBR_1372;
   END_IF;
END_REGION

REGION Network 48: MONITORING - UNIT 02 - NOOZLE
   RUNG wire#powerrail
      Contact( "M_ONE" )
      Move(in := "DB1512_PROTECTION_GAS_VALVE_UNIT_2".FLOW_VALUE, out1 => "DB16701_OPC_UA_MASTER_MACHINE_DATA_UPDATE_2".MONITORING.UNIT_2.NOZZLE.SHIELD_GAS_FLOW)
   END_RUNG
   // the same network as SCL:
   IF "M_ONE" THEN
       "DB16701_OPC_UA_MASTER_MACHINE_DATA_UPDATE_2".MONITORING.UNIT_2.NOZZLE.SHIELD_GAS_FLOW := "DB1512_PROTECTION_GAS_VALVE_UNIT_2".FLOW_VALUE;
   END_IF;
END_REGION

REGION Network 49: STATUS - ACK BUTTON
   RUNG wire#powerrail
      Contact( "DB2120_MPP_ITC_IPC".RESET_FAULTS )
      Contact( "M_DUMMY_OFF" )
      wire#w1
      Coil( "DB16701_OPC_UA_MASTER_MACHINE_DATA_UPDATE_2".STATUS.ACK_BUTTON )
   END_RUNG
   RUNG wire#powerrail
      Contact( "M_DUMMY_ON" )
      Contact( "M_1_SEC_1HZ" )
   END_RUNG wire#w1
   // the same network as SCL:
   "DB16701_OPC_UA_MASTER_MACHINE_DATA_UPDATE_2".STATUS.ACK_BUTTON := ("DB2120_MPP_ITC_IPC".RESET_FAULTS AND "M_DUMMY_OFF") OR ("M_DUMMY_ON" AND "M_1_SEC_1HZ");
END_REGION

REGION Network 50: STATUS - PART TRACKING
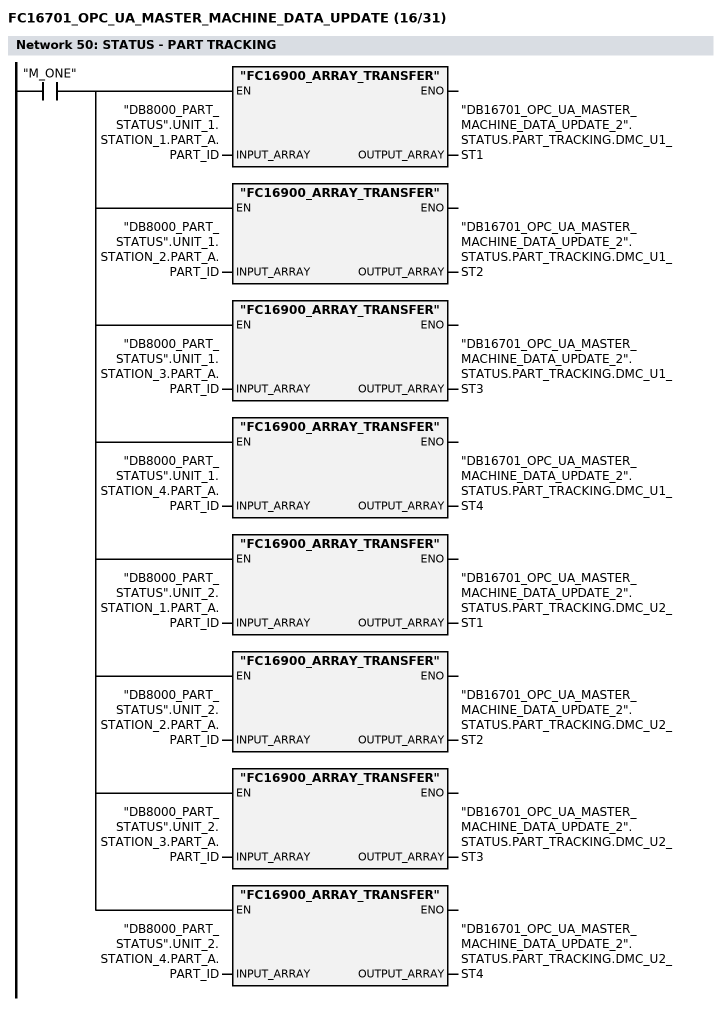
   RUNG wire#powerrail
      Contact( "M_ONE" )
      wire#w1
      "FC16900_ARRAY_TRANSFER"(INPUT_ARRAY := "DB8000_PART_STATUS".UNIT_1.STATION_1.PART_A.PART_ID, OUTPUT_ARRAY => "DB16701_OPC_UA_MASTER_MACHINE_DATA_UPDATE_2".STATUS.PART_TRACKING.DMC_U1_ST1)
   END_RUNG
   RUNG wire#w1
      "FC16900_ARRAY_TRANSFER"(INPUT_ARRAY := "DB8000_PART_STATUS".UNIT_1.STATION_2.PART_A.PART_ID, OUTPUT_ARRAY => "DB16701_OPC_UA_MASTER_MACHINE_DATA_UPDATE_2".STATUS.PART_TRACKING.DMC_U1_ST2)
   END_RUNG
   RUNG wire#w1
      "FC16900_ARRAY_TRANSFER"(INPUT_ARRAY := "DB8000_PART_STATUS".UNIT_1.STATION_3.PART_A.PART_ID, OUTPUT_ARRAY => "DB16701_OPC_UA_MASTER_MACHINE_DATA_UPDATE_2".STATUS.PART_TRACKING.DMC_U1_ST3)
   END_RUNG
   RUNG wire#w1
      "FC16900_ARRAY_TRANSFER"(INPUT_ARRAY := "DB8000_PART_STATUS".UNIT_1.STATION_4.PART_A.PART_ID, OUTPUT_ARRAY => "DB16701_OPC_UA_MASTER_MACHINE_DATA_UPDATE_2".STATUS.PART_TRACKING.DMC_U1_ST4)
   END_RUNG
   RUNG wire#w1
      "FC16900_ARRAY_TRANSFER"(INPUT_ARRAY := "DB8000_PART_STATUS".UNIT_2.STATION_1.PART_A.PART_ID, OUTPUT_ARRAY => "DB16701_OPC_UA_MASTER_MACHINE_DATA_UPDATE_2".STATUS.PART_TRACKING.DMC_U2_ST1)
   END_RUNG
   RUNG wire#w1
      "FC16900_ARRAY_TRANSFER"(INPUT_ARRAY := "DB8000_PART_STATUS".UNIT_2.STATION_2.PART_A.PART_ID, OUTPUT_ARRAY => "DB16701_OPC_UA_MASTER_MACHINE_DATA_UPDATE_2".STATUS.PART_TRACKING.DMC_U2_ST2)
   END_RUNG
   RUNG wire#w1
      "FC16900_ARRAY_TRANSFER"(INPUT_ARRAY := "DB8000_PART_STATUS".UNIT_2.STATION_3.PART_A.PART_ID, OUTPUT_ARRAY => "DB16701_OPC_UA_MASTER_MACHINE_DATA_UPDATE_2".STATUS.PART_TRACKING.DMC_U2_ST3)
   END_RUNG
   RUNG wire#w1
      "FC16900_ARRAY_TRANSFER"(INPUT_ARRAY := "DB8000_PART_STATUS".UNIT_2.STATION_4.PART_A.PART_ID, OUTPUT_ARRAY => "DB16701_OPC_UA_MASTER_MACHINE_DATA_UPDATE_2".STATUS.PART_TRACKING.DMC_U2_ST4)
   END_RUNG
   // the same network as SCL:
   #_w1 := "M_ONE";
   IF #_w1 THEN
       "FC16900_ARRAY_TRANSFER"(INPUT_ARRAY := "DB8000_PART_STATUS".UNIT_1.STATION_1.PART_A.PART_ID,
                               OUTPUT_ARRAY => "DB16701_OPC_UA_MASTER_MACHINE_DATA_UPDATE_2".STATUS.PART_TRACKING.DMC_U1_ST1);
       "FC16900_ARRAY_TRANSFER"(INPUT_ARRAY := "DB8000_PART_STATUS".UNIT_1.STATION_2.PART_A.PART_ID,
                               OUTPUT_ARRAY => "DB16701_OPC_UA_MASTER_MACHINE_DATA_UPDATE_2".STATUS.PART_TRACKING.DMC_U1_ST2);
       "FC16900_ARRAY_TRANSFER"(INPUT_ARRAY := "DB8000_PART_STATUS".UNIT_1.STATION_3.PART_A.PART_ID,
                               OUTPUT_ARRAY => "DB16701_OPC_UA_MASTER_MACHINE_DATA_UPDATE_2".STATUS.PART_TRACKING.DMC_U1_ST3);
       "FC16900_ARRAY_TRANSFER"(INPUT_ARRAY := "DB8000_PART_STATUS".UNIT_1.STATION_4.PART_A.PART_ID,
                               OUTPUT_ARRAY => "DB16701_OPC_UA_MASTER_MACHINE_DATA_UPDATE_2".STATUS.PART_TRACKING.DMC_U1_ST4);
       "FC16900_ARRAY_TRANSFER"(INPUT_ARRAY := "DB8000_PART_STATUS".UNIT_2.STATION_1.PART_A.PART_ID,
                               OUTPUT_ARRAY => "DB16701_OPC_UA_MASTER_MACHINE_DATA_UPDATE_2".STATUS.PART_TRACKING.DMC_U2_ST1);
       "FC16900_ARRAY_TRANSFER"(INPUT_ARRAY := "DB8000_PART_STATUS".UNIT_2.STATION_2.PART_A.PART_ID,
                               OUTPUT_ARRAY => "DB16701_OPC_UA_MASTER_MACHINE_DATA_UPDATE_2".STATUS.PART_TRACKING.DMC_U2_ST2);
       "FC16900_ARRAY_TRANSFER"(INPUT_ARRAY := "DB8000_PART_STATUS".UNIT_2.STATION_3.PART_A.PART_ID,
                               OUTPUT_ARRAY => "DB16701_OPC_UA_MASTER_MACHINE_DATA_UPDATE_2".STATUS.PART_TRACKING.DMC_U2_ST3);
       "FC16900_ARRAY_TRANSFER"(INPUT_ARRAY := "DB8000_PART_STATUS".UNIT_2.STATION_4.PART_A.PART_ID,
                               OUTPUT_ARRAY => "DB16701_OPC_UA_MASTER_MACHINE_DATA_UPDATE_2".STATUS.PART_TRACKING.DMC_U2_ST4);
   END_IF;
END_REGION

REGION Network 51: STATUS - MACHINE - GLOBAL STATUS
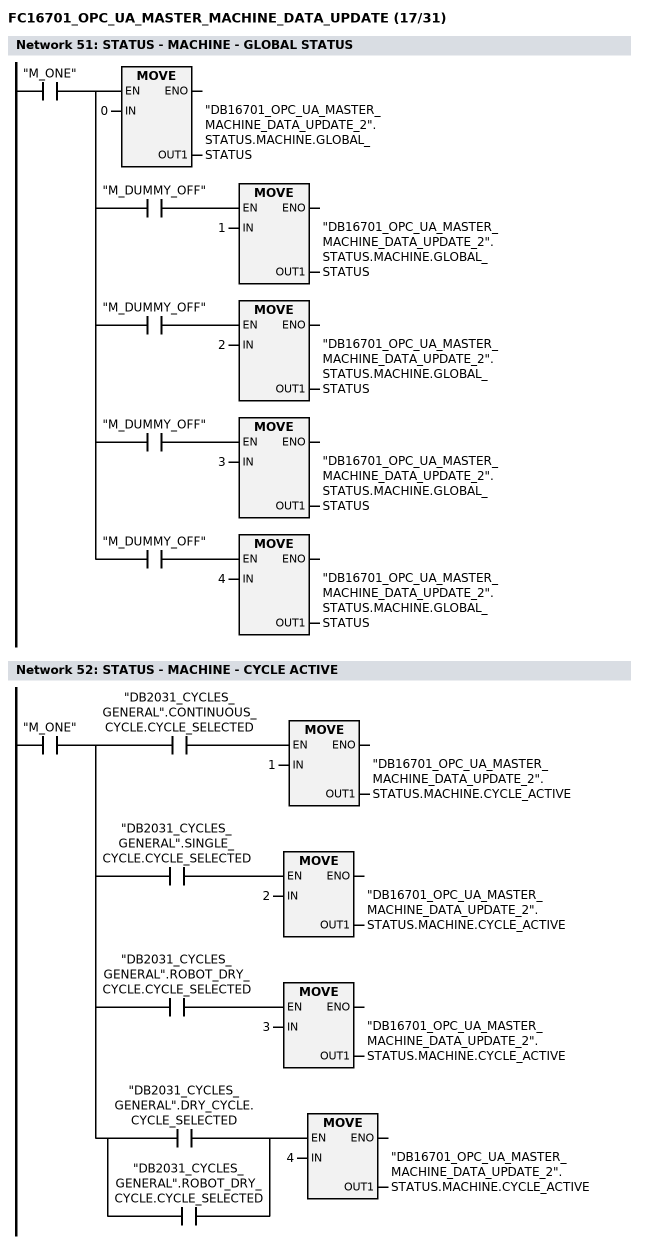
   RUNG wire#powerrail
      Contact( "M_ONE" )
      wire#w1
      Move(in := 0, out1 => "DB16701_OPC_UA_MASTER_MACHINE_DATA_UPDATE_2".STATUS.MACHINE.GLOBAL_STATUS)
   END_RUNG
   RUNG wire#w1
      Contact( "M_DUMMY_OFF" )
      Move(in := 1, out1 => "DB16701_OPC_UA_MASTER_MACHINE_DATA_UPDATE_2".STATUS.MACHINE.GLOBAL_STATUS)
   END_RUNG
   RUNG wire#w1
      Contact( "M_DUMMY_OFF" )
      Move(in := 2, out1 => "DB16701_OPC_UA_MASTER_MACHINE_DATA_UPDATE_2".STATUS.MACHINE.GLOBAL_STATUS)
   END_RUNG
   RUNG wire#w1
      Contact( "M_DUMMY_OFF" )
      Move(in := 3, out1 => "DB16701_OPC_UA_MASTER_MACHINE_DATA_UPDATE_2".STATUS.MACHINE.GLOBAL_STATUS)
   END_RUNG
   RUNG wire#w1
      Contact( "M_DUMMY_OFF" )
      Move(in := 4, out1 => "DB16701_OPC_UA_MASTER_MACHINE_DATA_UPDATE_2".STATUS.MACHINE.GLOBAL_STATUS)
   END_RUNG
   // the same network as SCL:
   IF "M_ONE" THEN "DB16701_OPC_UA_MASTER_MACHINE_DATA_UPDATE_2".STATUS.MACHINE.GLOBAL_STATUS := 0; END_IF;
   IF "M_ONE" AND "M_DUMMY_OFF" THEN
       "DB16701_OPC_UA_MASTER_MACHINE_DATA_UPDATE_2".STATUS.MACHINE.GLOBAL_STATUS := 1;
       "DB16701_OPC_UA_MASTER_MACHINE_DATA_UPDATE_2".STATUS.MACHINE.GLOBAL_STATUS := 2;
       "DB16701_OPC_UA_MASTER_MACHINE_DATA_UPDATE_2".STATUS.MACHINE.GLOBAL_STATUS := 3;
       "DB16701_OPC_UA_MASTER_MACHINE_DATA_UPDATE_2".STATUS.MACHINE.GLOBAL_STATUS := 4;
   END_IF;
END_REGION

REGION Network 52: STATUS - MACHINE - CYCLE ACTIVE
   RUNG wire#powerrail
      Contact( "M_ONE" )
      wire#w1
      Contact( "DB2031_CYCLES_GENERAL".CONTINUOUS_CYCLE.CYCLE_SELECTED )
      Move(in := 1, out1 => "DB16701_OPC_UA_MASTER_MACHINE_DATA_UPDATE_2".STATUS.MACHINE.CYCLE_ACTIVE)
   END_RUNG
   RUNG wire#w1
      Contact( "DB2031_CYCLES_GENERAL".SINGLE_CYCLE.CYCLE_SELECTED )
      Move(in := 2, out1 => "DB16701_OPC_UA_MASTER_MACHINE_DATA_UPDATE_2".STATUS.MACHINE.CYCLE_ACTIVE)
   END_RUNG
   RUNG wire#w1
      Contact( "DB2031_CYCLES_GENERAL".ROBOT_DRY_CYCLE.CYCLE_SELECTED )
      Move(in := 3, out1 => "DB16701_OPC_UA_MASTER_MACHINE_DATA_UPDATE_2".STATUS.MACHINE.CYCLE_ACTIVE)
   END_RUNG
   RUNG wire#w1
      Contact( "DB2031_CYCLES_GENERAL".DRY_CYCLE.CYCLE_SELECTED )
      wire#w2
      Move(in := 4, out1 => "DB16701_OPC_UA_MASTER_MACHINE_DATA_UPDATE_2".STATUS.MACHINE.CYCLE_ACTIVE)
   END_RUNG
   RUNG wire#w1
      Contact( "DB2031_CYCLES_GENERAL".ROBOT_DRY_CYCLE.CYCLE_SELECTED )
   END_RUNG wire#w2
   // the same network as SCL:
   IF "M_ONE" AND "DB2031_CYCLES_GENERAL".CONTINUOUS_CYCLE.CYCLE_SELECTED THEN
       "DB16701_OPC_UA_MASTER_MACHINE_DATA_UPDATE_2".STATUS.MACHINE.CYCLE_ACTIVE := 1;
   END_IF;
   IF "M_ONE" AND "DB2031_CYCLES_GENERAL".SINGLE_CYCLE.CYCLE_SELECTED THEN
       "DB16701_OPC_UA_MASTER_MACHINE_DATA_UPDATE_2".STATUS.MACHINE.CYCLE_ACTIVE := 2;
   END_IF;
   IF "M_ONE" AND "DB2031_CYCLES_GENERAL".ROBOT_DRY_CYCLE.CYCLE_SELECTED THEN
       "DB16701_OPC_UA_MASTER_MACHINE_DATA_UPDATE_2".STATUS.MACHINE.CYCLE_ACTIVE := 3;
   END_IF;
   IF "M_ONE" AND ("DB2031_CYCLES_GENERAL".DRY_CYCLE.CYCLE_SELECTED OR "DB2031_CYCLES_GENERAL".ROBOT_DRY_CYCLE.CYCLE_SELECTED) THEN
       "DB16701_OPC_UA_MASTER_MACHINE_DATA_UPDATE_2".STATUS.MACHINE.CYCLE_ACTIVE := 4;
   END_IF;
END_REGION

REGION Network 53: STATUS - MACHINE - MODE ACTIVE
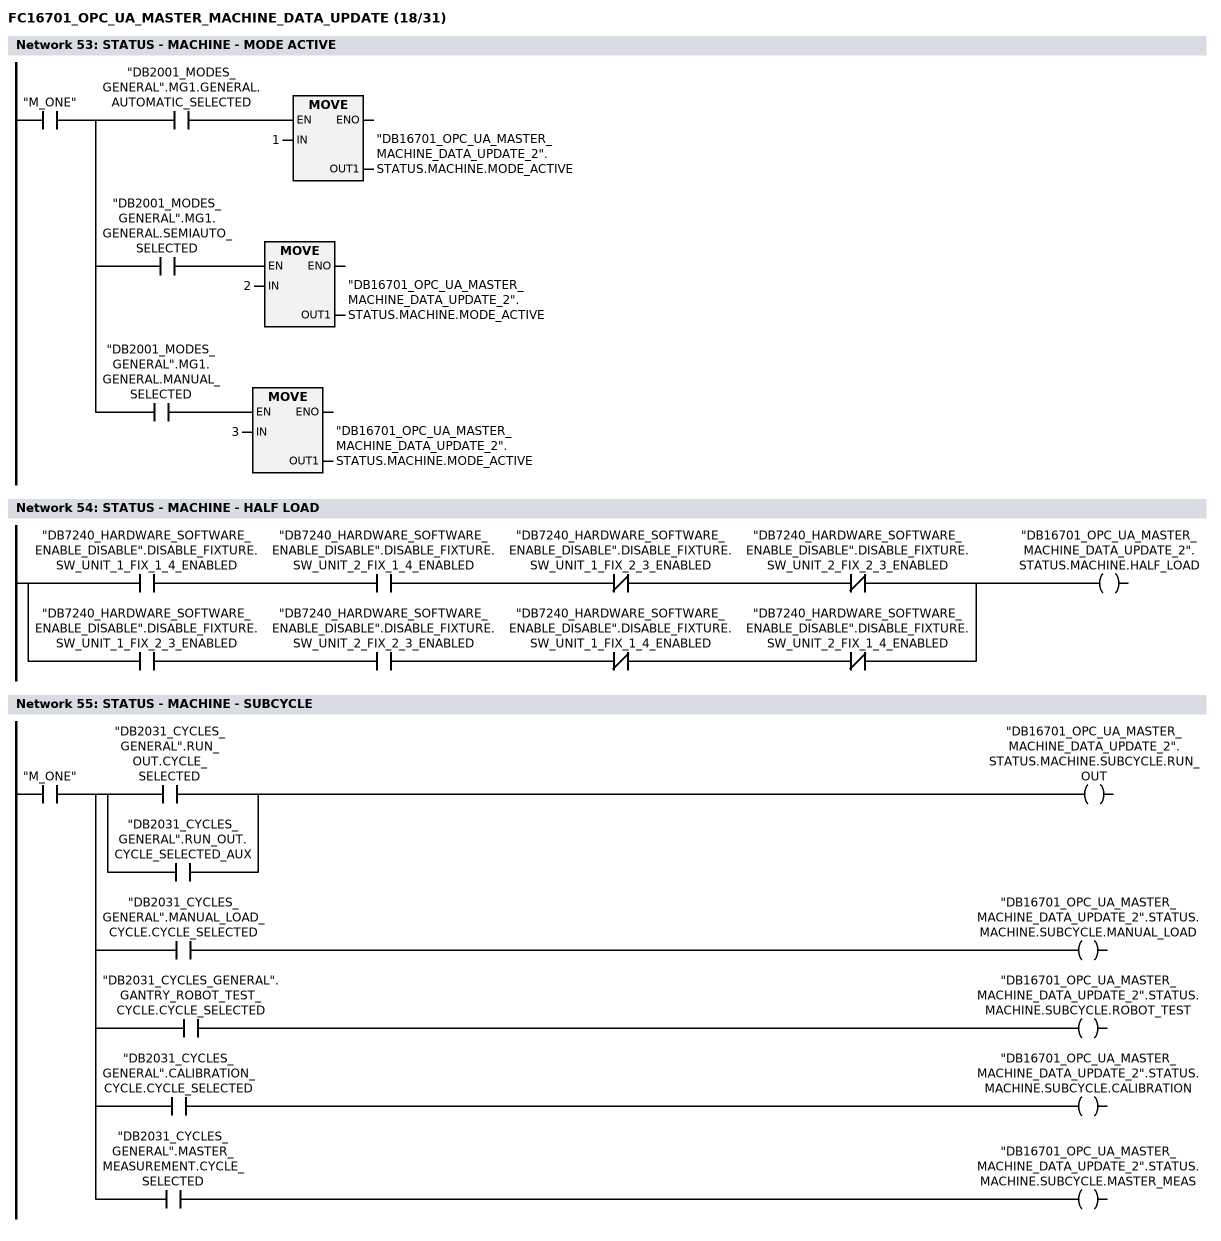
   RUNG wire#powerrail
      Contact( "M_ONE" )
      wire#w1
      Contact( "DB2001_MODES_GENERAL".MG1.GENERAL.AUTOMATIC_SELECTED )
      Move(in := 1, out1 => "DB16701_OPC_UA_MASTER_MACHINE_DATA_UPDATE_2".STATUS.MACHINE.MODE_ACTIVE)
   END_RUNG
   RUNG wire#w1
      Contact( "DB2001_MODES_GENERAL".MG1.GENERAL.SEMIAUTO_SELECTED )
      Move(in := 2, out1 => "DB16701_OPC_UA_MASTER_MACHINE_DATA_UPDATE_2".STATUS.MACHINE.MODE_ACTIVE)
   END_RUNG
   RUNG wire#w1
      Contact( "DB2001_MODES_GENERAL".MG1.GENERAL.MANUAL_SELECTED )
      Move(in := 3, out1 => "DB16701_OPC_UA_MASTER_MACHINE_DATA_UPDATE_2".STATUS.MACHINE.MODE_ACTIVE)
   END_RUNG
   // the same network as SCL:
   IF "M_ONE" AND "DB2001_MODES_GENERAL".MG1.GENERAL.AUTOMATIC_SELECTED THEN
       "DB16701_OPC_UA_MASTER_MACHINE_DATA_UPDATE_2".STATUS.MACHINE.MODE_ACTIVE := 1;
   END_IF;
   IF "M_ONE" AND "DB2001_MODES_GENERAL".MG1.GENERAL.SEMIAUTO_SELECTED THEN
       "DB16701_OPC_UA_MASTER_MACHINE_DATA_UPDATE_2".STATUS.MACHINE.MODE_ACTIVE := 2;
   END_IF;
   IF "M_ONE" AND "DB2001_MODES_GENERAL".MG1.GENERAL.MANUAL_SELECTED THEN
       "DB16701_OPC_UA_MASTER_MACHINE_DATA_UPDATE_2".STATUS.MACHINE.MODE_ACTIVE := 3;
   END_IF;
END_REGION

REGION Network 54: STATUS - MACHINE - HALF LOAD
   RUNG wire#powerrail
      Contact( "DB7240_HARDWARE_SOFTWARE_ENABLE_DISABLE".DISABLE_FIXTURE.SW_UNIT_1_FIX_1_4_ENABLED )
      Contact( "DB7240_HARDWARE_SOFTWARE_ENABLE_DISABLE".DISABLE_FIXTURE.SW_UNIT_2_FIX_1_4_ENABLED )
      I_Contact( "DB7240_HARDWARE_SOFTWARE_ENABLE_DISABLE".DISABLE_FIXTURE.SW_UNIT_1_FIX_2_3_ENABLED )
      I_Contact( "DB7240_HARDWARE_SOFTWARE_ENABLE_DISABLE".DISABLE_FIXTURE.SW_UNIT_2_FIX_2_3_ENABLED )
      wire#w1
      Coil( "DB16701_OPC_UA_MASTER_MACHINE_DATA_UPDATE_2".STATUS.MACHINE.HALF_LOAD )
   END_RUNG
   RUNG wire#powerrail
      Contact( "DB7240_HARDWARE_SOFTWARE_ENABLE_DISABLE".DISABLE_FIXTURE.SW_UNIT_1_FIX_2_3_ENABLED )
      Contact( "DB7240_HARDWARE_SOFTWARE_ENABLE_DISABLE".DISABLE_FIXTURE.SW_UNIT_2_FIX_2_3_ENABLED )
      I_Contact( "DB7240_HARDWARE_SOFTWARE_ENABLE_DISABLE".DISABLE_FIXTURE.SW_UNIT_1_FIX_1_4_ENABLED )
      I_Contact( "DB7240_HARDWARE_SOFTWARE_ENABLE_DISABLE".DISABLE_FIXTURE.SW_UNIT_2_FIX_1_4_ENABLED )
   END_RUNG wire#w1
   // the same network as SCL:
   "DB16701_OPC_UA_MASTER_MACHINE_DATA_UPDATE_2".STATUS.MACHINE.HALF_LOAD := ("DB7240_HARDWARE_SOFTWARE_ENABLE_DISABLE".DISABLE_FIXTURE.SW_UNIT_1_FIX_1_4_ENABLED AND "DB7240_HARDWARE_SOFTWARE_ENABLE_DISABLE".DISABLE_FIXTURE.SW_UNIT_2_FIX_1_4_ENABLED AND NOT "DB7240_HARDWARE_SOFTWARE_ENABLE_DISABLE".DISABLE_FIXTURE.SW_UNIT_1_FIX_2_3_ENABLED AND NOT "DB7240_HARDWARE_SOFTWARE_ENABLE_DISABLE".DISABLE_FIXTURE.SW_UNIT_2_FIX_2_3_ENABLED) OR ("DB7240_HARDWARE_SOFTWARE_ENABLE_DISABLE".DISABLE_FIXTURE.SW_UNIT_1_FIX_2_3_ENABLED AND "DB7240_HARDWARE_SOFTWARE_ENABLE_DISABLE".DISABLE_FIXTURE.SW_UNIT_2_FIX_2_3_ENABLED AND NOT "DB7240_HARDWARE_SOFTWARE_ENABLE_DISABLE".DISABLE_FIXTURE.SW_UNIT_1_FIX_1_4_ENABLED AND NOT "DB7240_HARDWARE_SOFTWARE_ENABLE_DISABLE".DISABLE_FIXTURE.SW_UNIT_2_FIX_1_4_ENABLED);
END_REGION

REGION Network 55: STATUS - MACHINE - SUBCYCLE
   RUNG wire#powerrail
      Contact( "M_ONE" )
      wire#w1
      Contact( "DB2031_CYCLES_GENERAL".RUN_OUT.CYCLE_SELECTED )
      wire#w2
      Coil( "DB16701_OPC_UA_MASTER_MACHINE_DATA_UPDATE_2".STATUS.MACHINE.SUBCYCLE.RUN_OUT )
   END_RUNG
   RUNG wire#w1
      Contact( "DB2031_CYCLES_GENERAL".RUN_OUT.CYCLE_SELECTED_AUX )
   END_RUNG wire#w2
   RUNG wire#w1
      Contact( "DB2031_CYCLES_GENERAL".MANUAL_LOAD_CYCLE.CYCLE_SELECTED )
      Coil( "DB16701_OPC_UA_MASTER_MACHINE_DATA_UPDATE_2".STATUS.MACHINE.SUBCYCLE.MANUAL_LOAD )
   END_RUNG
   RUNG wire#w1
      Contact( "DB2031_CYCLES_GENERAL".GANTRY_ROBOT_TEST_CYCLE.CYCLE_SELECTED )
      Coil( "DB16701_OPC_UA_MASTER_MACHINE_DATA_UPDATE_2".STATUS.MACHINE.SUBCYCLE.ROBOT_TEST )
   END_RUNG
   RUNG wire#w1
      Contact( "DB2031_CYCLES_GENERAL".CALIBRATION_CYCLE.CYCLE_SELECTED )
      Coil( "DB16701_OPC_UA_MASTER_MACHINE_DATA_UPDATE_2".STATUS.MACHINE.SUBCYCLE.CALIBRATION )
   END_RUNG
   RUNG wire#w1
      Contact( "DB2031_CYCLES_GENERAL".MASTER_MEASUREMENT.CYCLE_SELECTED )
      Coil( "DB16701_OPC_UA_MASTER_MACHINE_DATA_UPDATE_2".STATUS.MACHINE.SUBCYCLE.MASTER_MEAS )
   END_RUNG
   // the same network as SCL:
   "DB16701_OPC_UA_MASTER_MACHINE_DATA_UPDATE_2".STATUS.MACHINE.SUBCYCLE.RUN_OUT := "M_ONE" AND ("DB2031_CYCLES_GENERAL".RUN_OUT.CYCLE_SELECTED OR "DB2031_CYCLES_GENERAL".RUN_OUT.CYCLE_SELECTED_AUX);
   "DB16701_OPC_UA_MASTER_MACHINE_DATA_UPDATE_2".STATUS.MACHINE.SUBCYCLE.MANUAL_LOAD := "M_ONE" AND "DB2031_CYCLES_GENERAL".MANUAL_LOAD_CYCLE.CYCLE_SELECTED;
   "DB16701_OPC_UA_MASTER_MACHINE_DATA_UPDATE_2".STATUS.MACHINE.SUBCYCLE.ROBOT_TEST := "M_ONE" AND "DB2031_CYCLES_GENERAL".GANTRY_ROBOT_TEST_CYCLE.CYCLE_SELECTED;
   "DB16701_OPC_UA_MASTER_MACHINE_DATA_UPDATE_2".STATUS.MACHINE.SUBCYCLE.CALIBRATION := "M_ONE" AND "DB2031_CYCLES_GENERAL".CALIBRATION_CYCLE.CYCLE_SELECTED;
   "DB16701_OPC_UA_MASTER_MACHINE_DATA_UPDATE_2".STATUS.MACHINE.SUBCYCLE.MASTER_MEAS := "M_ONE" AND "DB2031_CYCLES_GENERAL".MASTER_MEASUREMENT.CYCLE_SELECTED;
END_REGION

REGION Network 56: STATUS - MACHINE - HARDWARE DISABLE
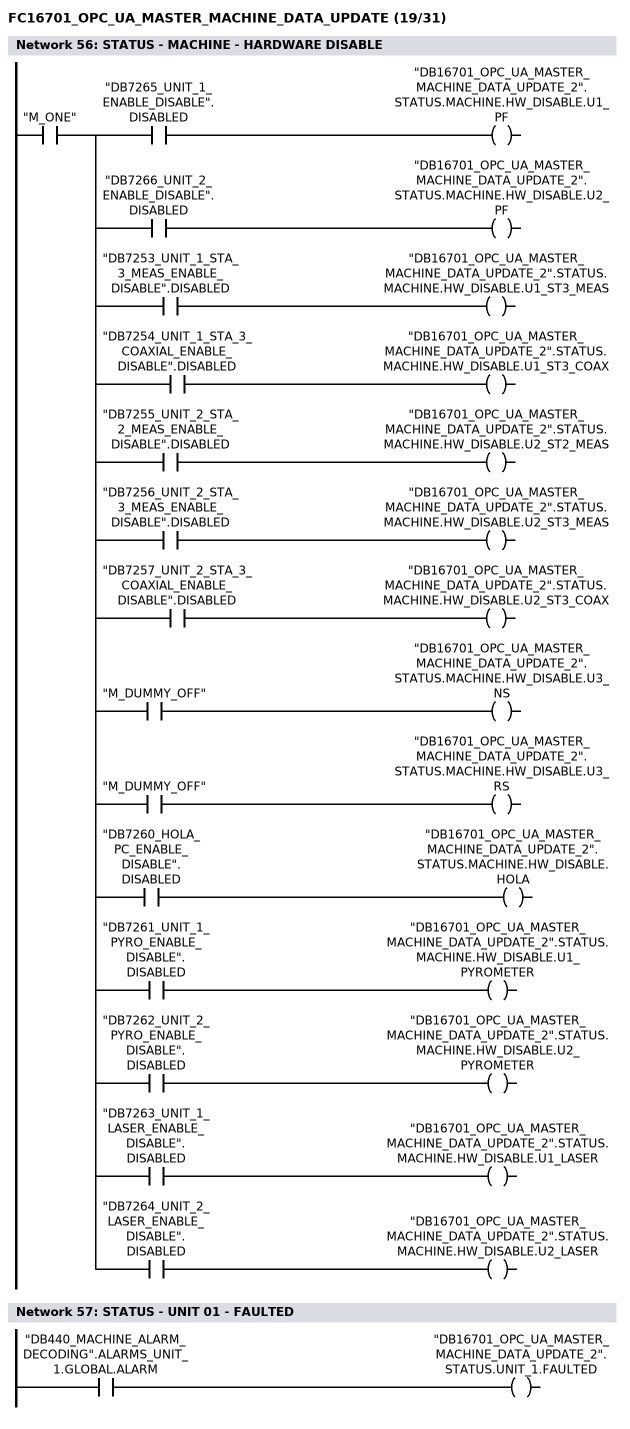
   RUNG wire#powerrail
      Contact( "M_ONE" )
      wire#w1
      Contact( "DB7265_UNIT_1_ENABLE_DISABLE".DISABLED )
      Coil( "DB16701_OPC_UA_MASTER_MACHINE_DATA_UPDATE_2".STATUS.MACHINE.HW_DISABLE.U1_PF )
   END_RUNG
   RUNG wire#w1
      Contact( "DB7266_UNIT_2_ENABLE_DISABLE".DISABLED )
      Coil( "DB16701_OPC_UA_MASTER_MACHINE_DATA_UPDATE_2".STATUS.MACHINE.HW_DISABLE.U2_PF )
   END_RUNG
   RUNG wire#w1
      Contact( "DB7253_UNIT_1_STA_3_MEAS_ENABLE_DISABLE".DISABLED )
      Coil( "DB16701_OPC_UA_MASTER_MACHINE_DATA_UPDATE_2".STATUS.MACHINE.HW_DISABLE.U1_ST3_MEAS )
   END_RUNG
   RUNG wire#w1
      Contact( "DB7254_UNIT_1_STA_3_COAXIAL_ENABLE_DISABLE".DISABLED )
      Coil( "DB16701_OPC_UA_MASTER_MACHINE_DATA_UPDATE_2".STATUS.MACHINE.HW_DISABLE.U1_ST3_COAX )
   END_RUNG
   RUNG wire#w1
      Contact( "DB7255_UNIT_2_STA_2_MEAS_ENABLE_DISABLE".DISABLED )
      Coil( "DB16701_OPC_UA_MASTER_MACHINE_DATA_UPDATE_2".STATUS.MACHINE.HW_DISABLE.U2_ST2_MEAS )
   END_RUNG
   RUNG wire#w1
      Contact( "DB7256_UNIT_2_STA_3_MEAS_ENABLE_DISABLE".DISABLED )
      Coil( "DB16701_OPC_UA_MASTER_MACHINE_DATA_UPDATE_2".STATUS.MACHINE.HW_DISABLE.U2_ST3_MEAS )
   END_RUNG
   RUNG wire#w1
      Contact( "DB7257_UNIT_2_STA_3_COAXIAL_ENABLE_DISABLE".DISABLED )
      Coil( "DB16701_OPC_UA_MASTER_MACHINE_DATA_UPDATE_2".STATUS.MACHINE.HW_DISABLE.U2_ST3_COAX )
   END_RUNG
   RUNG wire#w1
      Contact( "M_DUMMY_OFF" )
      Coil( "DB16701_OPC_UA_MASTER_MACHINE_DATA_UPDATE_2".STATUS.MACHINE.HW_DISABLE.U3_NS )
   END_RUNG
   RUNG wire#w1
      Contact( "M_DUMMY_OFF" )
      Coil( "DB16701_OPC_UA_MASTER_MACHINE_DATA_UPDATE_2".STATUS.MACHINE.HW_DISABLE.U3_RS )
   END_RUNG
   RUNG wire#w1
      Contact( "DB7260_HOLA_PC_ENABLE_DISABLE".DISABLED )
      Coil( "DB16701_OPC_UA_MASTER_MACHINE_DATA_UPDATE_2".STATUS.MACHINE.HW_DISABLE.HOLA )
   END_RUNG
   RUNG wire#w1
      Contact( "DB7261_UNIT_1_PYRO_ENABLE_DISABLE".DISABLED )
      Coil( "DB16701_OPC_UA_MASTER_MACHINE_DATA_UPDATE_2".STATUS.MACHINE.HW_DISABLE.U1_PYROMETER )
   END_RUNG
   RUNG wire#w1
      Contact( "DB7262_UNIT_2_PYRO_ENABLE_DISABLE".DISABLED )
      Coil( "DB16701_OPC_UA_MASTER_MACHINE_DATA_UPDATE_2".STATUS.MACHINE.HW_DISABLE.U2_PYROMETER )
   END_RUNG
   RUNG wire#w1
      Contact( "DB7263_UNIT_1_LASER_ENABLE_DISABLE".DISABLED )
      Coil( "DB16701_OPC_UA_MASTER_MACHINE_DATA_UPDATE_2".STATUS.MACHINE.HW_DISABLE.U1_LASER )
   END_RUNG
   RUNG wire#w1
      Contact( "DB7264_UNIT_2_LASER_ENABLE_DISABLE".DISABLED )
      Coil( "DB16701_OPC_UA_MASTER_MACHINE_DATA_UPDATE_2".STATUS.MACHINE.HW_DISABLE.U2_LASER )
   END_RUNG
   // the same network as SCL:
   "DB16701_OPC_UA_MASTER_MACHINE_DATA_UPDATE_2".STATUS.MACHINE.HW_DISABLE.U1_PF := "M_ONE" AND "DB7265_UNIT_1_ENABLE_DISABLE".DISABLED;
   "DB16701_OPC_UA_MASTER_MACHINE_DATA_UPDATE_2".STATUS.MACHINE.HW_DISABLE.U2_PF := "M_ONE" AND "DB7266_UNIT_2_ENABLE_DISABLE".DISABLED;
   "DB16701_OPC_UA_MASTER_MACHINE_DATA_UPDATE_2".STATUS.MACHINE.HW_DISABLE.U1_ST3_MEAS := "M_ONE" AND "DB7253_UNIT_1_STA_3_MEAS_ENABLE_DISABLE".DISABLED;
   "DB16701_OPC_UA_MASTER_MACHINE_DATA_UPDATE_2".STATUS.MACHINE.HW_DISABLE.U1_ST3_COAX := "M_ONE" AND "DB7254_UNIT_1_STA_3_COAXIAL_ENABLE_DISABLE".DISABLED;
   "DB16701_OPC_UA_MASTER_MACHINE_DATA_UPDATE_2".STATUS.MACHINE.HW_DISABLE.U2_ST2_MEAS := "M_ONE" AND "DB7255_UNIT_2_STA_2_MEAS_ENABLE_DISABLE".DISABLED;
   "DB16701_OPC_UA_MASTER_MACHINE_DATA_UPDATE_2".STATUS.MACHINE.HW_DISABLE.U2_ST3_MEAS := "M_ONE" AND "DB7256_UNIT_2_STA_3_MEAS_ENABLE_DISABLE".DISABLED;
   "DB16701_OPC_UA_MASTER_MACHINE_DATA_UPDATE_2".STATUS.MACHINE.HW_DISABLE.U2_ST3_COAX := "M_ONE" AND "DB7257_UNIT_2_STA_3_COAXIAL_ENABLE_DISABLE".DISABLED;
   "DB16701_OPC_UA_MASTER_MACHINE_DATA_UPDATE_2".STATUS.MACHINE.HW_DISABLE.U3_NS := "M_ONE" AND "M_DUMMY_OFF";
   "DB16701_OPC_UA_MASTER_MACHINE_DATA_UPDATE_2".STATUS.MACHINE.HW_DISABLE.U3_RS := "M_ONE" AND "M_DUMMY_OFF";
   "DB16701_OPC_UA_MASTER_MACHINE_DATA_UPDATE_2".STATUS.MACHINE.HW_DISABLE.HOLA := "M_ONE" AND "DB7260_HOLA_PC_ENABLE_DISABLE".DISABLED;
   "DB16701_OPC_UA_MASTER_MACHINE_DATA_UPDATE_2".STATUS.MACHINE.HW_DISABLE.U1_PYROMETER := "M_ONE" AND "DB7261_UNIT_1_PYRO_ENABLE_DISABLE".DISABLED;
   "DB16701_OPC_UA_MASTER_MACHINE_DATA_UPDATE_2".STATUS.MACHINE.HW_DISABLE.U2_PYROMETER := "M_ONE" AND "DB7262_UNIT_2_PYRO_ENABLE_DISABLE".DISABLED;
   "DB16701_OPC_UA_MASTER_MACHINE_DATA_UPDATE_2".STATUS.MACHINE.HW_DISABLE.U1_LASER := "M_ONE" AND "DB7263_UNIT_1_LASER_ENABLE_DISABLE".DISABLED;
   "DB16701_OPC_UA_MASTER_MACHINE_DATA_UPDATE_2".STATUS.MACHINE.HW_DISABLE.U2_LASER := "M_ONE" AND "DB7264_UNIT_2_LASER_ENABLE_DISABLE".DISABLED;
END_REGION

REGION Network 57: STATUS - UNIT 01 - FAULTED
   RUNG wire#powerrail
      Contact( "DB440_MACHINE_ALARM_DECODING".ALARMS_UNIT_1.GLOBAL.ALARM )
      Coil( "DB16701_OPC_UA_MASTER_MACHINE_DATA_UPDATE_2".STATUS.UNIT_1.FAULTED )
   END_RUNG
   // the same network as SCL:
   "DB16701_OPC_UA_MASTER_MACHINE_DATA_UPDATE_2".STATUS.UNIT_1.FAULTED := "DB440_MACHINE_ALARM_DECODING".ALARMS_UNIT_1.GLOBAL.ALARM;
END_REGION

REGION Network 58: STATUS - UNIT 01 - ST0
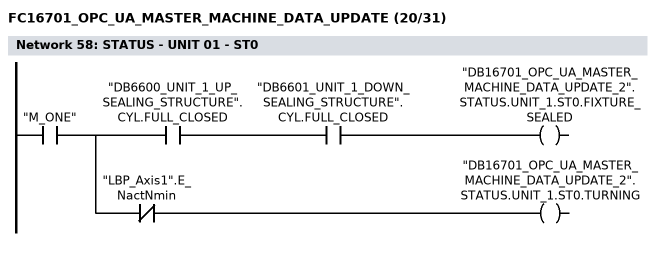
   RUNG wire#powerrail
      Contact( "M_ONE" )
      wire#w1
      Contact( "DB6600_UNIT_1_UP_SEALING_STRUCTURE".CYL.FULL_CLOSED )
      Contact( "DB6601_UNIT_1_DOWN_SEALING_STRUCTURE".CYL.FULL_CLOSED )
      Coil( "DB16701_OPC_UA_MASTER_MACHINE_DATA_UPDATE_2".STATUS.UNIT_1.ST0.FIXTURE_SEALED )
   END_RUNG
   RUNG wire#w1
      I_Contact( "LBP_Axis1".E_NactNmin )
      Coil( "DB16701_OPC_UA_MASTER_MACHINE_DATA_UPDATE_2".STATUS.UNIT_1.ST0.TURNING )
   END_RUNG
   // the same network as SCL:
   "DB16701_OPC_UA_MASTER_MACHINE_DATA_UPDATE_2".STATUS.UNIT_1.ST0.FIXTURE_SEALED := "M_ONE" AND "DB6600_UNIT_1_UP_SEALING_STRUCTURE".CYL.FULL_CLOSED AND "DB6601_UNIT_1_DOWN_SEALING_STRUCTURE".CYL.FULL_CLOSED;
   "DB16701_OPC_UA_MASTER_MACHINE_DATA_UPDATE_2".STATUS.UNIT_1.ST0.TURNING := "M_ONE" AND NOT "LBP_Axis1".E_NactNmin;
END_REGION

REGION Network 59: STATUS - UNIT 01 - ST1
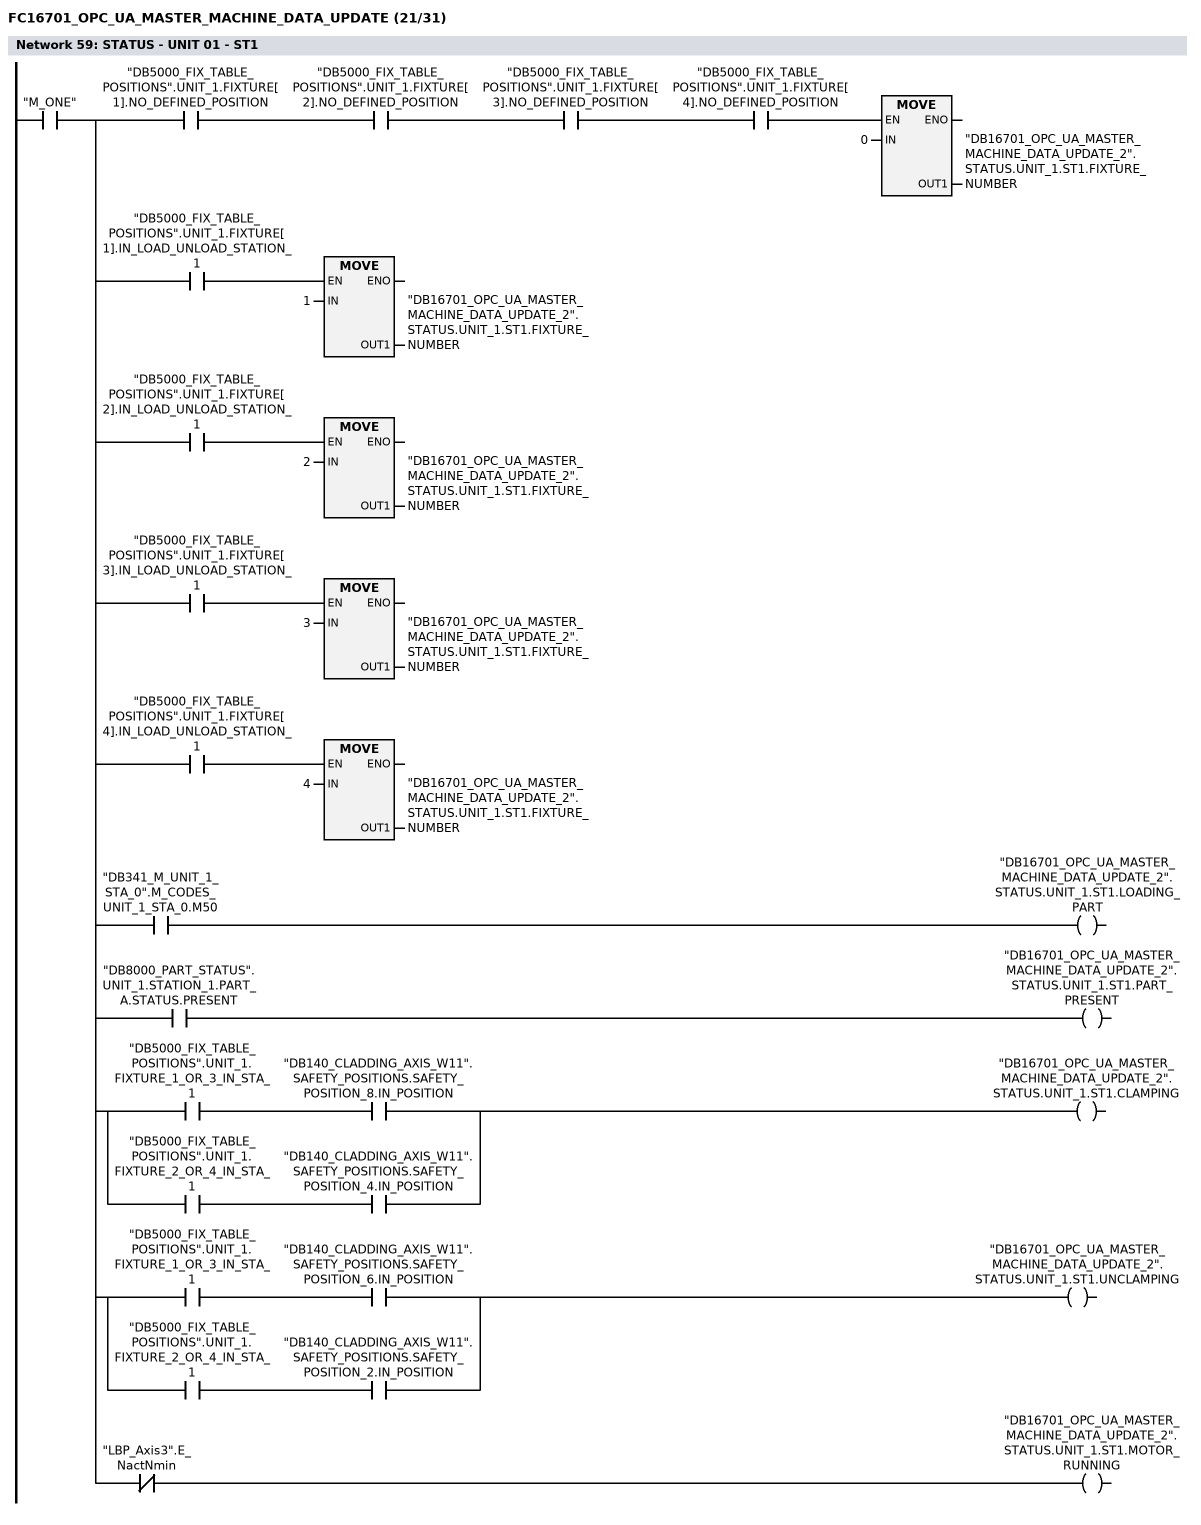
   RUNG wire#powerrail
      Contact( "M_ONE" )
      wire#w1
      Contact( "DB5000_FIX_TABLE_POSITIONS".UNIT_1.FIXTURE[1].NO_DEFINED_POSITION )
      Contact( "DB5000_FIX_TABLE_POSITIONS".UNIT_1.FIXTURE[2].NO_DEFINED_POSITION )
      Contact( "DB5000_FIX_TABLE_POSITIONS".UNIT_1.FIXTURE[3].NO_DEFINED_POSITION )
      Contact( "DB5000_FIX_TABLE_POSITIONS".UNIT_1.FIXTURE[4].NO_DEFINED_POSITION )
      Move(in := 0, out1 => "DB16701_OPC_UA_MASTER_MACHINE_DATA_UPDATE_2".STATUS.UNIT_1.ST1.FIXTURE_NUMBER)
   END_RUNG
   RUNG wire#w1
      Contact( "DB5000_FIX_TABLE_POSITIONS".UNIT_1.FIXTURE[1].IN_LOAD_UNLOAD_STATION_1 )
      Move(in := 1, out1 => "DB16701_OPC_UA_MASTER_MACHINE_DATA_UPDATE_2".STATUS.UNIT_1.ST1.FIXTURE_NUMBER)
   END_RUNG
   RUNG wire#w1
      Contact( "DB5000_FIX_TABLE_POSITIONS".UNIT_1.FIXTURE[2].IN_LOAD_UNLOAD_STATION_1 )
      Move(in := 2, out1 => "DB16701_OPC_UA_MASTER_MACHINE_DATA_UPDATE_2".STATUS.UNIT_1.ST1.FIXTURE_NUMBER)
   END_RUNG
   RUNG wire#w1
      Contact( "DB5000_FIX_TABLE_POSITIONS".UNIT_1.FIXTURE[3].IN_LOAD_UNLOAD_STATION_1 )
      Move(in := 3, out1 => "DB16701_OPC_UA_MASTER_MACHINE_DATA_UPDATE_2".STATUS.UNIT_1.ST1.FIXTURE_NUMBER)
   END_RUNG
   RUNG wire#w1
      Contact( "DB5000_FIX_TABLE_POSITIONS".UNIT_1.FIXTURE[4].IN_LOAD_UNLOAD_STATION_1 )
      Move(in := 4, out1 => "DB16701_OPC_UA_MASTER_MACHINE_DATA_UPDATE_2".STATUS.UNIT_1.ST1.FIXTURE_NUMBER)
   END_RUNG
   RUNG wire#w1
      Contact( "DB341_M_UNIT_1_STA_0".M_CODES_UNIT_1_STA_0.M50 )
      Coil( "DB16701_OPC_UA_MASTER_MACHINE_DATA_UPDATE_2".STATUS.UNIT_1.ST1.LOADING_PART )
   END_RUNG
   RUNG wire#w1
      Contact( "DB8000_PART_STATUS".UNIT_1.STATION_1.PART_A.STATUS.PRESENT )
      Coil( "DB16701_OPC_UA_MASTER_MACHINE_DATA_UPDATE_2".STATUS.UNIT_1.ST1.PART_PRESENT )
   END_RUNG
   RUNG wire#w1
      Contact( "DB5000_FIX_TABLE_POSITIONS".UNIT_1.FIXTURE_1_OR_3_IN_STA_1 )
      Contact( "DB140_CLADDING_AXIS_W11".SAFETY_POSITIONS.SAFETY_POSITION_8.IN_POSITION )
      wire#w2
      Coil( "DB16701_OPC_UA_MASTER_MACHINE_DATA_UPDATE_2".STATUS.UNIT_1.ST1.CLAMPING )
   END_RUNG
   RUNG wire#w1
      Contact( "DB5000_FIX_TABLE_POSITIONS".UNIT_1.FIXTURE_2_OR_4_IN_STA_1 )
      Contact( "DB140_CLADDING_AXIS_W11".SAFETY_POSITIONS.SAFETY_POSITION_4.IN_POSITION )
   END_RUNG wire#w2
   RUNG wire#w1
      Contact( "DB5000_FIX_TABLE_POSITIONS".UNIT_1.FIXTURE_1_OR_3_IN_STA_1 )
      Contact( "DB140_CLADDING_AXIS_W11".SAFETY_POSITIONS.SAFETY_POSITION_6.IN_POSITION )
      wire#w3
      Coil( "DB16701_OPC_UA_MASTER_MACHINE_DATA_UPDATE_2".STATUS.UNIT_1.ST1.UNCLAMPING )
   END_RUNG
   RUNG wire#w1
      Contact( "DB5000_FIX_TABLE_POSITIONS".UNIT_1.FIXTURE_2_OR_4_IN_STA_1 )
      Contact( "DB140_CLADDING_AXIS_W11".SAFETY_POSITIONS.SAFETY_POSITION_2.IN_POSITION )
   END_RUNG wire#w3
   RUNG wire#w1
      I_Contact( "LBP_Axis3".E_NactNmin )
      Coil( "DB16701_OPC_UA_MASTER_MACHINE_DATA_UPDATE_2".STATUS.UNIT_1.ST1.MOTOR_RUNNING )
   END_RUNG
   // the same network as SCL:
   IF "M_ONE" AND "DB5000_FIX_TABLE_POSITIONS".UNIT_1.FIXTURE[1].NO_DEFINED_POSITION AND "DB5000_FIX_TABLE_POSITIONS".UNIT_1.FIXTURE[2].NO_DEFINED_POSITION AND "DB5000_FIX_TABLE_POSITIONS".UNIT_1.FIXTURE[3].NO_DEFINED_POSITION AND "DB5000_FIX_TABLE_POSITIONS".UNIT_1.FIXTURE[4].NO_DEFINED_POSITION THEN
       "DB16701_OPC_UA_MASTER_MACHINE_DATA_UPDATE_2".STATUS.UNIT_1.ST1.FIXTURE_NUMBER := 0;
   END_IF;
   IF "M_ONE" AND "DB5000_FIX_TABLE_POSITIONS".UNIT_1.FIXTURE[1].IN_LOAD_UNLOAD_STATION_1 THEN
       "DB16701_OPC_UA_MASTER_MACHINE_DATA_UPDATE_2".STATUS.UNIT_1.ST1.FIXTURE_NUMBER := 1;
   END_IF;
   IF "M_ONE" AND "DB5000_FIX_TABLE_POSITIONS".UNIT_1.FIXTURE[2].IN_LOAD_UNLOAD_STATION_1 THEN
       "DB16701_OPC_UA_MASTER_MACHINE_DATA_UPDATE_2".STATUS.UNIT_1.ST1.FIXTURE_NUMBER := 2;
   END_IF;
   IF "M_ONE" AND "DB5000_FIX_TABLE_POSITIONS".UNIT_1.FIXTURE[3].IN_LOAD_UNLOAD_STATION_1 THEN
       "DB16701_OPC_UA_MASTER_MACHINE_DATA_UPDATE_2".STATUS.UNIT_1.ST1.FIXTURE_NUMBER := 3;
   END_IF;
   IF "M_ONE" AND "DB5000_FIX_TABLE_POSITIONS".UNIT_1.FIXTURE[4].IN_LOAD_UNLOAD_STATION_1 THEN
       "DB16701_OPC_UA_MASTER_MACHINE_DATA_UPDATE_2".STATUS.UNIT_1.ST1.FIXTURE_NUMBER := 4;
   END_IF;
   "DB16701_OPC_UA_MASTER_MACHINE_DATA_UPDATE_2".STATUS.UNIT_1.ST1.LOADING_PART := "M_ONE" AND "DB341_M_UNIT_1_STA_0".M_CODES_UNIT_1_STA_0.M50;
   "DB16701_OPC_UA_MASTER_MACHINE_DATA_UPDATE_2".STATUS.UNIT_1.ST1.PART_PRESENT := "M_ONE" AND "DB8000_PART_STATUS".UNIT_1.STATION_1.PART_A.STATUS.PRESENT;
   "DB16701_OPC_UA_MASTER_MACHINE_DATA_UPDATE_2".STATUS.UNIT_1.ST1.CLAMPING := "M_ONE" AND (("DB5000_FIX_TABLE_POSITIONS".UNIT_1.FIXTURE_1_OR_3_IN_STA_1 AND "DB140_CLADDING_AXIS_W11".SAFETY_POSITIONS.SAFETY_POSITION_8.IN_POSITION) OR ("DB5000_FIX_TABLE_POSITIONS".UNIT_1.FIXTURE_2_OR_4_IN_STA_1 AND "DB140_CLADDING_AXIS_W11".SAFETY_POSITIONS.SAFETY_POSITION_4.IN_POSITION));
   "DB16701_OPC_UA_MASTER_MACHINE_DATA_UPDATE_2".STATUS.UNIT_1.ST1.UNCLAMPING := "M_ONE" AND (("DB5000_FIX_TABLE_POSITIONS".UNIT_1.FIXTURE_1_OR_3_IN_STA_1 AND "DB140_CLADDING_AXIS_W11".SAFETY_POSITIONS.SAFETY_POSITION_6.IN_POSITION) OR ("DB5000_FIX_TABLE_POSITIONS".UNIT_1.FIXTURE_2_OR_4_IN_STA_1 AND "DB140_CLADDING_AXIS_W11".SAFETY_POSITIONS.SAFETY_POSITION_2.IN_POSITION));
   "DB16701_OPC_UA_MASTER_MACHINE_DATA_UPDATE_2".STATUS.UNIT_1.ST1.MOTOR_RUNNING := "M_ONE" AND NOT "LBP_Axis3".E_NactNmin;
END_REGION

